(* IEC 61131-3 sources: volt/packages/volt-lsp-iec/test-corpus/pro2193/Device/Plc Logic/Application/09 Misc/Library Manager/BrinkEdgePcLogging, 50 files *)

(* ---- ANYNUMBER.dut ---- *)
TYPE ANYNUMBER :
UNION
	SINTVAL : SINT;
	USINTVAL : USINT;
	INTVAL : INT;
	UINTVAL : UINT;
	DINTVAL : DINT;
	UDINTVAL : UDINT;
	LINTVAL : LINT;
	ULINTVAL : ULINT;
	REALVALUE : REAL;
	LREALVALUE : LREAL;
END_UNION
END_TYPE

(* ---- CACHESTATUS.dut ---- *)
TYPE CACHESTATUS :
STRUCT
	LOCK : DWORD;
	COUNT : BYTE;
END_STRUCT
END_TYPE

(* ---- CAVITYPLCDATATYPES.dut ---- *)
TYPE CAVITYPLCDATATYPES :
STRUCT
	PRODUCED : PlcDataType := -1;
	UNCOUNTEDREJECT : PlcDataType := -1;
	REJECTED : PlcDataType := -1;
	REJECTREASONS : ARRAY [0..20] OF PlcDataType := [21(-1)];
	STACKED : PlcDataType := -1;
END_STRUCT
END_TYPE

(* ---- CLIENTSTATISTICS.dut ---- *)
TYPE CLIENTSTATISTICS :
STRUCT
	LOGFAILDISCONNECTED : ULINT;
	RECONNECTCOUNT : ULINT;
	LOSTDUETOCONNECTIONPROBLEMS : ULINT;
	KEEPALIVEMESSAGESSENT : ULINT;
	PLCDATATYPENOTDEFINED : ULINT;
	SENDNOTIMMEDIATELYCOMPLETED : ULINT;
	DATATOOLONG : ULINT;
	LOGQUEUESFULL : ULINT;
	LOGQUEUESBUSY : ULINT;
	ERRORWHILESENDINGDATA : ULINT;
	WRITEISBUSY : ULINT;
	TOOMANYWRITESPERCYCLE : ULINT;
END_STRUCT
END_TYPE

(* ---- CONNECTIONSPEED.dut ---- *)
TYPE CONNECTIONSPEED :
(
	S100MBPS := 100,
	S1000MBPS := 1000
);
END_TYPE

(* ---- DATATYPE.dut ---- *)
TYPE DATATYPE :
(
	NONE := -1,
	ULINTEGER := 0,
	INTEGER := 1,
	FLOAT := 2,
	BOOLEAN := 3,
	TEXT := 4
);
END_TYPE

(* ---- DEBUGLOGINFO.dut ---- *)
TYPE DEBUGLOGINFO :
STRUCT
	MSTIME : ULINT;
	DESCRIPTION : STRING(255);
END_STRUCT
END_TYPE

(* ---- LABELADJUSTMENTSPLCDATATYPESCONFIG.dut ---- *)
TYPE LABELADJUSTMENTSPLCDATATYPESCONFIG : ARRAY [1..2, 1..2, 1..32, 1..3] OF PlcDataType;
END_TYPE

(* ---- LOGCACHE.dut ---- *)
TYPE LOGCACHE : ARRAY [1..QueuesInCache] OF LogQueue;
END_TYPE

(* ---- LOGQUEUESTATS.dut ---- *)
TYPE LOGQUEUESTATS :
STRUCT
	ADDLOGFAILEDDUETOQUEUEFULL : ULINT;
END_STRUCT
END_TYPE

(* ---- LOGRECORD.dut ---- *)
TYPE LOGRECORD :
STRUCT
	PLCDATATYPE : PlcDataType;
	DATATYPE : DataType;
	PLCUTCTIME : ULINT;
	VALUE : NumberUnion;
END_STRUCT
END_TYPE

(* ---- LOGRECORDARRAY.dut ---- *)
TYPE LOGRECORDARRAY : ARRAY [1..GVL_Dashboard.LogQueueLength] OF LogRecord;
END_TYPE

(* ---- MOULDCONTROLCAVITYPLCDATATYPES.dut ---- *)
TYPE MOULDCONTROLCAVITYPLCDATATYPES :
STRUCT
	PEAKPRESSURE : PlcDataType := -1;
	TARGETVALUE : PlcDataType := -1;
	ACTUALVALUE : PlcDataType := -1;
END_STRUCT
END_TYPE

(* ---- MOULDCONTROLCAVITYPLCDATATYPESCONFIG.dut ---- *)
TYPE MOULDCONTROLCAVITYPLCDATATYPESCONFIG : ARRAY [1..64] OF MouldControlCavityPlcDataTypes;
END_TYPE

(* ---- MVACUUMSPLCDATATYPESCONFIG.dut ---- *)
TYPE MVACUUMSPLCDATATYPESCONFIG : ARRAY [1..2, 1..32] OF PlcDataType;
END_TYPE

(* ---- NUMBERUNION.dut ---- *)
TYPE NUMBERUNION :
UNION
	BOOLVALUE : BOOL;
	INTVALUE : LINT;
	UINTVALUE : ULINT;
	REALVALUE : LREAL;
END_UNION
END_TYPE

(* ---- PLCDATATYPE.dut ---- *)
TYPE PLCDATATYPE :
(
	MAIN_ROBOTSTATUS := 23,
	MAIN_ENABLEIML := 24,
	MAIN_ENABLEHMU := 25,
	MAIN_ENABLEVISION := 26,
	MAIN_RELAYS_HIGHVACUUMPUMPRUNNING := 27,
	MAIN_RELAYS_LOWVACUUMPUMPRUNNING := 28,
	RELAYS_MOULDAREAFREE := 29,
	RELAYS_ENABLEMOULDCLOSURE := 30,
	RELAYS_ENABLEFULLMOULDOPENING := 31,
	RELAYS_OPERATIONWITHROBOT := 32,
	RELAYS_ENABLEEJECTORBACK := 33,
	RELAYS_ENABLEEJECTORFORWARD := 34,
	RELAYS_ENABLECOREPOS1BACK := 35,
	RELAYS_ENABLECOREPOS2FORWARD := 36,
	RELAYS_GLOBALRESET := 37,
	RELAYS_MAINAIRVALVE := 38,
	RELAYS_YUNIT_MOTORCOOLING := 39,
	RELAYS_ENABLEFREQUENCYCONTROLLER := 40,
	RELAYS_SAFETYGATE := 41,
	YUNIT_ACTPOS := 42,
	YUNIT_ERRORID := 43,
	YUNIT_AXISERRORID := 44,
	YUNIT_DRIVEERRORID := 45,
	YUNIT_DRIVEUTILISATION := 46,
	YUNIT_MOTORUTILISATION := 47,
	XRUNIT_ACTPOS := 48,
	XRUNIT_ERRORID := 49,
	XRUNIT_AXISERRORID := 50,
	XRUNIT_DRIVEERRORID := 51,
	XRUNIT_DRIVEUTILISATION := 52,
	XRUNIT_MOTORUTILISATION := 53,
	XIUNIT_ACTPOS := 54,
	XIUNIT_ERRORID := 55,
	XIUNIT_AXISERRORID := 56,
	XIUNIT_DRIVEERRORID := 57,
	XIUNIT_DRIVEUTILISATION := 58,
	XIUNIT_MOTORUTILISATION := 59,
	XUUNIT_ACTPOS := 60,
	XUUNIT_ERRORID := 61,
	XUUNIT_AXISERRORID := 62,
	XUUNIT_DRIVEERRORID := 63,
	XUUNIT_DRIVEUTILISATION := 64,
	XUUNIT_MOTORUTILISATION := 65,
	CHAIN_ACTPOS := 66,
	CHAIN_ERRORID := 67,
	CHAIN_AXISERRORID := 68,
	CHAIN_DRIVEERRORID := 69,
	CHAIN_DRIVEUTILISATION := 70,
	CHAIN_MOTORUTILISATION := 71,
	MAGAZINE_M1_1_ACTPOS := 72,
	MAGAZINE_M1_1_ERRORID := 73,
	MAGAZINE_M1_1_AXISERRORID := 74,
	MAGAZINE_M1_1_DRIVEERRORID := 75,
	MAGAZINE_M1_1_DRIVEUTILISATION := 76,
	MAGAZINE_M1_1_MOTORUTILISATION := 77,
	MAGAZINE_M1_2_ACTPOS := 78,
	MAGAZINE_M1_2_ERRORID := 79,
	MAGAZINE_M1_2_AXISERRORID := 80,
	MAGAZINE_M1_2_DRIVEERRORID := 81,
	MAGAZINE_M1_2_DRIVEUTILISATION := 82,
	MAGAZINE_M1_2_MOTORUTILISATION := 83,
	ZUNIT_ACTPOS := 84,
	ZUNIT_ERRORID := 85,
	ZUNIT_AXISERRORID := 86,
	ZUNIT_DRIVEERRORID := 87,
	ZUNIT_DRIVEUTILISATION := 88,
	ZUNIT_MOTORUTILISATION := 89,
	YUNIT_ACTTORQUE := 90,
	XRUNIT_ACTTORQUE := 91,
	XIUNIT_ACTTORQUE := 92,
	XUUNIT_ACTTORQUE := 93,
	CHAIN_ACTTORQUE := 94,
	MAGAZINE_M1_1_ACTTORQUE := 95,
	MAGAZINE_M1_2_ACTTORQUE := 96,
	ZUNIT_ACTTORQUE := 97,
	YUNIT_COVEREDDISTANCE := 98,
	XRUNIT_COVEREDDISTANCE := 99,
	XIUNIT_COVEREDDISTANCE := 100,
	XUUNIT_COVEREDDISTANCE := 101,
	CHAIN_COVEREDDISTANCE := 102,
	MAGAZINE_M1_1_COVEREDDISTANCE := 103,
	MAGAZINE_M1_2_COVEREDDISTANCE := 104,
	ZUNIT_COVEREDDISTANCE := 105,
	CYCLETIMES_TIMESTOPPED := 106,
	CYCLETIMES_TIMERESETTING := 107,
	CYCLETIMES_TIMEIDLE := 108,
	CYCLETIMES_TIMEAUTOMATIC := 109,
	CYCLETIMES_AUTOMATICCYCLESTARTS := 110,
	YUNIT_ALARMS := 111,
	YUNIT_TIME_ACTIVE := 112,
	YUNIT_TIME_IDLE := 113,
	XRUNIT_ALARMS := 114,
	XRUNIT_TIME_ACTIVE := 115,
	XRUNIT_TIME_IDLE := 116,
	XIUNIT_ALARMS := 117,
	XIUNIT_TIME_ACTIVE := 118,
	XIUNIT_TIME_IDLE := 119,
	XUUNIT_ALARMS := 120,
	XUUNIT_TIME_ACTIVE := 121,
	XUUNIT_TIME_IDLE := 122,
	CHAIN_ALARMS := 123,
	CHAIN_TIME_ACTIVE := 124,
	CHAIN_TIME_IDLE := 125,
	MAGAZINE_M1_1_ALARMS := 126,
	MAGAZINE_M1_1_TIME_ACTIVE := 127,
	MAGAZINE_M1_1_TIME_IDLE := 128,
	MAGAZINE_M1_2_ALARMS := 129,
	MAGAZINE_M1_2_TIME_ACTIVE := 130,
	MAGAZINE_M1_2_TIME_IDLE := 131,
	ZUNIT_ALARMS := 132,
	ZUNIT_TIME_ACTIVE := 133,
	ZUNIT_TIME_IDLE := 134,
	CAMERA_ALARMS := 135,
	CAMERA_TIME_ACTIVE := 136,
	CAMERA_TIME_IDLE := 137,
	REJECTSTATION_ALARMS := 138,
	REJECTSTATION_TIME_ACTIVE := 139,
	REJECTSTATION_TIME_IDLE := 140,
	CONVEYORS_ALARMS := 141,
	CONVEYORS_TIME_ACTIVE := 142,
	CONVEYORS_TIME_IDLE := 143,
	IMM_CYCLETIMETAKEOUT := 144,
	IMM_CYCLETIMETOTAL := 145,
	IMM_SAVEDCYCLETIMEBYEARLYMOULDCLOSING := 146,
	XUUNIT_SENSORTIMES_VACUUM_1 := 147,
	XUUNIT_SENSORTIMES_VACUUM_2 := 148,
	XUUNIT_SENSORTIMES_VACUUM_3 := 149,
	XUUNIT_SENSORTIMES_SHIFTIN := 150,
	XUUNIT_SENSORTIMES_SHIFTOUT := 151,
	MAGAZINE_SENSORTIMES_VACUUM_1 := 152,
	MAGAZINE_SENSORTIMES_VACUUM_2 := 153,
	MAGAZINE_SENSORTIMES_VACUUM_3 := 154,
	MAGAZINE_SENSORTIMES_VACUUM_4 := 155,
	MAGAZINE_SENSORTIMES_FLIPLABEL1IN := 156,
	MAGAZINE_SENSORTIMES_FLIPLABEL1OUT := 157,
	MAGAZINE_SENSORTIMES_FLIPLABEL2IN := 158,
	MAGAZINE_SENSORTIMES_FLIPLABEL2OUT := 159,
	MAGAZINE_SENSORTIMES_CHANGEDRAWERIN := 160,
	MAGAZINE_SENSORTIMES_CHANGEDRAWEROUT := 161,
	MAGAZINE_SENSORTIMES_LOCKDRAWERIN := 162,
	MAGAZINE_SENSORTIMES_LOCKDRAWEROUT := 163,
	ZUNIT_SENSORTIMES_VACUUM_1 := 164,
	ZUNIT_SENSORTIMES_VACUUM_2 := 165,
	ZUNIT_SENSORTIMES_VACUUM_3 := 166,
	ZUNIT_SENSORTIMES_VACUUM_4 := 167,
	ZUNIT_SENSORTIMES_ROTATEIN := 168,
	ZUNIT_SENSORTIMES_ROTATEOUT := 169,
	ZUNIT_SENSORTIMES_EXTEND1IN := 170,
	ZUNIT_SENSORTIMES_EXTEND2IN := 171,
	ZUNIT_SENSORTIMES_EXTEND3IN := 172,
	ZUNIT_SENSORTIMES_EXTEND4IN := 173,
	REJECTSTATION_SENSORTIMES_REJECTCYLINDERIN := 174,
	REJECTSTATION_SENSORTIMES_REJECTCYLINDEROUT := 175,
	METADATA_REJECTREASON_0_DESCRIPTION := 176,
	METADATA_REJECTREASON_1_DESCRIPTION := 177,
	METADATA_REJECTREASON_2_DESCRIPTION := 178,
	METADATA_REJECTREASON_3_DESCRIPTION := 179,
	METADATA_REJECTREASON_4_DESCRIPTION := 180,
	METADATA_REJECTREASON_5_DESCRIPTION := 181,
	METADATA_REJECTREASON_6_DESCRIPTION := 182,
	PRODUCTIONCOUNTERS_TOTAL_PRODUCED := 183,
	PRODUCTIONCOUNTERS_TOTAL_STACKED := 184,
	PRODUCTIONCOUNTERS_TOTAL_REJECTED := 185,
	PRODUCTIONCOUNTERS_TOTAL_UNCOUNTEDREJECT := 186,
	PRODUCTIONCOUNTERS_TOTAL_REJECTREASON_0 := 187,
	PRODUCTIONCOUNTERS_TOTAL_REJECTREASON_1 := 188,
	PRODUCTIONCOUNTERS_TOTAL_REJECTREASON_2 := 189,
	PRODUCTIONCOUNTERS_TOTAL_REJECTREASON_3 := 190,
	PRODUCTIONCOUNTERS_TOTAL_REJECTREASON_4 := 191,
	PRODUCTIONCOUNTERS_TOTAL_REJECTREASON_5 := 192,
	PRODUCTIONCOUNTERS_TOTAL_REJECTREASON_6 := 193,
	PRODUCTIONCOUNTERS_CAVITY_1_PRODUCED := 194,
	PRODUCTIONCOUNTERS_CAVITY_1_STACKED := 195,
	PRODUCTIONCOUNTERS_CAVITY_1_REJECTED := 196,
	PRODUCTIONCOUNTERS_CAVITY_1_UNCOUNTEDREJECT := 197,
	PRODUCTIONCOUNTERS_CAVITY_1_REJECTREASON_0 := 198,
	PRODUCTIONCOUNTERS_CAVITY_1_REJECTREASON_1 := 199,
	PRODUCTIONCOUNTERS_CAVITY_1_REJECTREASON_2 := 200,
	PRODUCTIONCOUNTERS_CAVITY_1_REJECTREASON_3 := 201,
	PRODUCTIONCOUNTERS_CAVITY_1_REJECTREASON_4 := 202,
	PRODUCTIONCOUNTERS_CAVITY_1_REJECTREASON_5 := 203,
	PRODUCTIONCOUNTERS_CAVITY_1_REJECTREASON_6 := 204,
	PRODUCTIONCOUNTERS_CAVITY_2_PRODUCED := 205,
	PRODUCTIONCOUNTERS_CAVITY_2_STACKED := 206,
	PRODUCTIONCOUNTERS_CAVITY_2_REJECTED := 207,
	PRODUCTIONCOUNTERS_CAVITY_2_UNCOUNTEDREJECT := 208,
	PRODUCTIONCOUNTERS_CAVITY_2_REJECTREASON_0 := 209,
	PRODUCTIONCOUNTERS_CAVITY_2_REJECTREASON_1 := 210,
	PRODUCTIONCOUNTERS_CAVITY_2_REJECTREASON_2 := 211,
	PRODUCTIONCOUNTERS_CAVITY_2_REJECTREASON_3 := 212,
	PRODUCTIONCOUNTERS_CAVITY_2_REJECTREASON_4 := 213,
	PRODUCTIONCOUNTERS_CAVITY_2_REJECTREASON_5 := 214,
	PRODUCTIONCOUNTERS_CAVITY_2_REJECTREASON_6 := 215,
	PRODUCTIONCOUNTERS_CAVITY_3_PRODUCED := 216,
	PRODUCTIONCOUNTERS_CAVITY_3_STACKED := 217,
	PRODUCTIONCOUNTERS_CAVITY_3_REJECTED := 218,
	PRODUCTIONCOUNTERS_CAVITY_3_UNCOUNTEDREJECT := 219,
	PRODUCTIONCOUNTERS_CAVITY_3_REJECTREASON_0 := 220,
	PRODUCTIONCOUNTERS_CAVITY_3_REJECTREASON_1 := 221,
	PRODUCTIONCOUNTERS_CAVITY_3_REJECTREASON_2 := 222,
	PRODUCTIONCOUNTERS_CAVITY_3_REJECTREASON_3 := 223,
	PRODUCTIONCOUNTERS_CAVITY_3_REJECTREASON_4 := 224,
	PRODUCTIONCOUNTERS_CAVITY_3_REJECTREASON_5 := 225,
	PRODUCTIONCOUNTERS_CAVITY_3_REJECTREASON_6 := 226,
	PRODUCTIONCOUNTERS_CAVITY_4_PRODUCED := 227,
	PRODUCTIONCOUNTERS_CAVITY_4_STACKED := 228,
	PRODUCTIONCOUNTERS_CAVITY_4_REJECTED := 229,
	PRODUCTIONCOUNTERS_CAVITY_4_UNCOUNTEDREJECT := 230,
	PRODUCTIONCOUNTERS_CAVITY_4_REJECTREASON_0 := 231,
	PRODUCTIONCOUNTERS_CAVITY_4_REJECTREASON_1 := 232,
	PRODUCTIONCOUNTERS_CAVITY_4_REJECTREASON_2 := 233,
	PRODUCTIONCOUNTERS_CAVITY_4_REJECTREASON_3 := 234,
	PRODUCTIONCOUNTERS_CAVITY_4_REJECTREASON_4 := 235,
	PRODUCTIONCOUNTERS_CAVITY_4_REJECTREASON_5 := 236,
	PRODUCTIONCOUNTERS_CAVITY_4_REJECTREASON_6 := 237,
	PRODUCTIONCOUNTERS_CAVITY_5_PRODUCED := 238,
	PRODUCTIONCOUNTERS_CAVITY_5_STACKED := 239,
	PRODUCTIONCOUNTERS_CAVITY_5_REJECTED := 240,
	PRODUCTIONCOUNTERS_CAVITY_5_UNCOUNTEDREJECT := 241,
	PRODUCTIONCOUNTERS_CAVITY_5_REJECTREASON_0 := 242,
	PRODUCTIONCOUNTERS_CAVITY_5_REJECTREASON_1 := 243,
	PRODUCTIONCOUNTERS_CAVITY_5_REJECTREASON_2 := 244,
	PRODUCTIONCOUNTERS_CAVITY_5_REJECTREASON_3 := 245,
	PRODUCTIONCOUNTERS_CAVITY_5_REJECTREASON_4 := 246,
	PRODUCTIONCOUNTERS_CAVITY_5_REJECTREASON_5 := 247,
	PRODUCTIONCOUNTERS_CAVITY_5_REJECTREASON_6 := 248,
	PRODUCTIONCOUNTERS_CAVITY_6_PRODUCED := 249,
	PRODUCTIONCOUNTERS_CAVITY_6_STACKED := 250,
	PRODUCTIONCOUNTERS_CAVITY_6_REJECTED := 251,
	PRODUCTIONCOUNTERS_CAVITY_6_UNCOUNTEDREJECT := 252,
	PRODUCTIONCOUNTERS_CAVITY_6_REJECTREASON_0 := 253,
	PRODUCTIONCOUNTERS_CAVITY_6_REJECTREASON_1 := 254,
	PRODUCTIONCOUNTERS_CAVITY_6_REJECTREASON_2 := 255,
	PRODUCTIONCOUNTERS_CAVITY_6_REJECTREASON_3 := 256,
	PRODUCTIONCOUNTERS_CAVITY_6_REJECTREASON_4 := 257,
	PRODUCTIONCOUNTERS_CAVITY_6_REJECTREASON_5 := 258,
	PRODUCTIONCOUNTERS_CAVITY_6_REJECTREASON_6 := 259,
	MAIN_RECIPENAME := 260,
	MAIN_RECIPENAME_CASSETTE := 261,
	MAIN_PARAMETERCHANGED := 262,
	MAIN_AIRPRESSUREOK := 263,
	MAIN_GENERALALARMACTIVE := 264,
	MAIN_GENERALWARNINGACTIVE := 265,
	MAIN_ALARMS := 266,
	MAIN_ALARMSFUSE := 267,
	MAIN_ALARMSIMM := 268,
	MAIN_MESSAGES := 269,
	MAIN_WARNINGS := 270,
	MAGAZINE_ALARMS := 273,
	YUNIT_ALARMSMOTIONCONTROL := 274,
	MAIN_SAFETYPLCSTATUS1 := 275,
	MAIN_SAFETYPLCSTATUS2 := 276,
	MAIN_SAFETYPLCSTATUS3 := 277,
	ROBOTCONNECTED := 278,
	ZUNIT_SENSORTIMES_SHIFT1IN := 279,
	ZUNIT_SENSORTIMES_SHIFT1OUT := 280,
	MAIN_SER_STATE := 281,
	MAIN_SER_OPERATIONMODE := 282,
	MAIN_RECIPENAME_BRINK := 283,
	REJECTSTATION_SENSORTIMES_REJECTCYLINDER2IN := 284,
	REJECTSTATION_SENSORTIMES_REJECTCYLINDER2OUT := 285,
	XUUNIT_SENSORTIMES_SHIFTHORIZONTALIN := 286,
	XUUNIT_SENSORTIMES_SHIFTHORIZONTALOUT := 287,
	XUUNIT_SENSORTIMES_SHIFTVERTICALIN := 288,
	XUUNIT_SENSORTIMES_SHIFTVERTICALOUT := 289,
	METADATA_REJECTREASON_7_DESCRIPTION := 290,
	PRODUCTIONCOUNTERS_TOTAL_REJECTREASON_7 := 291,
	PRODUCTIONCOUNTERS_CAVITY_1_REJECTREASON_7 := 292,
	PRODUCTIONCOUNTERS_CAVITY_2_REJECTREASON_7 := 293,
	PRODUCTIONCOUNTERS_CAVITY_3_REJECTREASON_7 := 294,
	PRODUCTIONCOUNTERS_CAVITY_4_REJECTREASON_7 := 295,
	PRODUCTIONCOUNTERS_CAVITY_5_REJECTREASON_7 := 296,
	PRODUCTIONCOUNTERS_CAVITY_6_REJECTREASON_7 := 297,
	MOULDMEASUREMENT_MAXPRESSURE := 298,
	MOULDMEASUREMENT_MINPRESSURE := 299,
	MOULDMEASUREMENT_IDEALPRESSURE := 300,
	MOULDMEASUREMENT_AVERAGEPRESSURE := 301,
	MOULDMEASUREMENT_CALCULATEDIDEALPRESSURE := 302,
	MOULDMEASUREMENT_HOLDINGPRESSURE_TARGETVALUE := 303,
	MOULDMEASUREMENT_HOLDINGPRESSURE_ACTUALVALUE := 304,
	MOULDMEASUREMENT_SWITCHOVERPOINT_TARGETVALUE := 305,
	MOULDMEASUREMENT_SWITCHOVERPOINT_ACTUALVALUE := 306,
	MOULDMEASUREMENT_CAVITY_1_PEAKPRESSURE := 307,
	MOULDMEASUREMENT_CAVITY_2_PEAKPRESSURE := 308,
	MOULDMEASUREMENT_CAVITY_3_PEAKPRESSURE := 309,
	MOULDMEASUREMENT_CAVITY_4_PEAKPRESSURE := 310,
	MOULDMEASUREMENT_CAVITY_5_PEAKPRESSURE := 311,
	MOULDMEASUREMENT_CAVITY_6_PEAKPRESSURE := 312,
	MOULDMEASUREMENT_HOTRUNNER_CAVITY_1_TARGETVALUE := 313,
	MOULDMEASUREMENT_HOTRUNNER_CAVITY_1_ACTUALVALUE := 314,
	MOULDMEASUREMENT_HOTRUNNER_CAVITY_2_TARGETVALUE := 315,
	MOULDMEASUREMENT_HOTRUNNER_CAVITY_2_ACTUALVALUE := 316,
	MOULDMEASUREMENT_HOTRUNNER_CAVITY_3_TARGETVALUE := 317,
	MOULDMEASUREMENT_HOTRUNNER_CAVITY_3_ACTUALVALUE := 318,
	MOULDMEASUREMENT_HOTRUNNER_CAVITY_4_TARGETVALUE := 319,
	MOULDMEASUREMENT_HOTRUNNER_CAVITY_4_ACTUALVALUE := 320,
	MOULDMEASUREMENT_HOTRUNNER_CAVITY_5_TARGETVALUE := 321,
	MOULDMEASUREMENT_HOTRUNNER_CAVITY_5_ACTUALVALUE := 322,
	MOULDMEASUREMENT_HOTRUNNER_CAVITY_6_TARGETVALUE := 323,
	MOULDMEASUREMENT_HOTRUNNER_CAVITY_6_ACTUALVALUE := 324,
	METADATA_REJECTREASON_8_DESCRIPTION := 325,
	PRODUCTIONCOUNTERS_TOTAL_REJECTREASON_8 := 326,
	PRODUCTIONCOUNTERS_CAVITY_1_REJECTREASON_8 := 327,
	PRODUCTIONCOUNTERS_CAVITY_2_REJECTREASON_8 := 328,
	PRODUCTIONCOUNTERS_CAVITY_3_REJECTREASON_8 := 329,
	PRODUCTIONCOUNTERS_CAVITY_4_REJECTREASON_8 := 330,
	PRODUCTIONCOUNTERS_CAVITY_5_REJECTREASON_8 := 331,
	PRODUCTIONCOUNTERS_CAVITY_6_REJECTREASON_8 := 332,
	METADATA_REJECTREASON_9_DESCRIPTION := 333,
	PRODUCTIONCOUNTERS_TOTAL_REJECTREASON_9 := 334,
	PRODUCTIONCOUNTERS_CAVITY_1_REJECTREASON_9 := 335,
	PRODUCTIONCOUNTERS_CAVITY_2_REJECTREASON_9 := 336,
	PRODUCTIONCOUNTERS_CAVITY_3_REJECTREASON_9 := 337,
	PRODUCTIONCOUNTERS_CAVITY_4_REJECTREASON_9 := 338,
	PRODUCTIONCOUNTERS_CAVITY_5_REJECTREASON_9 := 339,
	PRODUCTIONCOUNTERS_CAVITY_6_REJECTREASON_9 := 340,
	METADATA_REJECTREASON_10_DESCRIPTION := 341,
	PRODUCTIONCOUNTERS_TOTAL_REJECTREASON_10 := 342,
	PRODUCTIONCOUNTERS_CAVITY_1_REJECTREASON_10 := 343,
	PRODUCTIONCOUNTERS_CAVITY_2_REJECTREASON_10 := 344,
	PRODUCTIONCOUNTERS_CAVITY_3_REJECTREASON_10 := 345,
	PRODUCTIONCOUNTERS_CAVITY_4_REJECTREASON_10 := 346,
	PRODUCTIONCOUNTERS_CAVITY_5_REJECTREASON_10 := 347,
	PRODUCTIONCOUNTERS_CAVITY_6_REJECTREASON_10 := 348,
	METADATA_REJECTREASON_11_DESCRIPTION := 349,
	PRODUCTIONCOUNTERS_TOTAL_REJECTREASON_11 := 350,
	PRODUCTIONCOUNTERS_CAVITY_1_REJECTREASON_11 := 351,
	PRODUCTIONCOUNTERS_CAVITY_2_REJECTREASON_11 := 352,
	PRODUCTIONCOUNTERS_CAVITY_3_REJECTREASON_11 := 353,
	PRODUCTIONCOUNTERS_CAVITY_4_REJECTREASON_11 := 354,
	PRODUCTIONCOUNTERS_CAVITY_5_REJECTREASON_11 := 355,
	PRODUCTIONCOUNTERS_CAVITY_6_REJECTREASON_11 := 356,
	METADATA_REJECTREASON_12_DESCRIPTION := 357,
	PRODUCTIONCOUNTERS_TOTAL_REJECTREASON_12 := 358,
	PRODUCTIONCOUNTERS_CAVITY_1_REJECTREASON_12 := 359,
	PRODUCTIONCOUNTERS_CAVITY_2_REJECTREASON_12 := 360,
	PRODUCTIONCOUNTERS_CAVITY_3_REJECTREASON_12 := 361,
	PRODUCTIONCOUNTERS_CAVITY_4_REJECTREASON_12 := 362,
	PRODUCTIONCOUNTERS_CAVITY_5_REJECTREASON_12 := 363,
	PRODUCTIONCOUNTERS_CAVITY_6_REJECTREASON_12 := 364,
	METADATA_REJECTREASON_13_DESCRIPTION := 365,
	PRODUCTIONCOUNTERS_TOTAL_REJECTREASON_13 := 366,
	PRODUCTIONCOUNTERS_CAVITY_1_REJECTREASON_13 := 367,
	PRODUCTIONCOUNTERS_CAVITY_2_REJECTREASON_13 := 368,
	PRODUCTIONCOUNTERS_CAVITY_3_REJECTREASON_13 := 369,
	PRODUCTIONCOUNTERS_CAVITY_4_REJECTREASON_13 := 370,
	PRODUCTIONCOUNTERS_CAVITY_5_REJECTREASON_13 := 371,
	PRODUCTIONCOUNTERS_CAVITY_6_REJECTREASON_13 := 372,
	METADATA_REJECTREASON_14_DESCRIPTION := 373,
	PRODUCTIONCOUNTERS_TOTAL_REJECTREASON_14 := 374,
	PRODUCTIONCOUNTERS_CAVITY_1_REJECTREASON_14 := 375,
	PRODUCTIONCOUNTERS_CAVITY_2_REJECTREASON_14 := 376,
	PRODUCTIONCOUNTERS_CAVITY_3_REJECTREASON_14 := 377,
	PRODUCTIONCOUNTERS_CAVITY_4_REJECTREASON_14 := 378,
	PRODUCTIONCOUNTERS_CAVITY_5_REJECTREASON_14 := 379,
	PRODUCTIONCOUNTERS_CAVITY_6_REJECTREASON_14 := 380,
	METADATA_REJECTREASON_15_DESCRIPTION := 381,
	PRODUCTIONCOUNTERS_TOTAL_REJECTREASON_15 := 382,
	PRODUCTIONCOUNTERS_CAVITY_1_REJECTREASON_15 := 383,
	PRODUCTIONCOUNTERS_CAVITY_2_REJECTREASON_15 := 384,
	PRODUCTIONCOUNTERS_CAVITY_3_REJECTREASON_15 := 385,
	PRODUCTIONCOUNTERS_CAVITY_4_REJECTREASON_15 := 386,
	PRODUCTIONCOUNTERS_CAVITY_5_REJECTREASON_15 := 387,
	PRODUCTIONCOUNTERS_CAVITY_6_REJECTREASON_15 := 388,
	METADATA_REJECTREASON_16_DESCRIPTION := 389,
	PRODUCTIONCOUNTERS_TOTAL_REJECTREASON_16 := 390,
	PRODUCTIONCOUNTERS_CAVITY_1_REJECTREASON_16 := 391,
	PRODUCTIONCOUNTERS_CAVITY_2_REJECTREASON_16 := 392,
	PRODUCTIONCOUNTERS_CAVITY_3_REJECTREASON_16 := 393,
	PRODUCTIONCOUNTERS_CAVITY_4_REJECTREASON_16 := 394,
	PRODUCTIONCOUNTERS_CAVITY_5_REJECTREASON_16 := 395,
	PRODUCTIONCOUNTERS_CAVITY_6_REJECTREASON_16 := 396,
	METADATA_REJECTREASON_17_DESCRIPTION := 397,
	PRODUCTIONCOUNTERS_TOTAL_REJECTREASON_17 := 398,
	PRODUCTIONCOUNTERS_CAVITY_1_REJECTREASON_17 := 399,
	PRODUCTIONCOUNTERS_CAVITY_2_REJECTREASON_17 := 400,
	PRODUCTIONCOUNTERS_CAVITY_3_REJECTREASON_17 := 401,
	PRODUCTIONCOUNTERS_CAVITY_4_REJECTREASON_17 := 402,
	PRODUCTIONCOUNTERS_CAVITY_5_REJECTREASON_17 := 403,
	PRODUCTIONCOUNTERS_CAVITY_6_REJECTREASON_17 := 404,
	METADATA_REJECTREASON_18_DESCRIPTION := 405,
	PRODUCTIONCOUNTERS_TOTAL_REJECTREASON_18 := 406,
	PRODUCTIONCOUNTERS_CAVITY_1_REJECTREASON_18 := 407,
	PRODUCTIONCOUNTERS_CAVITY_2_REJECTREASON_18 := 408,
	PRODUCTIONCOUNTERS_CAVITY_3_REJECTREASON_18 := 409,
	PRODUCTIONCOUNTERS_CAVITY_4_REJECTREASON_18 := 410,
	PRODUCTIONCOUNTERS_CAVITY_5_REJECTREASON_18 := 411,
	PRODUCTIONCOUNTERS_CAVITY_6_REJECTREASON_18 := 412,
	METADATA_REJECTREASON_19_DESCRIPTION := 413,
	PRODUCTIONCOUNTERS_TOTAL_REJECTREASON_19 := 414,
	PRODUCTIONCOUNTERS_CAVITY_1_REJECTREASON_19 := 415,
	PRODUCTIONCOUNTERS_CAVITY_2_REJECTREASON_19 := 416,
	PRODUCTIONCOUNTERS_CAVITY_3_REJECTREASON_19 := 417,
	PRODUCTIONCOUNTERS_CAVITY_4_REJECTREASON_19 := 418,
	PRODUCTIONCOUNTERS_CAVITY_5_REJECTREASON_19 := 419,
	PRODUCTIONCOUNTERS_CAVITY_6_REJECTREASON_19 := 420,
	METADATA_REJECTREASON_20_DESCRIPTION := 421,
	PRODUCTIONCOUNTERS_TOTAL_REJECTREASON_20 := 422,
	PRODUCTIONCOUNTERS_CAVITY_1_REJECTREASON_20 := 423,
	PRODUCTIONCOUNTERS_CAVITY_2_REJECTREASON_20 := 424,
	PRODUCTIONCOUNTERS_CAVITY_3_REJECTREASON_20 := 425,
	PRODUCTIONCOUNTERS_CAVITY_4_REJECTREASON_20 := 426,
	PRODUCTIONCOUNTERS_CAVITY_5_REJECTREASON_20 := 427,
	PRODUCTIONCOUNTERS_CAVITY_6_REJECTREASON_20 := 428,
	PRODUCTIONCOUNTERS_CAVITY_7_PRODUCED := 429,
	PRODUCTIONCOUNTERS_CAVITY_7_STACKED := 430,
	PRODUCTIONCOUNTERS_CAVITY_7_REJECTED := 431,
	PRODUCTIONCOUNTERS_CAVITY_7_UNCOUNTEDREJECT := 432,
	PRODUCTIONCOUNTERS_CAVITY_7_REJECTREASON_0 := 433,
	PRODUCTIONCOUNTERS_CAVITY_7_REJECTREASON_1 := 434,
	PRODUCTIONCOUNTERS_CAVITY_7_REJECTREASON_2 := 435,
	PRODUCTIONCOUNTERS_CAVITY_7_REJECTREASON_3 := 436,
	PRODUCTIONCOUNTERS_CAVITY_7_REJECTREASON_4 := 437,
	PRODUCTIONCOUNTERS_CAVITY_7_REJECTREASON_5 := 438,
	PRODUCTIONCOUNTERS_CAVITY_7_REJECTREASON_6 := 439,
	PRODUCTIONCOUNTERS_CAVITY_7_REJECTREASON_7 := 440,
	PRODUCTIONCOUNTERS_CAVITY_7_REJECTREASON_8 := 441,
	PRODUCTIONCOUNTERS_CAVITY_7_REJECTREASON_9 := 442,
	PRODUCTIONCOUNTERS_CAVITY_7_REJECTREASON_10 := 443,
	PRODUCTIONCOUNTERS_CAVITY_7_REJECTREASON_11 := 444,
	PRODUCTIONCOUNTERS_CAVITY_7_REJECTREASON_12 := 445,
	PRODUCTIONCOUNTERS_CAVITY_7_REJECTREASON_13 := 446,
	PRODUCTIONCOUNTERS_CAVITY_7_REJECTREASON_14 := 447,
	PRODUCTIONCOUNTERS_CAVITY_7_REJECTREASON_15 := 448,
	PRODUCTIONCOUNTERS_CAVITY_7_REJECTREASON_16 := 449,
	PRODUCTIONCOUNTERS_CAVITY_7_REJECTREASON_17 := 450,
	PRODUCTIONCOUNTERS_CAVITY_7_REJECTREASON_18 := 451,
	PRODUCTIONCOUNTERS_CAVITY_7_REJECTREASON_19 := 452,
	PRODUCTIONCOUNTERS_CAVITY_7_REJECTREASON_20 := 453,
	MOULDMEASUREMENT_CAVITY_7_PEAKPRESSURE := 454,
	MOULDMEASUREMENT_HOTRUNNER_CAVITY_7_TARGETVALUE := 455,
	MOULDMEASUREMENT_HOTRUNNER_CAVITY_7_ACTUALVALUE := 456,
	PRODUCTIONCOUNTERS_CAVITY_8_PRODUCED := 457,
	PRODUCTIONCOUNTERS_CAVITY_8_STACKED := 458,
	PRODUCTIONCOUNTERS_CAVITY_8_REJECTED := 459,
	PRODUCTIONCOUNTERS_CAVITY_8_UNCOUNTEDREJECT := 460,
	PRODUCTIONCOUNTERS_CAVITY_8_REJECTREASON_0 := 461,
	PRODUCTIONCOUNTERS_CAVITY_8_REJECTREASON_1 := 462,
	PRODUCTIONCOUNTERS_CAVITY_8_REJECTREASON_2 := 463,
	PRODUCTIONCOUNTERS_CAVITY_8_REJECTREASON_3 := 464,
	PRODUCTIONCOUNTERS_CAVITY_8_REJECTREASON_4 := 465,
	PRODUCTIONCOUNTERS_CAVITY_8_REJECTREASON_5 := 466,
	PRODUCTIONCOUNTERS_CAVITY_8_REJECTREASON_6 := 467,
	PRODUCTIONCOUNTERS_CAVITY_8_REJECTREASON_7 := 468,
	PRODUCTIONCOUNTERS_CAVITY_8_REJECTREASON_8 := 469,
	PRODUCTIONCOUNTERS_CAVITY_8_REJECTREASON_9 := 470,
	PRODUCTIONCOUNTERS_CAVITY_8_REJECTREASON_10 := 471,
	PRODUCTIONCOUNTERS_CAVITY_8_REJECTREASON_11 := 472,
	PRODUCTIONCOUNTERS_CAVITY_8_REJECTREASON_12 := 473,
	PRODUCTIONCOUNTERS_CAVITY_8_REJECTREASON_13 := 474,
	PRODUCTIONCOUNTERS_CAVITY_8_REJECTREASON_14 := 475,
	PRODUCTIONCOUNTERS_CAVITY_8_REJECTREASON_15 := 476,
	PRODUCTIONCOUNTERS_CAVITY_8_REJECTREASON_16 := 477,
	PRODUCTIONCOUNTERS_CAVITY_8_REJECTREASON_17 := 478,
	PRODUCTIONCOUNTERS_CAVITY_8_REJECTREASON_18 := 479,
	PRODUCTIONCOUNTERS_CAVITY_8_REJECTREASON_19 := 480,
	PRODUCTIONCOUNTERS_CAVITY_8_REJECTREASON_20 := 481,
	MOULDMEASUREMENT_CAVITY_8_PEAKPRESSURE := 482,
	MOULDMEASUREMENT_HOTRUNNER_CAVITY_8_TARGETVALUE := 483,
	MOULDMEASUREMENT_HOTRUNNER_CAVITY_8_ACTUALVALUE := 484,
	PRODUCTIONCOUNTERS_CAVITY_9_PRODUCED := 485,
	PRODUCTIONCOUNTERS_CAVITY_9_STACKED := 486,
	PRODUCTIONCOUNTERS_CAVITY_9_REJECTED := 487,
	PRODUCTIONCOUNTERS_CAVITY_9_UNCOUNTEDREJECT := 488,
	PRODUCTIONCOUNTERS_CAVITY_9_REJECTREASON_0 := 489,
	PRODUCTIONCOUNTERS_CAVITY_9_REJECTREASON_1 := 490,
	PRODUCTIONCOUNTERS_CAVITY_9_REJECTREASON_2 := 491,
	PRODUCTIONCOUNTERS_CAVITY_9_REJECTREASON_3 := 492,
	PRODUCTIONCOUNTERS_CAVITY_9_REJECTREASON_4 := 493,
	PRODUCTIONCOUNTERS_CAVITY_9_REJECTREASON_5 := 494,
	PRODUCTIONCOUNTERS_CAVITY_9_REJECTREASON_6 := 495,
	PRODUCTIONCOUNTERS_CAVITY_9_REJECTREASON_7 := 496,
	PRODUCTIONCOUNTERS_CAVITY_9_REJECTREASON_8 := 497,
	PRODUCTIONCOUNTERS_CAVITY_9_REJECTREASON_9 := 498,
	PRODUCTIONCOUNTERS_CAVITY_9_REJECTREASON_10 := 499,
	PRODUCTIONCOUNTERS_CAVITY_9_REJECTREASON_11 := 500,
	PRODUCTIONCOUNTERS_CAVITY_9_REJECTREASON_12 := 501,
	PRODUCTIONCOUNTERS_CAVITY_9_REJECTREASON_13 := 502,
	PRODUCTIONCOUNTERS_CAVITY_9_REJECTREASON_14 := 503,
	PRODUCTIONCOUNTERS_CAVITY_9_REJECTREASON_15 := 504,
	PRODUCTIONCOUNTERS_CAVITY_9_REJECTREASON_16 := 505,
	PRODUCTIONCOUNTERS_CAVITY_9_REJECTREASON_17 := 506,
	PRODUCTIONCOUNTERS_CAVITY_9_REJECTREASON_18 := 507,
	PRODUCTIONCOUNTERS_CAVITY_9_REJECTREASON_19 := 508,
	PRODUCTIONCOUNTERS_CAVITY_9_REJECTREASON_20 := 509,
	MOULDMEASUREMENT_CAVITY_9_PEAKPRESSURE := 510,
	MOULDMEASUREMENT_HOTRUNNER_CAVITY_9_TARGETVALUE := 511,
	MOULDMEASUREMENT_HOTRUNNER_CAVITY_9_ACTUALVALUE := 512,
	PRODUCTIONCOUNTERS_CAVITY_10_PRODUCED := 513,
	PRODUCTIONCOUNTERS_CAVITY_10_STACKED := 514,
	PRODUCTIONCOUNTERS_CAVITY_10_REJECTED := 515,
	PRODUCTIONCOUNTERS_CAVITY_10_UNCOUNTEDREJECT := 516,
	PRODUCTIONCOUNTERS_CAVITY_10_REJECTREASON_0 := 517,
	PRODUCTIONCOUNTERS_CAVITY_10_REJECTREASON_1 := 518,
	PRODUCTIONCOUNTERS_CAVITY_10_REJECTREASON_2 := 519,
	PRODUCTIONCOUNTERS_CAVITY_10_REJECTREASON_3 := 520,
	PRODUCTIONCOUNTERS_CAVITY_10_REJECTREASON_4 := 521,
	PRODUCTIONCOUNTERS_CAVITY_10_REJECTREASON_5 := 522,
	PRODUCTIONCOUNTERS_CAVITY_10_REJECTREASON_6 := 523,
	PRODUCTIONCOUNTERS_CAVITY_10_REJECTREASON_7 := 524,
	PRODUCTIONCOUNTERS_CAVITY_10_REJECTREASON_8 := 525,
	PRODUCTIONCOUNTERS_CAVITY_10_REJECTREASON_9 := 526,
	PRODUCTIONCOUNTERS_CAVITY_10_REJECTREASON_10 := 527,
	PRODUCTIONCOUNTERS_CAVITY_10_REJECTREASON_11 := 528,
	PRODUCTIONCOUNTERS_CAVITY_10_REJECTREASON_12 := 529,
	PRODUCTIONCOUNTERS_CAVITY_10_REJECTREASON_13 := 530,
	PRODUCTIONCOUNTERS_CAVITY_10_REJECTREASON_14 := 531,
	PRODUCTIONCOUNTERS_CAVITY_10_REJECTREASON_15 := 532,
	PRODUCTIONCOUNTERS_CAVITY_10_REJECTREASON_16 := 533,
	PRODUCTIONCOUNTERS_CAVITY_10_REJECTREASON_17 := 534,
	PRODUCTIONCOUNTERS_CAVITY_10_REJECTREASON_18 := 535,
	PRODUCTIONCOUNTERS_CAVITY_10_REJECTREASON_19 := 536,
	PRODUCTIONCOUNTERS_CAVITY_10_REJECTREASON_20 := 537,
	MOULDMEASUREMENT_CAVITY_10_PEAKPRESSURE := 538,
	MOULDMEASUREMENT_HOTRUNNER_CAVITY_10_TARGETVALUE := 539,
	MOULDMEASUREMENT_HOTRUNNER_CAVITY_10_ACTUALVALUE := 540,
	PRODUCTIONCOUNTERS_CAVITY_11_PRODUCED := 541,
	PRODUCTIONCOUNTERS_CAVITY_11_STACKED := 542,
	PRODUCTIONCOUNTERS_CAVITY_11_REJECTED := 543,
	PRODUCTIONCOUNTERS_CAVITY_11_UNCOUNTEDREJECT := 544,
	PRODUCTIONCOUNTERS_CAVITY_11_REJECTREASON_0 := 545,
	PRODUCTIONCOUNTERS_CAVITY_11_REJECTREASON_1 := 546,
	PRODUCTIONCOUNTERS_CAVITY_11_REJECTREASON_2 := 547,
	PRODUCTIONCOUNTERS_CAVITY_11_REJECTREASON_3 := 548,
	PRODUCTIONCOUNTERS_CAVITY_11_REJECTREASON_4 := 549,
	PRODUCTIONCOUNTERS_CAVITY_11_REJECTREASON_5 := 550,
	PRODUCTIONCOUNTERS_CAVITY_11_REJECTREASON_6 := 551,
	PRODUCTIONCOUNTERS_CAVITY_11_REJECTREASON_7 := 552,
	PRODUCTIONCOUNTERS_CAVITY_11_REJECTREASON_8 := 553,
	PRODUCTIONCOUNTERS_CAVITY_11_REJECTREASON_9 := 554,
	PRODUCTIONCOUNTERS_CAVITY_11_REJECTREASON_10 := 555,
	PRODUCTIONCOUNTERS_CAVITY_11_REJECTREASON_11 := 556,
	PRODUCTIONCOUNTERS_CAVITY_11_REJECTREASON_12 := 557,
	PRODUCTIONCOUNTERS_CAVITY_11_REJECTREASON_13 := 558,
	PRODUCTIONCOUNTERS_CAVITY_11_REJECTREASON_14 := 559,
	PRODUCTIONCOUNTERS_CAVITY_11_REJECTREASON_15 := 560,
	PRODUCTIONCOUNTERS_CAVITY_11_REJECTREASON_16 := 561,
	PRODUCTIONCOUNTERS_CAVITY_11_REJECTREASON_17 := 562,
	PRODUCTIONCOUNTERS_CAVITY_11_REJECTREASON_18 := 563,
	PRODUCTIONCOUNTERS_CAVITY_11_REJECTREASON_19 := 564,
	PRODUCTIONCOUNTERS_CAVITY_11_REJECTREASON_20 := 565,
	MOULDMEASUREMENT_CAVITY_11_PEAKPRESSURE := 566,
	MOULDMEASUREMENT_HOTRUNNER_CAVITY_11_TARGETVALUE := 567,
	MOULDMEASUREMENT_HOTRUNNER_CAVITY_11_ACTUALVALUE := 568,
	PRODUCTIONCOUNTERS_CAVITY_12_PRODUCED := 569,
	PRODUCTIONCOUNTERS_CAVITY_12_STACKED := 570,
	PRODUCTIONCOUNTERS_CAVITY_12_REJECTED := 571,
	PRODUCTIONCOUNTERS_CAVITY_12_UNCOUNTEDREJECT := 572,
	PRODUCTIONCOUNTERS_CAVITY_12_REJECTREASON_0 := 573,
	PRODUCTIONCOUNTERS_CAVITY_12_REJECTREASON_1 := 574,
	PRODUCTIONCOUNTERS_CAVITY_12_REJECTREASON_2 := 575,
	PRODUCTIONCOUNTERS_CAVITY_12_REJECTREASON_3 := 576,
	PRODUCTIONCOUNTERS_CAVITY_12_REJECTREASON_4 := 577,
	PRODUCTIONCOUNTERS_CAVITY_12_REJECTREASON_5 := 578,
	PRODUCTIONCOUNTERS_CAVITY_12_REJECTREASON_6 := 579,
	PRODUCTIONCOUNTERS_CAVITY_12_REJECTREASON_7 := 580,
	PRODUCTIONCOUNTERS_CAVITY_12_REJECTREASON_8 := 581,
	PRODUCTIONCOUNTERS_CAVITY_12_REJECTREASON_9 := 582,
	PRODUCTIONCOUNTERS_CAVITY_12_REJECTREASON_10 := 583,
	PRODUCTIONCOUNTERS_CAVITY_12_REJECTREASON_11 := 584,
	PRODUCTIONCOUNTERS_CAVITY_12_REJECTREASON_12 := 585,
	PRODUCTIONCOUNTERS_CAVITY_12_REJECTREASON_13 := 586,
	PRODUCTIONCOUNTERS_CAVITY_12_REJECTREASON_14 := 587,
	PRODUCTIONCOUNTERS_CAVITY_12_REJECTREASON_15 := 588,
	PRODUCTIONCOUNTERS_CAVITY_12_REJECTREASON_16 := 589,
	PRODUCTIONCOUNTERS_CAVITY_12_REJECTREASON_17 := 590,
	PRODUCTIONCOUNTERS_CAVITY_12_REJECTREASON_18 := 591,
	PRODUCTIONCOUNTERS_CAVITY_12_REJECTREASON_19 := 592,
	PRODUCTIONCOUNTERS_CAVITY_12_REJECTREASON_20 := 593,
	MOULDMEASUREMENT_CAVITY_12_PEAKPRESSURE := 594,
	MOULDMEASUREMENT_HOTRUNNER_CAVITY_12_TARGETVALUE := 595,
	MOULDMEASUREMENT_HOTRUNNER_CAVITY_12_ACTUALVALUE := 596,
	PRODUCTIONCOUNTERS_CAVITY_13_PRODUCED := 597,
	PRODUCTIONCOUNTERS_CAVITY_13_STACKED := 598,
	PRODUCTIONCOUNTERS_CAVITY_13_REJECTED := 599,
	PRODUCTIONCOUNTERS_CAVITY_13_UNCOUNTEDREJECT := 600,
	PRODUCTIONCOUNTERS_CAVITY_13_REJECTREASON_0 := 601,
	PRODUCTIONCOUNTERS_CAVITY_13_REJECTREASON_1 := 602,
	PRODUCTIONCOUNTERS_CAVITY_13_REJECTREASON_2 := 603,
	PRODUCTIONCOUNTERS_CAVITY_13_REJECTREASON_3 := 604,
	PRODUCTIONCOUNTERS_CAVITY_13_REJECTREASON_4 := 605,
	PRODUCTIONCOUNTERS_CAVITY_13_REJECTREASON_5 := 606,
	PRODUCTIONCOUNTERS_CAVITY_13_REJECTREASON_6 := 607,
	PRODUCTIONCOUNTERS_CAVITY_13_REJECTREASON_7 := 608,
	PRODUCTIONCOUNTERS_CAVITY_13_REJECTREASON_8 := 609,
	PRODUCTIONCOUNTERS_CAVITY_13_REJECTREASON_9 := 610,
	PRODUCTIONCOUNTERS_CAVITY_13_REJECTREASON_10 := 611,
	PRODUCTIONCOUNTERS_CAVITY_13_REJECTREASON_11 := 612,
	PRODUCTIONCOUNTERS_CAVITY_13_REJECTREASON_12 := 613,
	PRODUCTIONCOUNTERS_CAVITY_13_REJECTREASON_13 := 614,
	PRODUCTIONCOUNTERS_CAVITY_13_REJECTREASON_14 := 615,
	PRODUCTIONCOUNTERS_CAVITY_13_REJECTREASON_15 := 616,
	PRODUCTIONCOUNTERS_CAVITY_13_REJECTREASON_16 := 617,
	PRODUCTIONCOUNTERS_CAVITY_13_REJECTREASON_17 := 618,
	PRODUCTIONCOUNTERS_CAVITY_13_REJECTREASON_18 := 619,
	PRODUCTIONCOUNTERS_CAVITY_13_REJECTREASON_19 := 620,
	PRODUCTIONCOUNTERS_CAVITY_13_REJECTREASON_20 := 621,
	MOULDMEASUREMENT_CAVITY_13_PEAKPRESSURE := 622,
	MOULDMEASUREMENT_HOTRUNNER_CAVITY_13_TARGETVALUE := 623,
	MOULDMEASUREMENT_HOTRUNNER_CAVITY_13_ACTUALVALUE := 624,
	PRODUCTIONCOUNTERS_CAVITY_14_PRODUCED := 625,
	PRODUCTIONCOUNTERS_CAVITY_14_STACKED := 626,
	PRODUCTIONCOUNTERS_CAVITY_14_REJECTED := 627,
	PRODUCTIONCOUNTERS_CAVITY_14_UNCOUNTEDREJECT := 628,
	PRODUCTIONCOUNTERS_CAVITY_14_REJECTREASON_0 := 629,
	PRODUCTIONCOUNTERS_CAVITY_14_REJECTREASON_1 := 630,
	PRODUCTIONCOUNTERS_CAVITY_14_REJECTREASON_2 := 631,
	PRODUCTIONCOUNTERS_CAVITY_14_REJECTREASON_3 := 632,
	PRODUCTIONCOUNTERS_CAVITY_14_REJECTREASON_4 := 633,
	PRODUCTIONCOUNTERS_CAVITY_14_REJECTREASON_5 := 634,
	PRODUCTIONCOUNTERS_CAVITY_14_REJECTREASON_6 := 635,
	PRODUCTIONCOUNTERS_CAVITY_14_REJECTREASON_7 := 636,
	PRODUCTIONCOUNTERS_CAVITY_14_REJECTREASON_8 := 637,
	PRODUCTIONCOUNTERS_CAVITY_14_REJECTREASON_9 := 638,
	PRODUCTIONCOUNTERS_CAVITY_14_REJECTREASON_10 := 639,
	PRODUCTIONCOUNTERS_CAVITY_14_REJECTREASON_11 := 640,
	PRODUCTIONCOUNTERS_CAVITY_14_REJECTREASON_12 := 641,
	PRODUCTIONCOUNTERS_CAVITY_14_REJECTREASON_13 := 642,
	PRODUCTIONCOUNTERS_CAVITY_14_REJECTREASON_14 := 643,
	PRODUCTIONCOUNTERS_CAVITY_14_REJECTREASON_15 := 644,
	PRODUCTIONCOUNTERS_CAVITY_14_REJECTREASON_16 := 645,
	PRODUCTIONCOUNTERS_CAVITY_14_REJECTREASON_17 := 646,
	PRODUCTIONCOUNTERS_CAVITY_14_REJECTREASON_18 := 647,
	PRODUCTIONCOUNTERS_CAVITY_14_REJECTREASON_19 := 648,
	PRODUCTIONCOUNTERS_CAVITY_14_REJECTREASON_20 := 649,
	MOULDMEASUREMENT_CAVITY_14_PEAKPRESSURE := 650,
	MOULDMEASUREMENT_HOTRUNNER_CAVITY_14_TARGETVALUE := 651,
	MOULDMEASUREMENT_HOTRUNNER_CAVITY_14_ACTUALVALUE := 652,
	PRODUCTIONCOUNTERS_CAVITY_15_PRODUCED := 653,
	PRODUCTIONCOUNTERS_CAVITY_15_STACKED := 654,
	PRODUCTIONCOUNTERS_CAVITY_15_REJECTED := 655,
	PRODUCTIONCOUNTERS_CAVITY_15_UNCOUNTEDREJECT := 656,
	PRODUCTIONCOUNTERS_CAVITY_15_REJECTREASON_0 := 657,
	PRODUCTIONCOUNTERS_CAVITY_15_REJECTREASON_1 := 658,
	PRODUCTIONCOUNTERS_CAVITY_15_REJECTREASON_2 := 659,
	PRODUCTIONCOUNTERS_CAVITY_15_REJECTREASON_3 := 660,
	PRODUCTIONCOUNTERS_CAVITY_15_REJECTREASON_4 := 661,
	PRODUCTIONCOUNTERS_CAVITY_15_REJECTREASON_5 := 662,
	PRODUCTIONCOUNTERS_CAVITY_15_REJECTREASON_6 := 663,
	PRODUCTIONCOUNTERS_CAVITY_15_REJECTREASON_7 := 664,
	PRODUCTIONCOUNTERS_CAVITY_15_REJECTREASON_8 := 665,
	PRODUCTIONCOUNTERS_CAVITY_15_REJECTREASON_9 := 666,
	PRODUCTIONCOUNTERS_CAVITY_15_REJECTREASON_10 := 667,
	PRODUCTIONCOUNTERS_CAVITY_15_REJECTREASON_11 := 668,
	PRODUCTIONCOUNTERS_CAVITY_15_REJECTREASON_12 := 669,
	PRODUCTIONCOUNTERS_CAVITY_15_REJECTREASON_13 := 670,
	PRODUCTIONCOUNTERS_CAVITY_15_REJECTREASON_14 := 671,
	PRODUCTIONCOUNTERS_CAVITY_15_REJECTREASON_15 := 672,
	PRODUCTIONCOUNTERS_CAVITY_15_REJECTREASON_16 := 673,
	PRODUCTIONCOUNTERS_CAVITY_15_REJECTREASON_17 := 674,
	PRODUCTIONCOUNTERS_CAVITY_15_REJECTREASON_18 := 675,
	PRODUCTIONCOUNTERS_CAVITY_15_REJECTREASON_19 := 676,
	PRODUCTIONCOUNTERS_CAVITY_15_REJECTREASON_20 := 677,
	MOULDMEASUREMENT_CAVITY_15_PEAKPRESSURE := 678,
	MOULDMEASUREMENT_HOTRUNNER_CAVITY_15_TARGETVALUE := 679,
	MOULDMEASUREMENT_HOTRUNNER_CAVITY_15_ACTUALVALUE := 680,
	PRODUCTIONCOUNTERS_CAVITY_16_PRODUCED := 681,
	PRODUCTIONCOUNTERS_CAVITY_16_STACKED := 682,
	PRODUCTIONCOUNTERS_CAVITY_16_REJECTED := 683,
	PRODUCTIONCOUNTERS_CAVITY_16_UNCOUNTEDREJECT := 684,
	PRODUCTIONCOUNTERS_CAVITY_16_REJECTREASON_0 := 685,
	PRODUCTIONCOUNTERS_CAVITY_16_REJECTREASON_1 := 686,
	PRODUCTIONCOUNTERS_CAVITY_16_REJECTREASON_2 := 687,
	PRODUCTIONCOUNTERS_CAVITY_16_REJECTREASON_3 := 688,
	PRODUCTIONCOUNTERS_CAVITY_16_REJECTREASON_4 := 689,
	PRODUCTIONCOUNTERS_CAVITY_16_REJECTREASON_5 := 690,
	PRODUCTIONCOUNTERS_CAVITY_16_REJECTREASON_6 := 691,
	PRODUCTIONCOUNTERS_CAVITY_16_REJECTREASON_7 := 692,
	PRODUCTIONCOUNTERS_CAVITY_16_REJECTREASON_8 := 693,
	PRODUCTIONCOUNTERS_CAVITY_16_REJECTREASON_9 := 694,
	PRODUCTIONCOUNTERS_CAVITY_16_REJECTREASON_10 := 695,
	PRODUCTIONCOUNTERS_CAVITY_16_REJECTREASON_11 := 696,
	PRODUCTIONCOUNTERS_CAVITY_16_REJECTREASON_12 := 697,
	PRODUCTIONCOUNTERS_CAVITY_16_REJECTREASON_13 := 698,
	PRODUCTIONCOUNTERS_CAVITY_16_REJECTREASON_14 := 699,
	PRODUCTIONCOUNTERS_CAVITY_16_REJECTREASON_15 := 700,
	PRODUCTIONCOUNTERS_CAVITY_16_REJECTREASON_16 := 701,
	PRODUCTIONCOUNTERS_CAVITY_16_REJECTREASON_17 := 702,
	PRODUCTIONCOUNTERS_CAVITY_16_REJECTREASON_18 := 703,
	PRODUCTIONCOUNTERS_CAVITY_16_REJECTREASON_19 := 704,
	PRODUCTIONCOUNTERS_CAVITY_16_REJECTREASON_20 := 705,
	MOULDMEASUREMENT_CAVITY_16_PEAKPRESSURE := 706,
	MOULDMEASUREMENT_HOTRUNNER_CAVITY_16_TARGETVALUE := 707,
	MOULDMEASUREMENT_HOTRUNNER_CAVITY_16_ACTUALVALUE := 708,
	PRODUCTIONCOUNTERS_CAVITY_17_PRODUCED := 709,
	PRODUCTIONCOUNTERS_CAVITY_17_STACKED := 710,
	PRODUCTIONCOUNTERS_CAVITY_17_REJECTED := 711,
	PRODUCTIONCOUNTERS_CAVITY_17_UNCOUNTEDREJECT := 712,
	PRODUCTIONCOUNTERS_CAVITY_17_REJECTREASON_0 := 713,
	PRODUCTIONCOUNTERS_CAVITY_17_REJECTREASON_1 := 714,
	PRODUCTIONCOUNTERS_CAVITY_17_REJECTREASON_2 := 715,
	PRODUCTIONCOUNTERS_CAVITY_17_REJECTREASON_3 := 716,
	PRODUCTIONCOUNTERS_CAVITY_17_REJECTREASON_4 := 717,
	PRODUCTIONCOUNTERS_CAVITY_17_REJECTREASON_5 := 718,
	PRODUCTIONCOUNTERS_CAVITY_17_REJECTREASON_6 := 719,
	PRODUCTIONCOUNTERS_CAVITY_17_REJECTREASON_7 := 720,
	PRODUCTIONCOUNTERS_CAVITY_17_REJECTREASON_8 := 721,
	PRODUCTIONCOUNTERS_CAVITY_17_REJECTREASON_9 := 722,
	PRODUCTIONCOUNTERS_CAVITY_17_REJECTREASON_10 := 723,
	PRODUCTIONCOUNTERS_CAVITY_17_REJECTREASON_11 := 724,
	PRODUCTIONCOUNTERS_CAVITY_17_REJECTREASON_12 := 725,
	PRODUCTIONCOUNTERS_CAVITY_17_REJECTREASON_13 := 726,
	PRODUCTIONCOUNTERS_CAVITY_17_REJECTREASON_14 := 727,
	PRODUCTIONCOUNTERS_CAVITY_17_REJECTREASON_15 := 728,
	PRODUCTIONCOUNTERS_CAVITY_17_REJECTREASON_16 := 729,
	PRODUCTIONCOUNTERS_CAVITY_17_REJECTREASON_17 := 730,
	PRODUCTIONCOUNTERS_CAVITY_17_REJECTREASON_18 := 731,
	PRODUCTIONCOUNTERS_CAVITY_17_REJECTREASON_19 := 732,
	PRODUCTIONCOUNTERS_CAVITY_17_REJECTREASON_20 := 733,
	MOULDMEASUREMENT_CAVITY_17_PEAKPRESSURE := 734,
	MOULDMEASUREMENT_HOTRUNNER_CAVITY_17_TARGETVALUE := 735,
	MOULDMEASUREMENT_HOTRUNNER_CAVITY_17_ACTUALVALUE := 736,
	PRODUCTIONCOUNTERS_CAVITY_18_PRODUCED := 737,
	PRODUCTIONCOUNTERS_CAVITY_18_STACKED := 738,
	PRODUCTIONCOUNTERS_CAVITY_18_REJECTED := 739,
	PRODUCTIONCOUNTERS_CAVITY_18_UNCOUNTEDREJECT := 740,
	PRODUCTIONCOUNTERS_CAVITY_18_REJECTREASON_0 := 741,
	PRODUCTIONCOUNTERS_CAVITY_18_REJECTREASON_1 := 742,
	PRODUCTIONCOUNTERS_CAVITY_18_REJECTREASON_2 := 743,
	PRODUCTIONCOUNTERS_CAVITY_18_REJECTREASON_3 := 744,
	PRODUCTIONCOUNTERS_CAVITY_18_REJECTREASON_4 := 745,
	PRODUCTIONCOUNTERS_CAVITY_18_REJECTREASON_5 := 746,
	PRODUCTIONCOUNTERS_CAVITY_18_REJECTREASON_6 := 747,
	PRODUCTIONCOUNTERS_CAVITY_18_REJECTREASON_7 := 748,
	PRODUCTIONCOUNTERS_CAVITY_18_REJECTREASON_8 := 749,
	PRODUCTIONCOUNTERS_CAVITY_18_REJECTREASON_9 := 750,
	PRODUCTIONCOUNTERS_CAVITY_18_REJECTREASON_10 := 751,
	PRODUCTIONCOUNTERS_CAVITY_18_REJECTREASON_11 := 752,
	PRODUCTIONCOUNTERS_CAVITY_18_REJECTREASON_12 := 753,
	PRODUCTIONCOUNTERS_CAVITY_18_REJECTREASON_13 := 754,
	PRODUCTIONCOUNTERS_CAVITY_18_REJECTREASON_14 := 755,
	PRODUCTIONCOUNTERS_CAVITY_18_REJECTREASON_15 := 756,
	PRODUCTIONCOUNTERS_CAVITY_18_REJECTREASON_16 := 757,
	PRODUCTIONCOUNTERS_CAVITY_18_REJECTREASON_17 := 758,
	PRODUCTIONCOUNTERS_CAVITY_18_REJECTREASON_18 := 759,
	PRODUCTIONCOUNTERS_CAVITY_18_REJECTREASON_19 := 760,
	PRODUCTIONCOUNTERS_CAVITY_18_REJECTREASON_20 := 761,
	MOULDMEASUREMENT_CAVITY_18_PEAKPRESSURE := 762,
	MOULDMEASUREMENT_HOTRUNNER_CAVITY_18_TARGETVALUE := 763,
	MOULDMEASUREMENT_HOTRUNNER_CAVITY_18_ACTUALVALUE := 764,
	PRODUCTIONCOUNTERS_CAVITY_19_PRODUCED := 765,
	PRODUCTIONCOUNTERS_CAVITY_19_STACKED := 766,
	PRODUCTIONCOUNTERS_CAVITY_19_REJECTED := 767,
	PRODUCTIONCOUNTERS_CAVITY_19_UNCOUNTEDREJECT := 768,
	PRODUCTIONCOUNTERS_CAVITY_19_REJECTREASON_0 := 769,
	PRODUCTIONCOUNTERS_CAVITY_19_REJECTREASON_1 := 770,
	PRODUCTIONCOUNTERS_CAVITY_19_REJECTREASON_2 := 771,
	PRODUCTIONCOUNTERS_CAVITY_19_REJECTREASON_3 := 772,
	PRODUCTIONCOUNTERS_CAVITY_19_REJECTREASON_4 := 773,
	PRODUCTIONCOUNTERS_CAVITY_19_REJECTREASON_5 := 774,
	PRODUCTIONCOUNTERS_CAVITY_19_REJECTREASON_6 := 775,
	PRODUCTIONCOUNTERS_CAVITY_19_REJECTREASON_7 := 776,
	PRODUCTIONCOUNTERS_CAVITY_19_REJECTREASON_8 := 777,
	PRODUCTIONCOUNTERS_CAVITY_19_REJECTREASON_9 := 778,
	PRODUCTIONCOUNTERS_CAVITY_19_REJECTREASON_10 := 779,
	PRODUCTIONCOUNTERS_CAVITY_19_REJECTREASON_11 := 780,
	PRODUCTIONCOUNTERS_CAVITY_19_REJECTREASON_12 := 781,
	PRODUCTIONCOUNTERS_CAVITY_19_REJECTREASON_13 := 782,
	PRODUCTIONCOUNTERS_CAVITY_19_REJECTREASON_14 := 783,
	PRODUCTIONCOUNTERS_CAVITY_19_REJECTREASON_15 := 784,
	PRODUCTIONCOUNTERS_CAVITY_19_REJECTREASON_16 := 785,
	PRODUCTIONCOUNTERS_CAVITY_19_REJECTREASON_17 := 786,
	PRODUCTIONCOUNTERS_CAVITY_19_REJECTREASON_18 := 787,
	PRODUCTIONCOUNTERS_CAVITY_19_REJECTREASON_19 := 788,
	PRODUCTIONCOUNTERS_CAVITY_19_REJECTREASON_20 := 789,
	MOULDMEASUREMENT_CAVITY_19_PEAKPRESSURE := 790,
	MOULDMEASUREMENT_HOTRUNNER_CAVITY_19_TARGETVALUE := 791,
	MOULDMEASUREMENT_HOTRUNNER_CAVITY_19_ACTUALVALUE := 792,
	PRODUCTIONCOUNTERS_CAVITY_20_PRODUCED := 793,
	PRODUCTIONCOUNTERS_CAVITY_20_STACKED := 794,
	PRODUCTIONCOUNTERS_CAVITY_20_REJECTED := 795,
	PRODUCTIONCOUNTERS_CAVITY_20_UNCOUNTEDREJECT := 796,
	PRODUCTIONCOUNTERS_CAVITY_20_REJECTREASON_0 := 797,
	PRODUCTIONCOUNTERS_CAVITY_20_REJECTREASON_1 := 798,
	PRODUCTIONCOUNTERS_CAVITY_20_REJECTREASON_2 := 799,
	PRODUCTIONCOUNTERS_CAVITY_20_REJECTREASON_3 := 800,
	PRODUCTIONCOUNTERS_CAVITY_20_REJECTREASON_4 := 801,
	PRODUCTIONCOUNTERS_CAVITY_20_REJECTREASON_5 := 802,
	PRODUCTIONCOUNTERS_CAVITY_20_REJECTREASON_6 := 803,
	PRODUCTIONCOUNTERS_CAVITY_20_REJECTREASON_7 := 804,
	PRODUCTIONCOUNTERS_CAVITY_20_REJECTREASON_8 := 805,
	PRODUCTIONCOUNTERS_CAVITY_20_REJECTREASON_9 := 806,
	PRODUCTIONCOUNTERS_CAVITY_20_REJECTREASON_10 := 807,
	PRODUCTIONCOUNTERS_CAVITY_20_REJECTREASON_11 := 808,
	PRODUCTIONCOUNTERS_CAVITY_20_REJECTREASON_12 := 809,
	PRODUCTIONCOUNTERS_CAVITY_20_REJECTREASON_13 := 810,
	PRODUCTIONCOUNTERS_CAVITY_20_REJECTREASON_14 := 811,
	PRODUCTIONCOUNTERS_CAVITY_20_REJECTREASON_15 := 812,
	PRODUCTIONCOUNTERS_CAVITY_20_REJECTREASON_16 := 813,
	PRODUCTIONCOUNTERS_CAVITY_20_REJECTREASON_17 := 814,
	PRODUCTIONCOUNTERS_CAVITY_20_REJECTREASON_18 := 815,
	PRODUCTIONCOUNTERS_CAVITY_20_REJECTREASON_19 := 816,
	PRODUCTIONCOUNTERS_CAVITY_20_REJECTREASON_20 := 817,
	MOULDMEASUREMENT_CAVITY_20_PEAKPRESSURE := 818,
	MOULDMEASUREMENT_HOTRUNNER_CAVITY_20_TARGETVALUE := 819,
	MOULDMEASUREMENT_HOTRUNNER_CAVITY_20_ACTUALVALUE := 820,
	PRODUCTIONCOUNTERS_CAVITY_21_PRODUCED := 821,
	PRODUCTIONCOUNTERS_CAVITY_21_STACKED := 822,
	PRODUCTIONCOUNTERS_CAVITY_21_REJECTED := 823,
	PRODUCTIONCOUNTERS_CAVITY_21_UNCOUNTEDREJECT := 824,
	PRODUCTIONCOUNTERS_CAVITY_21_REJECTREASON_0 := 825,
	PRODUCTIONCOUNTERS_CAVITY_21_REJECTREASON_1 := 826,
	PRODUCTIONCOUNTERS_CAVITY_21_REJECTREASON_2 := 827,
	PRODUCTIONCOUNTERS_CAVITY_21_REJECTREASON_3 := 828,
	PRODUCTIONCOUNTERS_CAVITY_21_REJECTREASON_4 := 829,
	PRODUCTIONCOUNTERS_CAVITY_21_REJECTREASON_5 := 830,
	PRODUCTIONCOUNTERS_CAVITY_21_REJECTREASON_6 := 831,
	PRODUCTIONCOUNTERS_CAVITY_21_REJECTREASON_7 := 832,
	PRODUCTIONCOUNTERS_CAVITY_21_REJECTREASON_8 := 833,
	PRODUCTIONCOUNTERS_CAVITY_21_REJECTREASON_9 := 834,
	PRODUCTIONCOUNTERS_CAVITY_21_REJECTREASON_10 := 835,
	PRODUCTIONCOUNTERS_CAVITY_21_REJECTREASON_11 := 836,
	PRODUCTIONCOUNTERS_CAVITY_21_REJECTREASON_12 := 837,
	PRODUCTIONCOUNTERS_CAVITY_21_REJECTREASON_13 := 838,
	PRODUCTIONCOUNTERS_CAVITY_21_REJECTREASON_14 := 839,
	PRODUCTIONCOUNTERS_CAVITY_21_REJECTREASON_15 := 840,
	PRODUCTIONCOUNTERS_CAVITY_21_REJECTREASON_16 := 841,
	PRODUCTIONCOUNTERS_CAVITY_21_REJECTREASON_17 := 842,
	PRODUCTIONCOUNTERS_CAVITY_21_REJECTREASON_18 := 843,
	PRODUCTIONCOUNTERS_CAVITY_21_REJECTREASON_19 := 844,
	PRODUCTIONCOUNTERS_CAVITY_21_REJECTREASON_20 := 845,
	MOULDMEASUREMENT_CAVITY_21_PEAKPRESSURE := 846,
	MOULDMEASUREMENT_HOTRUNNER_CAVITY_21_TARGETVALUE := 847,
	MOULDMEASUREMENT_HOTRUNNER_CAVITY_21_ACTUALVALUE := 848,
	PRODUCTIONCOUNTERS_CAVITY_22_PRODUCED := 849,
	PRODUCTIONCOUNTERS_CAVITY_22_STACKED := 850,
	PRODUCTIONCOUNTERS_CAVITY_22_REJECTED := 851,
	PRODUCTIONCOUNTERS_CAVITY_22_UNCOUNTEDREJECT := 852,
	PRODUCTIONCOUNTERS_CAVITY_22_REJECTREASON_0 := 853,
	PRODUCTIONCOUNTERS_CAVITY_22_REJECTREASON_1 := 854,
	PRODUCTIONCOUNTERS_CAVITY_22_REJECTREASON_2 := 855,
	PRODUCTIONCOUNTERS_CAVITY_22_REJECTREASON_3 := 856,
	PRODUCTIONCOUNTERS_CAVITY_22_REJECTREASON_4 := 857,
	PRODUCTIONCOUNTERS_CAVITY_22_REJECTREASON_5 := 858,
	PRODUCTIONCOUNTERS_CAVITY_22_REJECTREASON_6 := 859,
	PRODUCTIONCOUNTERS_CAVITY_22_REJECTREASON_7 := 860,
	PRODUCTIONCOUNTERS_CAVITY_22_REJECTREASON_8 := 861,
	PRODUCTIONCOUNTERS_CAVITY_22_REJECTREASON_9 := 862,
	PRODUCTIONCOUNTERS_CAVITY_22_REJECTREASON_10 := 863,
	PRODUCTIONCOUNTERS_CAVITY_22_REJECTREASON_11 := 864,
	PRODUCTIONCOUNTERS_CAVITY_22_REJECTREASON_12 := 865,
	PRODUCTIONCOUNTERS_CAVITY_22_REJECTREASON_13 := 866,
	PRODUCTIONCOUNTERS_CAVITY_22_REJECTREASON_14 := 867,
	PRODUCTIONCOUNTERS_CAVITY_22_REJECTREASON_15 := 868,
	PRODUCTIONCOUNTERS_CAVITY_22_REJECTREASON_16 := 869,
	PRODUCTIONCOUNTERS_CAVITY_22_REJECTREASON_17 := 870,
	PRODUCTIONCOUNTERS_CAVITY_22_REJECTREASON_18 := 871,
	PRODUCTIONCOUNTERS_CAVITY_22_REJECTREASON_19 := 872,
	PRODUCTIONCOUNTERS_CAVITY_22_REJECTREASON_20 := 873,
	MOULDMEASUREMENT_CAVITY_22_PEAKPRESSURE := 874,
	MOULDMEASUREMENT_HOTRUNNER_CAVITY_22_TARGETVALUE := 875,
	MOULDMEASUREMENT_HOTRUNNER_CAVITY_22_ACTUALVALUE := 876,
	PRODUCTIONCOUNTERS_CAVITY_23_PRODUCED := 877,
	PRODUCTIONCOUNTERS_CAVITY_23_STACKED := 878,
	PRODUCTIONCOUNTERS_CAVITY_23_REJECTED := 879,
	PRODUCTIONCOUNTERS_CAVITY_23_UNCOUNTEDREJECT := 880,
	PRODUCTIONCOUNTERS_CAVITY_23_REJECTREASON_0 := 881,
	PRODUCTIONCOUNTERS_CAVITY_23_REJECTREASON_1 := 882,
	PRODUCTIONCOUNTERS_CAVITY_23_REJECTREASON_2 := 883,
	PRODUCTIONCOUNTERS_CAVITY_23_REJECTREASON_3 := 884,
	PRODUCTIONCOUNTERS_CAVITY_23_REJECTREASON_4 := 885,
	PRODUCTIONCOUNTERS_CAVITY_23_REJECTREASON_5 := 886,
	PRODUCTIONCOUNTERS_CAVITY_23_REJECTREASON_6 := 887,
	PRODUCTIONCOUNTERS_CAVITY_23_REJECTREASON_7 := 888,
	PRODUCTIONCOUNTERS_CAVITY_23_REJECTREASON_8 := 889,
	PRODUCTIONCOUNTERS_CAVITY_23_REJECTREASON_9 := 890,
	PRODUCTIONCOUNTERS_CAVITY_23_REJECTREASON_10 := 891,
	PRODUCTIONCOUNTERS_CAVITY_23_REJECTREASON_11 := 892,
	PRODUCTIONCOUNTERS_CAVITY_23_REJECTREASON_12 := 893,
	PRODUCTIONCOUNTERS_CAVITY_23_REJECTREASON_13 := 894,
	PRODUCTIONCOUNTERS_CAVITY_23_REJECTREASON_14 := 895,
	PRODUCTIONCOUNTERS_CAVITY_23_REJECTREASON_15 := 896,
	PRODUCTIONCOUNTERS_CAVITY_23_REJECTREASON_16 := 897,
	PRODUCTIONCOUNTERS_CAVITY_23_REJECTREASON_17 := 898,
	PRODUCTIONCOUNTERS_CAVITY_23_REJECTREASON_18 := 899,
	PRODUCTIONCOUNTERS_CAVITY_23_REJECTREASON_19 := 900,
	PRODUCTIONCOUNTERS_CAVITY_23_REJECTREASON_20 := 901,
	MOULDMEASUREMENT_CAVITY_23_PEAKPRESSURE := 902,
	MOULDMEASUREMENT_HOTRUNNER_CAVITY_23_TARGETVALUE := 903,
	MOULDMEASUREMENT_HOTRUNNER_CAVITY_23_ACTUALVALUE := 904,
	PRODUCTIONCOUNTERS_CAVITY_24_PRODUCED := 905,
	PRODUCTIONCOUNTERS_CAVITY_24_STACKED := 906,
	PRODUCTIONCOUNTERS_CAVITY_24_REJECTED := 907,
	PRODUCTIONCOUNTERS_CAVITY_24_UNCOUNTEDREJECT := 908,
	PRODUCTIONCOUNTERS_CAVITY_24_REJECTREASON_0 := 909,
	PRODUCTIONCOUNTERS_CAVITY_24_REJECTREASON_1 := 910,
	PRODUCTIONCOUNTERS_CAVITY_24_REJECTREASON_2 := 911,
	PRODUCTIONCOUNTERS_CAVITY_24_REJECTREASON_3 := 912,
	PRODUCTIONCOUNTERS_CAVITY_24_REJECTREASON_4 := 913,
	PRODUCTIONCOUNTERS_CAVITY_24_REJECTREASON_5 := 914,
	PRODUCTIONCOUNTERS_CAVITY_24_REJECTREASON_6 := 915,
	PRODUCTIONCOUNTERS_CAVITY_24_REJECTREASON_7 := 916,
	PRODUCTIONCOUNTERS_CAVITY_24_REJECTREASON_8 := 917,
	PRODUCTIONCOUNTERS_CAVITY_24_REJECTREASON_9 := 918,
	PRODUCTIONCOUNTERS_CAVITY_24_REJECTREASON_10 := 919,
	PRODUCTIONCOUNTERS_CAVITY_24_REJECTREASON_11 := 920,
	PRODUCTIONCOUNTERS_CAVITY_24_REJECTREASON_12 := 921,
	PRODUCTIONCOUNTERS_CAVITY_24_REJECTREASON_13 := 922,
	PRODUCTIONCOUNTERS_CAVITY_24_REJECTREASON_14 := 923,
	PRODUCTIONCOUNTERS_CAVITY_24_REJECTREASON_15 := 924,
	PRODUCTIONCOUNTERS_CAVITY_24_REJECTREASON_16 := 925,
	PRODUCTIONCOUNTERS_CAVITY_24_REJECTREASON_17 := 926,
	PRODUCTIONCOUNTERS_CAVITY_24_REJECTREASON_18 := 927,
	PRODUCTIONCOUNTERS_CAVITY_24_REJECTREASON_19 := 928,
	PRODUCTIONCOUNTERS_CAVITY_24_REJECTREASON_20 := 929,
	MOULDMEASUREMENT_CAVITY_24_PEAKPRESSURE := 930,
	MOULDMEASUREMENT_HOTRUNNER_CAVITY_24_TARGETVALUE := 931,
	MOULDMEASUREMENT_HOTRUNNER_CAVITY_24_ACTUALVALUE := 932,
	PRODUCTIONCOUNTERS_CAVITY_25_PRODUCED := 933,
	PRODUCTIONCOUNTERS_CAVITY_25_STACKED := 934,
	PRODUCTIONCOUNTERS_CAVITY_25_REJECTED := 935,
	PRODUCTIONCOUNTERS_CAVITY_25_UNCOUNTEDREJECT := 936,
	PRODUCTIONCOUNTERS_CAVITY_25_REJECTREASON_0 := 937,
	PRODUCTIONCOUNTERS_CAVITY_25_REJECTREASON_1 := 938,
	PRODUCTIONCOUNTERS_CAVITY_25_REJECTREASON_2 := 939,
	PRODUCTIONCOUNTERS_CAVITY_25_REJECTREASON_3 := 940,
	PRODUCTIONCOUNTERS_CAVITY_25_REJECTREASON_4 := 941,
	PRODUCTIONCOUNTERS_CAVITY_25_REJECTREASON_5 := 942,
	PRODUCTIONCOUNTERS_CAVITY_25_REJECTREASON_6 := 943,
	PRODUCTIONCOUNTERS_CAVITY_25_REJECTREASON_7 := 944,
	PRODUCTIONCOUNTERS_CAVITY_25_REJECTREASON_8 := 945,
	PRODUCTIONCOUNTERS_CAVITY_25_REJECTREASON_9 := 946,
	PRODUCTIONCOUNTERS_CAVITY_25_REJECTREASON_10 := 947,
	PRODUCTIONCOUNTERS_CAVITY_25_REJECTREASON_11 := 948,
	PRODUCTIONCOUNTERS_CAVITY_25_REJECTREASON_12 := 949,
	PRODUCTIONCOUNTERS_CAVITY_25_REJECTREASON_13 := 950,
	PRODUCTIONCOUNTERS_CAVITY_25_REJECTREASON_14 := 951,
	PRODUCTIONCOUNTERS_CAVITY_25_REJECTREASON_15 := 952,
	PRODUCTIONCOUNTERS_CAVITY_25_REJECTREASON_16 := 953,
	PRODUCTIONCOUNTERS_CAVITY_25_REJECTREASON_17 := 954,
	PRODUCTIONCOUNTERS_CAVITY_25_REJECTREASON_18 := 955,
	PRODUCTIONCOUNTERS_CAVITY_25_REJECTREASON_19 := 956,
	PRODUCTIONCOUNTERS_CAVITY_25_REJECTREASON_20 := 957,
	MOULDMEASUREMENT_CAVITY_25_PEAKPRESSURE := 958,
	MOULDMEASUREMENT_HOTRUNNER_CAVITY_25_TARGETVALUE := 959,
	MOULDMEASUREMENT_HOTRUNNER_CAVITY_25_ACTUALVALUE := 960,
	PRODUCTIONCOUNTERS_CAVITY_26_PRODUCED := 961,
	PRODUCTIONCOUNTERS_CAVITY_26_STACKED := 962,
	PRODUCTIONCOUNTERS_CAVITY_26_REJECTED := 963,
	PRODUCTIONCOUNTERS_CAVITY_26_UNCOUNTEDREJECT := 964,
	PRODUCTIONCOUNTERS_CAVITY_26_REJECTREASON_0 := 965,
	PRODUCTIONCOUNTERS_CAVITY_26_REJECTREASON_1 := 966,
	PRODUCTIONCOUNTERS_CAVITY_26_REJECTREASON_2 := 967,
	PRODUCTIONCOUNTERS_CAVITY_26_REJECTREASON_3 := 968,
	PRODUCTIONCOUNTERS_CAVITY_26_REJECTREASON_4 := 969,
	PRODUCTIONCOUNTERS_CAVITY_26_REJECTREASON_5 := 970,
	PRODUCTIONCOUNTERS_CAVITY_26_REJECTREASON_6 := 971,
	PRODUCTIONCOUNTERS_CAVITY_26_REJECTREASON_7 := 972,
	PRODUCTIONCOUNTERS_CAVITY_26_REJECTREASON_8 := 973,
	PRODUCTIONCOUNTERS_CAVITY_26_REJECTREASON_9 := 974,
	PRODUCTIONCOUNTERS_CAVITY_26_REJECTREASON_10 := 975,
	PRODUCTIONCOUNTERS_CAVITY_26_REJECTREASON_11 := 976,
	PRODUCTIONCOUNTERS_CAVITY_26_REJECTREASON_12 := 977,
	PRODUCTIONCOUNTERS_CAVITY_26_REJECTREASON_13 := 978,
	PRODUCTIONCOUNTERS_CAVITY_26_REJECTREASON_14 := 979,
	PRODUCTIONCOUNTERS_CAVITY_26_REJECTREASON_15 := 980,
	PRODUCTIONCOUNTERS_CAVITY_26_REJECTREASON_16 := 981,
	PRODUCTIONCOUNTERS_CAVITY_26_REJECTREASON_17 := 982,
	PRODUCTIONCOUNTERS_CAVITY_26_REJECTREASON_18 := 983,
	PRODUCTIONCOUNTERS_CAVITY_26_REJECTREASON_19 := 984,
	PRODUCTIONCOUNTERS_CAVITY_26_REJECTREASON_20 := 985,
	MOULDMEASUREMENT_CAVITY_26_PEAKPRESSURE := 986,
	MOULDMEASUREMENT_HOTRUNNER_CAVITY_26_TARGETVALUE := 987,
	MOULDMEASUREMENT_HOTRUNNER_CAVITY_26_ACTUALVALUE := 988,
	PRODUCTIONCOUNTERS_CAVITY_27_PRODUCED := 989,
	PRODUCTIONCOUNTERS_CAVITY_27_STACKED := 990,
	PRODUCTIONCOUNTERS_CAVITY_27_REJECTED := 991,
	PRODUCTIONCOUNTERS_CAVITY_27_UNCOUNTEDREJECT := 992,
	PRODUCTIONCOUNTERS_CAVITY_27_REJECTREASON_0 := 993,
	PRODUCTIONCOUNTERS_CAVITY_27_REJECTREASON_1 := 994,
	PRODUCTIONCOUNTERS_CAVITY_27_REJECTREASON_2 := 995,
	PRODUCTIONCOUNTERS_CAVITY_27_REJECTREASON_3 := 996,
	PRODUCTIONCOUNTERS_CAVITY_27_REJECTREASON_4 := 997,
	PRODUCTIONCOUNTERS_CAVITY_27_REJECTREASON_5 := 998,
	PRODUCTIONCOUNTERS_CAVITY_27_REJECTREASON_6 := 999,
	PRODUCTIONCOUNTERS_CAVITY_27_REJECTREASON_7 := 1000,
	PRODUCTIONCOUNTERS_CAVITY_27_REJECTREASON_8 := 1001,
	PRODUCTIONCOUNTERS_CAVITY_27_REJECTREASON_9 := 1002,
	PRODUCTIONCOUNTERS_CAVITY_27_REJECTREASON_10 := 1003,
	PRODUCTIONCOUNTERS_CAVITY_27_REJECTREASON_11 := 1004,
	PRODUCTIONCOUNTERS_CAVITY_27_REJECTREASON_12 := 1005,
	PRODUCTIONCOUNTERS_CAVITY_27_REJECTREASON_13 := 1006,
	PRODUCTIONCOUNTERS_CAVITY_27_REJECTREASON_14 := 1007,
	PRODUCTIONCOUNTERS_CAVITY_27_REJECTREASON_15 := 1008,
	PRODUCTIONCOUNTERS_CAVITY_27_REJECTREASON_16 := 1009,
	PRODUCTIONCOUNTERS_CAVITY_27_REJECTREASON_17 := 1010,
	PRODUCTIONCOUNTERS_CAVITY_27_REJECTREASON_18 := 1011,
	PRODUCTIONCOUNTERS_CAVITY_27_REJECTREASON_19 := 1012,
	PRODUCTIONCOUNTERS_CAVITY_27_REJECTREASON_20 := 1013,
	MOULDMEASUREMENT_CAVITY_27_PEAKPRESSURE := 1014,
	MOULDMEASUREMENT_HOTRUNNER_CAVITY_27_TARGETVALUE := 1015,
	MOULDMEASUREMENT_HOTRUNNER_CAVITY_27_ACTUALVALUE := 1016,
	PRODUCTIONCOUNTERS_CAVITY_28_PRODUCED := 1017,
	PRODUCTIONCOUNTERS_CAVITY_28_STACKED := 1018,
	PRODUCTIONCOUNTERS_CAVITY_28_REJECTED := 1019,
	PRODUCTIONCOUNTERS_CAVITY_28_UNCOUNTEDREJECT := 1020,
	PRODUCTIONCOUNTERS_CAVITY_28_REJECTREASON_0 := 1021,
	PRODUCTIONCOUNTERS_CAVITY_28_REJECTREASON_1 := 1022,
	PRODUCTIONCOUNTERS_CAVITY_28_REJECTREASON_2 := 1023,
	PRODUCTIONCOUNTERS_CAVITY_28_REJECTREASON_3 := 1024,
	PRODUCTIONCOUNTERS_CAVITY_28_REJECTREASON_4 := 1025,
	PRODUCTIONCOUNTERS_CAVITY_28_REJECTREASON_5 := 1026,
	PRODUCTIONCOUNTERS_CAVITY_28_REJECTREASON_6 := 1027,
	PRODUCTIONCOUNTERS_CAVITY_28_REJECTREASON_7 := 1028,
	PRODUCTIONCOUNTERS_CAVITY_28_REJECTREASON_8 := 1029,
	PRODUCTIONCOUNTERS_CAVITY_28_REJECTREASON_9 := 1030,
	PRODUCTIONCOUNTERS_CAVITY_28_REJECTREASON_10 := 1031,
	PRODUCTIONCOUNTERS_CAVITY_28_REJECTREASON_11 := 1032,
	PRODUCTIONCOUNTERS_CAVITY_28_REJECTREASON_12 := 1033,
	PRODUCTIONCOUNTERS_CAVITY_28_REJECTREASON_13 := 1034,
	PRODUCTIONCOUNTERS_CAVITY_28_REJECTREASON_14 := 1035,
	PRODUCTIONCOUNTERS_CAVITY_28_REJECTREASON_15 := 1036,
	PRODUCTIONCOUNTERS_CAVITY_28_REJECTREASON_16 := 1037,
	PRODUCTIONCOUNTERS_CAVITY_28_REJECTREASON_17 := 1038,
	PRODUCTIONCOUNTERS_CAVITY_28_REJECTREASON_18 := 1039,
	PRODUCTIONCOUNTERS_CAVITY_28_REJECTREASON_19 := 1040,
	PRODUCTIONCOUNTERS_CAVITY_28_REJECTREASON_20 := 1041,
	MOULDMEASUREMENT_CAVITY_28_PEAKPRESSURE := 1042,
	MOULDMEASUREMENT_HOTRUNNER_CAVITY_28_TARGETVALUE := 1043,
	MOULDMEASUREMENT_HOTRUNNER_CAVITY_28_ACTUALVALUE := 1044,
	PRODUCTIONCOUNTERS_CAVITY_29_PRODUCED := 1045,
	PRODUCTIONCOUNTERS_CAVITY_29_STACKED := 1046,
	PRODUCTIONCOUNTERS_CAVITY_29_REJECTED := 1047,
	PRODUCTIONCOUNTERS_CAVITY_29_UNCOUNTEDREJECT := 1048,
	PRODUCTIONCOUNTERS_CAVITY_29_REJECTREASON_0 := 1049,
	PRODUCTIONCOUNTERS_CAVITY_29_REJECTREASON_1 := 1050,
	PRODUCTIONCOUNTERS_CAVITY_29_REJECTREASON_2 := 1051,
	PRODUCTIONCOUNTERS_CAVITY_29_REJECTREASON_3 := 1052,
	PRODUCTIONCOUNTERS_CAVITY_29_REJECTREASON_4 := 1053,
	PRODUCTIONCOUNTERS_CAVITY_29_REJECTREASON_5 := 1054,
	PRODUCTIONCOUNTERS_CAVITY_29_REJECTREASON_6 := 1055,
	PRODUCTIONCOUNTERS_CAVITY_29_REJECTREASON_7 := 1056,
	PRODUCTIONCOUNTERS_CAVITY_29_REJECTREASON_8 := 1057,
	PRODUCTIONCOUNTERS_CAVITY_29_REJECTREASON_9 := 1058,
	PRODUCTIONCOUNTERS_CAVITY_29_REJECTREASON_10 := 1059,
	PRODUCTIONCOUNTERS_CAVITY_29_REJECTREASON_11 := 1060,
	PRODUCTIONCOUNTERS_CAVITY_29_REJECTREASON_12 := 1061,
	PRODUCTIONCOUNTERS_CAVITY_29_REJECTREASON_13 := 1062,
	PRODUCTIONCOUNTERS_CAVITY_29_REJECTREASON_14 := 1063,
	PRODUCTIONCOUNTERS_CAVITY_29_REJECTREASON_15 := 1064,
	PRODUCTIONCOUNTERS_CAVITY_29_REJECTREASON_16 := 1065,
	PRODUCTIONCOUNTERS_CAVITY_29_REJECTREASON_17 := 1066,
	PRODUCTIONCOUNTERS_CAVITY_29_REJECTREASON_18 := 1067,
	PRODUCTIONCOUNTERS_CAVITY_29_REJECTREASON_19 := 1068,
	PRODUCTIONCOUNTERS_CAVITY_29_REJECTREASON_20 := 1069,
	MOULDMEASUREMENT_CAVITY_29_PEAKPRESSURE := 1070,
	MOULDMEASUREMENT_HOTRUNNER_CAVITY_29_TARGETVALUE := 1071,
	MOULDMEASUREMENT_HOTRUNNER_CAVITY_29_ACTUALVALUE := 1072,
	PRODUCTIONCOUNTERS_CAVITY_30_PRODUCED := 1073,
	PRODUCTIONCOUNTERS_CAVITY_30_STACKED := 1074,
	PRODUCTIONCOUNTERS_CAVITY_30_REJECTED := 1075,
	PRODUCTIONCOUNTERS_CAVITY_30_UNCOUNTEDREJECT := 1076,
	PRODUCTIONCOUNTERS_CAVITY_30_REJECTREASON_0 := 1077,
	PRODUCTIONCOUNTERS_CAVITY_30_REJECTREASON_1 := 1078,
	PRODUCTIONCOUNTERS_CAVITY_30_REJECTREASON_2 := 1079,
	PRODUCTIONCOUNTERS_CAVITY_30_REJECTREASON_3 := 1080,
	PRODUCTIONCOUNTERS_CAVITY_30_REJECTREASON_4 := 1081,
	PRODUCTIONCOUNTERS_CAVITY_30_REJECTREASON_5 := 1082,
	PRODUCTIONCOUNTERS_CAVITY_30_REJECTREASON_6 := 1083,
	PRODUCTIONCOUNTERS_CAVITY_30_REJECTREASON_7 := 1084,
	PRODUCTIONCOUNTERS_CAVITY_30_REJECTREASON_8 := 1085,
	PRODUCTIONCOUNTERS_CAVITY_30_REJECTREASON_9 := 1086,
	PRODUCTIONCOUNTERS_CAVITY_30_REJECTREASON_10 := 1087,
	PRODUCTIONCOUNTERS_CAVITY_30_REJECTREASON_11 := 1088,
	PRODUCTIONCOUNTERS_CAVITY_30_REJECTREASON_12 := 1089,
	PRODUCTIONCOUNTERS_CAVITY_30_REJECTREASON_13 := 1090,
	PRODUCTIONCOUNTERS_CAVITY_30_REJECTREASON_14 := 1091,
	PRODUCTIONCOUNTERS_CAVITY_30_REJECTREASON_15 := 1092,
	PRODUCTIONCOUNTERS_CAVITY_30_REJECTREASON_16 := 1093,
	PRODUCTIONCOUNTERS_CAVITY_30_REJECTREASON_17 := 1094,
	PRODUCTIONCOUNTERS_CAVITY_30_REJECTREASON_18 := 1095,
	PRODUCTIONCOUNTERS_CAVITY_30_REJECTREASON_19 := 1096,
	PRODUCTIONCOUNTERS_CAVITY_30_REJECTREASON_20 := 1097,
	MOULDMEASUREMENT_CAVITY_30_PEAKPRESSURE := 1098,
	MOULDMEASUREMENT_HOTRUNNER_CAVITY_30_TARGETVALUE := 1099,
	MOULDMEASUREMENT_HOTRUNNER_CAVITY_30_ACTUALVALUE := 1100,
	PRODUCTIONCOUNTERS_CAVITY_31_PRODUCED := 1101,
	PRODUCTIONCOUNTERS_CAVITY_31_STACKED := 1102,
	PRODUCTIONCOUNTERS_CAVITY_31_REJECTED := 1103,
	PRODUCTIONCOUNTERS_CAVITY_31_UNCOUNTEDREJECT := 1104,
	PRODUCTIONCOUNTERS_CAVITY_31_REJECTREASON_0 := 1105,
	PRODUCTIONCOUNTERS_CAVITY_31_REJECTREASON_1 := 1106,
	PRODUCTIONCOUNTERS_CAVITY_31_REJECTREASON_2 := 1107,
	PRODUCTIONCOUNTERS_CAVITY_31_REJECTREASON_3 := 1108,
	PRODUCTIONCOUNTERS_CAVITY_31_REJECTREASON_4 := 1109,
	PRODUCTIONCOUNTERS_CAVITY_31_REJECTREASON_5 := 1110,
	PRODUCTIONCOUNTERS_CAVITY_31_REJECTREASON_6 := 1111,
	PRODUCTIONCOUNTERS_CAVITY_31_REJECTREASON_7 := 1112,
	PRODUCTIONCOUNTERS_CAVITY_31_REJECTREASON_8 := 1113,
	PRODUCTIONCOUNTERS_CAVITY_31_REJECTREASON_9 := 1114,
	PRODUCTIONCOUNTERS_CAVITY_31_REJECTREASON_10 := 1115,
	PRODUCTIONCOUNTERS_CAVITY_31_REJECTREASON_11 := 1116,
	PRODUCTIONCOUNTERS_CAVITY_31_REJECTREASON_12 := 1117,
	PRODUCTIONCOUNTERS_CAVITY_31_REJECTREASON_13 := 1118,
	PRODUCTIONCOUNTERS_CAVITY_31_REJECTREASON_14 := 1119,
	PRODUCTIONCOUNTERS_CAVITY_31_REJECTREASON_15 := 1120,
	PRODUCTIONCOUNTERS_CAVITY_31_REJECTREASON_16 := 1121,
	PRODUCTIONCOUNTERS_CAVITY_31_REJECTREASON_17 := 1122,
	PRODUCTIONCOUNTERS_CAVITY_31_REJECTREASON_18 := 1123,
	PRODUCTIONCOUNTERS_CAVITY_31_REJECTREASON_19 := 1124,
	PRODUCTIONCOUNTERS_CAVITY_31_REJECTREASON_20 := 1125,
	MOULDMEASUREMENT_CAVITY_31_PEAKPRESSURE := 1126,
	MOULDMEASUREMENT_HOTRUNNER_CAVITY_31_TARGETVALUE := 1127,
	MOULDMEASUREMENT_HOTRUNNER_CAVITY_31_ACTUALVALUE := 1128,
	PRODUCTIONCOUNTERS_CAVITY_32_PRODUCED := 1129,
	PRODUCTIONCOUNTERS_CAVITY_32_STACKED := 1130,
	PRODUCTIONCOUNTERS_CAVITY_32_REJECTED := 1131,
	PRODUCTIONCOUNTERS_CAVITY_32_UNCOUNTEDREJECT := 1132,
	PRODUCTIONCOUNTERS_CAVITY_32_REJECTREASON_0 := 1133,
	PRODUCTIONCOUNTERS_CAVITY_32_REJECTREASON_1 := 1134,
	PRODUCTIONCOUNTERS_CAVITY_32_REJECTREASON_2 := 1135,
	PRODUCTIONCOUNTERS_CAVITY_32_REJECTREASON_3 := 1136,
	PRODUCTIONCOUNTERS_CAVITY_32_REJECTREASON_4 := 1137,
	PRODUCTIONCOUNTERS_CAVITY_32_REJECTREASON_5 := 1138,
	PRODUCTIONCOUNTERS_CAVITY_32_REJECTREASON_6 := 1139,
	PRODUCTIONCOUNTERS_CAVITY_32_REJECTREASON_7 := 1140,
	PRODUCTIONCOUNTERS_CAVITY_32_REJECTREASON_8 := 1141,
	PRODUCTIONCOUNTERS_CAVITY_32_REJECTREASON_9 := 1142,
	PRODUCTIONCOUNTERS_CAVITY_32_REJECTREASON_10 := 1143,
	PRODUCTIONCOUNTERS_CAVITY_32_REJECTREASON_11 := 1144,
	PRODUCTIONCOUNTERS_CAVITY_32_REJECTREASON_12 := 1145,
	PRODUCTIONCOUNTERS_CAVITY_32_REJECTREASON_13 := 1146,
	PRODUCTIONCOUNTERS_CAVITY_32_REJECTREASON_14 := 1147,
	PRODUCTIONCOUNTERS_CAVITY_32_REJECTREASON_15 := 1148,
	PRODUCTIONCOUNTERS_CAVITY_32_REJECTREASON_16 := 1149,
	PRODUCTIONCOUNTERS_CAVITY_32_REJECTREASON_17 := 1150,
	PRODUCTIONCOUNTERS_CAVITY_32_REJECTREASON_18 := 1151,
	PRODUCTIONCOUNTERS_CAVITY_32_REJECTREASON_19 := 1152,
	PRODUCTIONCOUNTERS_CAVITY_32_REJECTREASON_20 := 1153,
	MOULDMEASUREMENT_CAVITY_32_PEAKPRESSURE := 1154,
	MOULDMEASUREMENT_HOTRUNNER_CAVITY_32_TARGETVALUE := 1155,
	MOULDMEASUREMENT_HOTRUNNER_CAVITY_32_ACTUALVALUE := 1156,
	PRODUCTIONCOUNTERS_CAVITY_33_PRODUCED := 1157,
	PRODUCTIONCOUNTERS_CAVITY_33_STACKED := 1158,
	PRODUCTIONCOUNTERS_CAVITY_33_REJECTED := 1159,
	PRODUCTIONCOUNTERS_CAVITY_33_UNCOUNTEDREJECT := 1160,
	PRODUCTIONCOUNTERS_CAVITY_33_REJECTREASON_0 := 1161,
	PRODUCTIONCOUNTERS_CAVITY_33_REJECTREASON_1 := 1162,
	PRODUCTIONCOUNTERS_CAVITY_33_REJECTREASON_2 := 1163,
	PRODUCTIONCOUNTERS_CAVITY_33_REJECTREASON_3 := 1164,
	PRODUCTIONCOUNTERS_CAVITY_33_REJECTREASON_4 := 1165,
	PRODUCTIONCOUNTERS_CAVITY_33_REJECTREASON_5 := 1166,
	PRODUCTIONCOUNTERS_CAVITY_33_REJECTREASON_6 := 1167,
	PRODUCTIONCOUNTERS_CAVITY_33_REJECTREASON_7 := 1168,
	PRODUCTIONCOUNTERS_CAVITY_33_REJECTREASON_8 := 1169,
	PRODUCTIONCOUNTERS_CAVITY_33_REJECTREASON_9 := 1170,
	PRODUCTIONCOUNTERS_CAVITY_33_REJECTREASON_10 := 1171,
	PRODUCTIONCOUNTERS_CAVITY_33_REJECTREASON_11 := 1172,
	PRODUCTIONCOUNTERS_CAVITY_33_REJECTREASON_12 := 1173,
	PRODUCTIONCOUNTERS_CAVITY_33_REJECTREASON_13 := 1174,
	PRODUCTIONCOUNTERS_CAVITY_33_REJECTREASON_14 := 1175,
	PRODUCTIONCOUNTERS_CAVITY_33_REJECTREASON_15 := 1176,
	PRODUCTIONCOUNTERS_CAVITY_33_REJECTREASON_16 := 1177,
	PRODUCTIONCOUNTERS_CAVITY_33_REJECTREASON_17 := 1178,
	PRODUCTIONCOUNTERS_CAVITY_33_REJECTREASON_18 := 1179,
	PRODUCTIONCOUNTERS_CAVITY_33_REJECTREASON_19 := 1180,
	PRODUCTIONCOUNTERS_CAVITY_33_REJECTREASON_20 := 1181,
	MOULDMEASUREMENT_CAVITY_33_PEAKPRESSURE := 1182,
	MOULDMEASUREMENT_HOTRUNNER_CAVITY_33_TARGETVALUE := 1183,
	MOULDMEASUREMENT_HOTRUNNER_CAVITY_33_ACTUALVALUE := 1184,
	PRODUCTIONCOUNTERS_CAVITY_34_PRODUCED := 1185,
	PRODUCTIONCOUNTERS_CAVITY_34_STACKED := 1186,
	PRODUCTIONCOUNTERS_CAVITY_34_REJECTED := 1187,
	PRODUCTIONCOUNTERS_CAVITY_34_UNCOUNTEDREJECT := 1188,
	PRODUCTIONCOUNTERS_CAVITY_34_REJECTREASON_0 := 1189,
	PRODUCTIONCOUNTERS_CAVITY_34_REJECTREASON_1 := 1190,
	PRODUCTIONCOUNTERS_CAVITY_34_REJECTREASON_2 := 1191,
	PRODUCTIONCOUNTERS_CAVITY_34_REJECTREASON_3 := 1192,
	PRODUCTIONCOUNTERS_CAVITY_34_REJECTREASON_4 := 1193,
	PRODUCTIONCOUNTERS_CAVITY_34_REJECTREASON_5 := 1194,
	PRODUCTIONCOUNTERS_CAVITY_34_REJECTREASON_6 := 1195,
	PRODUCTIONCOUNTERS_CAVITY_34_REJECTREASON_7 := 1196,
	PRODUCTIONCOUNTERS_CAVITY_34_REJECTREASON_8 := 1197,
	PRODUCTIONCOUNTERS_CAVITY_34_REJECTREASON_9 := 1198,
	PRODUCTIONCOUNTERS_CAVITY_34_REJECTREASON_10 := 1199,
	PRODUCTIONCOUNTERS_CAVITY_34_REJECTREASON_11 := 1200,
	PRODUCTIONCOUNTERS_CAVITY_34_REJECTREASON_12 := 1201,
	PRODUCTIONCOUNTERS_CAVITY_34_REJECTREASON_13 := 1202,
	PRODUCTIONCOUNTERS_CAVITY_34_REJECTREASON_14 := 1203,
	PRODUCTIONCOUNTERS_CAVITY_34_REJECTREASON_15 := 1204,
	PRODUCTIONCOUNTERS_CAVITY_34_REJECTREASON_16 := 1205,
	PRODUCTIONCOUNTERS_CAVITY_34_REJECTREASON_17 := 1206,
	PRODUCTIONCOUNTERS_CAVITY_34_REJECTREASON_18 := 1207,
	PRODUCTIONCOUNTERS_CAVITY_34_REJECTREASON_19 := 1208,
	PRODUCTIONCOUNTERS_CAVITY_34_REJECTREASON_20 := 1209,
	MOULDMEASUREMENT_CAVITY_34_PEAKPRESSURE := 1210,
	MOULDMEASUREMENT_HOTRUNNER_CAVITY_34_TARGETVALUE := 1211,
	MOULDMEASUREMENT_HOTRUNNER_CAVITY_34_ACTUALVALUE := 1212,
	PRODUCTIONCOUNTERS_CAVITY_35_PRODUCED := 1213,
	PRODUCTIONCOUNTERS_CAVITY_35_STACKED := 1214,
	PRODUCTIONCOUNTERS_CAVITY_35_REJECTED := 1215,
	PRODUCTIONCOUNTERS_CAVITY_35_UNCOUNTEDREJECT := 1216,
	PRODUCTIONCOUNTERS_CAVITY_35_REJECTREASON_0 := 1217,
	PRODUCTIONCOUNTERS_CAVITY_35_REJECTREASON_1 := 1218,
	PRODUCTIONCOUNTERS_CAVITY_35_REJECTREASON_2 := 1219,
	PRODUCTIONCOUNTERS_CAVITY_35_REJECTREASON_3 := 1220,
	PRODUCTIONCOUNTERS_CAVITY_35_REJECTREASON_4 := 1221,
	PRODUCTIONCOUNTERS_CAVITY_35_REJECTREASON_5 := 1222,
	PRODUCTIONCOUNTERS_CAVITY_35_REJECTREASON_6 := 1223,
	PRODUCTIONCOUNTERS_CAVITY_35_REJECTREASON_7 := 1224,
	PRODUCTIONCOUNTERS_CAVITY_35_REJECTREASON_8 := 1225,
	PRODUCTIONCOUNTERS_CAVITY_35_REJECTREASON_9 := 1226,
	PRODUCTIONCOUNTERS_CAVITY_35_REJECTREASON_10 := 1227,
	PRODUCTIONCOUNTERS_CAVITY_35_REJECTREASON_11 := 1228,
	PRODUCTIONCOUNTERS_CAVITY_35_REJECTREASON_12 := 1229,
	PRODUCTIONCOUNTERS_CAVITY_35_REJECTREASON_13 := 1230,
	PRODUCTIONCOUNTERS_CAVITY_35_REJECTREASON_14 := 1231,
	PRODUCTIONCOUNTERS_CAVITY_35_REJECTREASON_15 := 1232,
	PRODUCTIONCOUNTERS_CAVITY_35_REJECTREASON_16 := 1233,
	PRODUCTIONCOUNTERS_CAVITY_35_REJECTREASON_17 := 1234,
	PRODUCTIONCOUNTERS_CAVITY_35_REJECTREASON_18 := 1235,
	PRODUCTIONCOUNTERS_CAVITY_35_REJECTREASON_19 := 1236,
	PRODUCTIONCOUNTERS_CAVITY_35_REJECTREASON_20 := 1237,
	MOULDMEASUREMENT_CAVITY_35_PEAKPRESSURE := 1238,
	MOULDMEASUREMENT_HOTRUNNER_CAVITY_35_TARGETVALUE := 1239,
	MOULDMEASUREMENT_HOTRUNNER_CAVITY_35_ACTUALVALUE := 1240,
	PRODUCTIONCOUNTERS_CAVITY_36_PRODUCED := 1241,
	PRODUCTIONCOUNTERS_CAVITY_36_STACKED := 1242,
	PRODUCTIONCOUNTERS_CAVITY_36_REJECTED := 1243,
	PRODUCTIONCOUNTERS_CAVITY_36_UNCOUNTEDREJECT := 1244,
	PRODUCTIONCOUNTERS_CAVITY_36_REJECTREASON_0 := 1245,
	PRODUCTIONCOUNTERS_CAVITY_36_REJECTREASON_1 := 1246,
	PRODUCTIONCOUNTERS_CAVITY_36_REJECTREASON_2 := 1247,
	PRODUCTIONCOUNTERS_CAVITY_36_REJECTREASON_3 := 1248,
	PRODUCTIONCOUNTERS_CAVITY_36_REJECTREASON_4 := 1249,
	PRODUCTIONCOUNTERS_CAVITY_36_REJECTREASON_5 := 1250,
	PRODUCTIONCOUNTERS_CAVITY_36_REJECTREASON_6 := 1251,
	PRODUCTIONCOUNTERS_CAVITY_36_REJECTREASON_7 := 1252,
	PRODUCTIONCOUNTERS_CAVITY_36_REJECTREASON_8 := 1253,
	PRODUCTIONCOUNTERS_CAVITY_36_REJECTREASON_9 := 1254,
	PRODUCTIONCOUNTERS_CAVITY_36_REJECTREASON_10 := 1255,
	PRODUCTIONCOUNTERS_CAVITY_36_REJECTREASON_11 := 1256,
	PRODUCTIONCOUNTERS_CAVITY_36_REJECTREASON_12 := 1257,
	PRODUCTIONCOUNTERS_CAVITY_36_REJECTREASON_13 := 1258,
	PRODUCTIONCOUNTERS_CAVITY_36_REJECTREASON_14 := 1259,
	PRODUCTIONCOUNTERS_CAVITY_36_REJECTREASON_15 := 1260,
	PRODUCTIONCOUNTERS_CAVITY_36_REJECTREASON_16 := 1261,
	PRODUCTIONCOUNTERS_CAVITY_36_REJECTREASON_17 := 1262,
	PRODUCTIONCOUNTERS_CAVITY_36_REJECTREASON_18 := 1263,
	PRODUCTIONCOUNTERS_CAVITY_36_REJECTREASON_19 := 1264,
	PRODUCTIONCOUNTERS_CAVITY_36_REJECTREASON_20 := 1265,
	MOULDMEASUREMENT_CAVITY_36_PEAKPRESSURE := 1266,
	MOULDMEASUREMENT_HOTRUNNER_CAVITY_36_TARGETVALUE := 1267,
	MOULDMEASUREMENT_HOTRUNNER_CAVITY_36_ACTUALVALUE := 1268,
	PRODUCTIONCOUNTERS_CAVITY_37_PRODUCED := 1269,
	PRODUCTIONCOUNTERS_CAVITY_37_STACKED := 1270,
	PRODUCTIONCOUNTERS_CAVITY_37_REJECTED := 1271,
	PRODUCTIONCOUNTERS_CAVITY_37_UNCOUNTEDREJECT := 1272,
	PRODUCTIONCOUNTERS_CAVITY_37_REJECTREASON_0 := 1273,
	PRODUCTIONCOUNTERS_CAVITY_37_REJECTREASON_1 := 1274,
	PRODUCTIONCOUNTERS_CAVITY_37_REJECTREASON_2 := 1275,
	PRODUCTIONCOUNTERS_CAVITY_37_REJECTREASON_3 := 1276,
	PRODUCTIONCOUNTERS_CAVITY_37_REJECTREASON_4 := 1277,
	PRODUCTIONCOUNTERS_CAVITY_37_REJECTREASON_5 := 1278,
	PRODUCTIONCOUNTERS_CAVITY_37_REJECTREASON_6 := 1279,
	PRODUCTIONCOUNTERS_CAVITY_37_REJECTREASON_7 := 1280,
	PRODUCTIONCOUNTERS_CAVITY_37_REJECTREASON_8 := 1281,
	PRODUCTIONCOUNTERS_CAVITY_37_REJECTREASON_9 := 1282,
	PRODUCTIONCOUNTERS_CAVITY_37_REJECTREASON_10 := 1283,
	PRODUCTIONCOUNTERS_CAVITY_37_REJECTREASON_11 := 1284,
	PRODUCTIONCOUNTERS_CAVITY_37_REJECTREASON_12 := 1285,
	PRODUCTIONCOUNTERS_CAVITY_37_REJECTREASON_13 := 1286,
	PRODUCTIONCOUNTERS_CAVITY_37_REJECTREASON_14 := 1287,
	PRODUCTIONCOUNTERS_CAVITY_37_REJECTREASON_15 := 1288,
	PRODUCTIONCOUNTERS_CAVITY_37_REJECTREASON_16 := 1289,
	PRODUCTIONCOUNTERS_CAVITY_37_REJECTREASON_17 := 1290,
	PRODUCTIONCOUNTERS_CAVITY_37_REJECTREASON_18 := 1291,
	PRODUCTIONCOUNTERS_CAVITY_37_REJECTREASON_19 := 1292,
	PRODUCTIONCOUNTERS_CAVITY_37_REJECTREASON_20 := 1293,
	MOULDMEASUREMENT_CAVITY_37_PEAKPRESSURE := 1294,
	MOULDMEASUREMENT_HOTRUNNER_CAVITY_37_TARGETVALUE := 1295,
	MOULDMEASUREMENT_HOTRUNNER_CAVITY_37_ACTUALVALUE := 1296,
	PRODUCTIONCOUNTERS_CAVITY_38_PRODUCED := 1297,
	PRODUCTIONCOUNTERS_CAVITY_38_STACKED := 1298,
	PRODUCTIONCOUNTERS_CAVITY_38_REJECTED := 1299,
	PRODUCTIONCOUNTERS_CAVITY_38_UNCOUNTEDREJECT := 1300,
	PRODUCTIONCOUNTERS_CAVITY_38_REJECTREASON_0 := 1301,
	PRODUCTIONCOUNTERS_CAVITY_38_REJECTREASON_1 := 1302,
	PRODUCTIONCOUNTERS_CAVITY_38_REJECTREASON_2 := 1303,
	PRODUCTIONCOUNTERS_CAVITY_38_REJECTREASON_3 := 1304,
	PRODUCTIONCOUNTERS_CAVITY_38_REJECTREASON_4 := 1305,
	PRODUCTIONCOUNTERS_CAVITY_38_REJECTREASON_5 := 1306,
	PRODUCTIONCOUNTERS_CAVITY_38_REJECTREASON_6 := 1307,
	PRODUCTIONCOUNTERS_CAVITY_38_REJECTREASON_7 := 1308,
	PRODUCTIONCOUNTERS_CAVITY_38_REJECTREASON_8 := 1309,
	PRODUCTIONCOUNTERS_CAVITY_38_REJECTREASON_9 := 1310,
	PRODUCTIONCOUNTERS_CAVITY_38_REJECTREASON_10 := 1311,
	PRODUCTIONCOUNTERS_CAVITY_38_REJECTREASON_11 := 1312,
	PRODUCTIONCOUNTERS_CAVITY_38_REJECTREASON_12 := 1313,
	PRODUCTIONCOUNTERS_CAVITY_38_REJECTREASON_13 := 1314,
	PRODUCTIONCOUNTERS_CAVITY_38_REJECTREASON_14 := 1315,
	PRODUCTIONCOUNTERS_CAVITY_38_REJECTREASON_15 := 1316,
	PRODUCTIONCOUNTERS_CAVITY_38_REJECTREASON_16 := 1317,
	PRODUCTIONCOUNTERS_CAVITY_38_REJECTREASON_17 := 1318,
	PRODUCTIONCOUNTERS_CAVITY_38_REJECTREASON_18 := 1319,
	PRODUCTIONCOUNTERS_CAVITY_38_REJECTREASON_19 := 1320,
	PRODUCTIONCOUNTERS_CAVITY_38_REJECTREASON_20 := 1321,
	MOULDMEASUREMENT_CAVITY_38_PEAKPRESSURE := 1322,
	MOULDMEASUREMENT_HOTRUNNER_CAVITY_38_TARGETVALUE := 1323,
	MOULDMEASUREMENT_HOTRUNNER_CAVITY_38_ACTUALVALUE := 1324,
	PRODUCTIONCOUNTERS_CAVITY_39_PRODUCED := 1325,
	PRODUCTIONCOUNTERS_CAVITY_39_STACKED := 1326,
	PRODUCTIONCOUNTERS_CAVITY_39_REJECTED := 1327,
	PRODUCTIONCOUNTERS_CAVITY_39_UNCOUNTEDREJECT := 1328,
	PRODUCTIONCOUNTERS_CAVITY_39_REJECTREASON_0 := 1329,
	PRODUCTIONCOUNTERS_CAVITY_39_REJECTREASON_1 := 1330,
	PRODUCTIONCOUNTERS_CAVITY_39_REJECTREASON_2 := 1331,
	PRODUCTIONCOUNTERS_CAVITY_39_REJECTREASON_3 := 1332,
	PRODUCTIONCOUNTERS_CAVITY_39_REJECTREASON_4 := 1333,
	PRODUCTIONCOUNTERS_CAVITY_39_REJECTREASON_5 := 1334,
	PRODUCTIONCOUNTERS_CAVITY_39_REJECTREASON_6 := 1335,
	PRODUCTIONCOUNTERS_CAVITY_39_REJECTREASON_7 := 1336,
	PRODUCTIONCOUNTERS_CAVITY_39_REJECTREASON_8 := 1337,
	PRODUCTIONCOUNTERS_CAVITY_39_REJECTREASON_9 := 1338,
	PRODUCTIONCOUNTERS_CAVITY_39_REJECTREASON_10 := 1339,
	PRODUCTIONCOUNTERS_CAVITY_39_REJECTREASON_11 := 1340,
	PRODUCTIONCOUNTERS_CAVITY_39_REJECTREASON_12 := 1341,
	PRODUCTIONCOUNTERS_CAVITY_39_REJECTREASON_13 := 1342,
	PRODUCTIONCOUNTERS_CAVITY_39_REJECTREASON_14 := 1343,
	PRODUCTIONCOUNTERS_CAVITY_39_REJECTREASON_15 := 1344,
	PRODUCTIONCOUNTERS_CAVITY_39_REJECTREASON_16 := 1345,
	PRODUCTIONCOUNTERS_CAVITY_39_REJECTREASON_17 := 1346,
	PRODUCTIONCOUNTERS_CAVITY_39_REJECTREASON_18 := 1347,
	PRODUCTIONCOUNTERS_CAVITY_39_REJECTREASON_19 := 1348,
	PRODUCTIONCOUNTERS_CAVITY_39_REJECTREASON_20 := 1349,
	MOULDMEASUREMENT_CAVITY_39_PEAKPRESSURE := 1350,
	MOULDMEASUREMENT_HOTRUNNER_CAVITY_39_TARGETVALUE := 1351,
	MOULDMEASUREMENT_HOTRUNNER_CAVITY_39_ACTUALVALUE := 1352,
	PRODUCTIONCOUNTERS_CAVITY_40_PRODUCED := 1353,
	PRODUCTIONCOUNTERS_CAVITY_40_STACKED := 1354,
	PRODUCTIONCOUNTERS_CAVITY_40_REJECTED := 1355,
	PRODUCTIONCOUNTERS_CAVITY_40_UNCOUNTEDREJECT := 1356,
	PRODUCTIONCOUNTERS_CAVITY_40_REJECTREASON_0 := 1357,
	PRODUCTIONCOUNTERS_CAVITY_40_REJECTREASON_1 := 1358,
	PRODUCTIONCOUNTERS_CAVITY_40_REJECTREASON_2 := 1359,
	PRODUCTIONCOUNTERS_CAVITY_40_REJECTREASON_3 := 1360,
	PRODUCTIONCOUNTERS_CAVITY_40_REJECTREASON_4 := 1361,
	PRODUCTIONCOUNTERS_CAVITY_40_REJECTREASON_5 := 1362,
	PRODUCTIONCOUNTERS_CAVITY_40_REJECTREASON_6 := 1363,
	PRODUCTIONCOUNTERS_CAVITY_40_REJECTREASON_7 := 1364,
	PRODUCTIONCOUNTERS_CAVITY_40_REJECTREASON_8 := 1365,
	PRODUCTIONCOUNTERS_CAVITY_40_REJECTREASON_9 := 1366,
	PRODUCTIONCOUNTERS_CAVITY_40_REJECTREASON_10 := 1367,
	PRODUCTIONCOUNTERS_CAVITY_40_REJECTREASON_11 := 1368,
	PRODUCTIONCOUNTERS_CAVITY_40_REJECTREASON_12 := 1369,
	PRODUCTIONCOUNTERS_CAVITY_40_REJECTREASON_13 := 1370,
	PRODUCTIONCOUNTERS_CAVITY_40_REJECTREASON_14 := 1371,
	PRODUCTIONCOUNTERS_CAVITY_40_REJECTREASON_15 := 1372,
	PRODUCTIONCOUNTERS_CAVITY_40_REJECTREASON_16 := 1373,
	PRODUCTIONCOUNTERS_CAVITY_40_REJECTREASON_17 := 1374,
	PRODUCTIONCOUNTERS_CAVITY_40_REJECTREASON_18 := 1375,
	PRODUCTIONCOUNTERS_CAVITY_40_REJECTREASON_19 := 1376,
	PRODUCTIONCOUNTERS_CAVITY_40_REJECTREASON_20 := 1377,
	MOULDMEASUREMENT_CAVITY_40_PEAKPRESSURE := 1378,
	MOULDMEASUREMENT_HOTRUNNER_CAVITY_40_TARGETVALUE := 1379,
	MOULDMEASUREMENT_HOTRUNNER_CAVITY_40_ACTUALVALUE := 1380,
	PRODUCTIONCOUNTERS_CAVITY_41_PRODUCED := 1381,
	PRODUCTIONCOUNTERS_CAVITY_41_STACKED := 1382,
	PRODUCTIONCOUNTERS_CAVITY_41_REJECTED := 1383,
	PRODUCTIONCOUNTERS_CAVITY_41_UNCOUNTEDREJECT := 1384,
	PRODUCTIONCOUNTERS_CAVITY_41_REJECTREASON_0 := 1385,
	PRODUCTIONCOUNTERS_CAVITY_41_REJECTREASON_1 := 1386,
	PRODUCTIONCOUNTERS_CAVITY_41_REJECTREASON_2 := 1387,
	PRODUCTIONCOUNTERS_CAVITY_41_REJECTREASON_3 := 1388,
	PRODUCTIONCOUNTERS_CAVITY_41_REJECTREASON_4 := 1389,
	PRODUCTIONCOUNTERS_CAVITY_41_REJECTREASON_5 := 1390,
	PRODUCTIONCOUNTERS_CAVITY_41_REJECTREASON_6 := 1391,
	PRODUCTIONCOUNTERS_CAVITY_41_REJECTREASON_7 := 1392,
	PRODUCTIONCOUNTERS_CAVITY_41_REJECTREASON_8 := 1393,
	PRODUCTIONCOUNTERS_CAVITY_41_REJECTREASON_9 := 1394,
	PRODUCTIONCOUNTERS_CAVITY_41_REJECTREASON_10 := 1395,
	PRODUCTIONCOUNTERS_CAVITY_41_REJECTREASON_11 := 1396,
	PRODUCTIONCOUNTERS_CAVITY_41_REJECTREASON_12 := 1397,
	PRODUCTIONCOUNTERS_CAVITY_41_REJECTREASON_13 := 1398,
	PRODUCTIONCOUNTERS_CAVITY_41_REJECTREASON_14 := 1399,
	PRODUCTIONCOUNTERS_CAVITY_41_REJECTREASON_15 := 1400,
	PRODUCTIONCOUNTERS_CAVITY_41_REJECTREASON_16 := 1401,
	PRODUCTIONCOUNTERS_CAVITY_41_REJECTREASON_17 := 1402,
	PRODUCTIONCOUNTERS_CAVITY_41_REJECTREASON_18 := 1403,
	PRODUCTIONCOUNTERS_CAVITY_41_REJECTREASON_19 := 1404,
	PRODUCTIONCOUNTERS_CAVITY_41_REJECTREASON_20 := 1405,
	MOULDMEASUREMENT_CAVITY_41_PEAKPRESSURE := 1406,
	MOULDMEASUREMENT_HOTRUNNER_CAVITY_41_TARGETVALUE := 1407,
	MOULDMEASUREMENT_HOTRUNNER_CAVITY_41_ACTUALVALUE := 1408,
	PRODUCTIONCOUNTERS_CAVITY_42_PRODUCED := 1409,
	PRODUCTIONCOUNTERS_CAVITY_42_STACKED := 1410,
	PRODUCTIONCOUNTERS_CAVITY_42_REJECTED := 1411,
	PRODUCTIONCOUNTERS_CAVITY_42_UNCOUNTEDREJECT := 1412,
	PRODUCTIONCOUNTERS_CAVITY_42_REJECTREASON_0 := 1413,
	PRODUCTIONCOUNTERS_CAVITY_42_REJECTREASON_1 := 1414,
	PRODUCTIONCOUNTERS_CAVITY_42_REJECTREASON_2 := 1415,
	PRODUCTIONCOUNTERS_CAVITY_42_REJECTREASON_3 := 1416,
	PRODUCTIONCOUNTERS_CAVITY_42_REJECTREASON_4 := 1417,
	PRODUCTIONCOUNTERS_CAVITY_42_REJECTREASON_5 := 1418,
	PRODUCTIONCOUNTERS_CAVITY_42_REJECTREASON_6 := 1419,
	PRODUCTIONCOUNTERS_CAVITY_42_REJECTREASON_7 := 1420,
	PRODUCTIONCOUNTERS_CAVITY_42_REJECTREASON_8 := 1421,
	PRODUCTIONCOUNTERS_CAVITY_42_REJECTREASON_9 := 1422,
	PRODUCTIONCOUNTERS_CAVITY_42_REJECTREASON_10 := 1423,
	PRODUCTIONCOUNTERS_CAVITY_42_REJECTREASON_11 := 1424,
	PRODUCTIONCOUNTERS_CAVITY_42_REJECTREASON_12 := 1425,
	PRODUCTIONCOUNTERS_CAVITY_42_REJECTREASON_13 := 1426,
	PRODUCTIONCOUNTERS_CAVITY_42_REJECTREASON_14 := 1427,
	PRODUCTIONCOUNTERS_CAVITY_42_REJECTREASON_15 := 1428,
	PRODUCTIONCOUNTERS_CAVITY_42_REJECTREASON_16 := 1429,
	PRODUCTIONCOUNTERS_CAVITY_42_REJECTREASON_17 := 1430,
	PRODUCTIONCOUNTERS_CAVITY_42_REJECTREASON_18 := 1431,
	PRODUCTIONCOUNTERS_CAVITY_42_REJECTREASON_19 := 1432,
	PRODUCTIONCOUNTERS_CAVITY_42_REJECTREASON_20 := 1433,
	MOULDMEASUREMENT_CAVITY_42_PEAKPRESSURE := 1434,
	MOULDMEASUREMENT_HOTRUNNER_CAVITY_42_TARGETVALUE := 1435,
	MOULDMEASUREMENT_HOTRUNNER_CAVITY_42_ACTUALVALUE := 1436,
	PRODUCTIONCOUNTERS_CAVITY_43_PRODUCED := 1437,
	PRODUCTIONCOUNTERS_CAVITY_43_STACKED := 1438,
	PRODUCTIONCOUNTERS_CAVITY_43_REJECTED := 1439,
	PRODUCTIONCOUNTERS_CAVITY_43_UNCOUNTEDREJECT := 1440,
	PRODUCTIONCOUNTERS_CAVITY_43_REJECTREASON_0 := 1441,
	PRODUCTIONCOUNTERS_CAVITY_43_REJECTREASON_1 := 1442,
	PRODUCTIONCOUNTERS_CAVITY_43_REJECTREASON_2 := 1443,
	PRODUCTIONCOUNTERS_CAVITY_43_REJECTREASON_3 := 1444,
	PRODUCTIONCOUNTERS_CAVITY_43_REJECTREASON_4 := 1445,
	PRODUCTIONCOUNTERS_CAVITY_43_REJECTREASON_5 := 1446,
	PRODUCTIONCOUNTERS_CAVITY_43_REJECTREASON_6 := 1447,
	PRODUCTIONCOUNTERS_CAVITY_43_REJECTREASON_7 := 1448,
	PRODUCTIONCOUNTERS_CAVITY_43_REJECTREASON_8 := 1449,
	PRODUCTIONCOUNTERS_CAVITY_43_REJECTREASON_9 := 1450,
	PRODUCTIONCOUNTERS_CAVITY_43_REJECTREASON_10 := 1451,
	PRODUCTIONCOUNTERS_CAVITY_43_REJECTREASON_11 := 1452,
	PRODUCTIONCOUNTERS_CAVITY_43_REJECTREASON_12 := 1453,
	PRODUCTIONCOUNTERS_CAVITY_43_REJECTREASON_13 := 1454,
	PRODUCTIONCOUNTERS_CAVITY_43_REJECTREASON_14 := 1455,
	PRODUCTIONCOUNTERS_CAVITY_43_REJECTREASON_15 := 1456,
	PRODUCTIONCOUNTERS_CAVITY_43_REJECTREASON_16 := 1457,
	PRODUCTIONCOUNTERS_CAVITY_43_REJECTREASON_17 := 1458,
	PRODUCTIONCOUNTERS_CAVITY_43_REJECTREASON_18 := 1459,
	PRODUCTIONCOUNTERS_CAVITY_43_REJECTREASON_19 := 1460,
	PRODUCTIONCOUNTERS_CAVITY_43_REJECTREASON_20 := 1461,
	MOULDMEASUREMENT_CAVITY_43_PEAKPRESSURE := 1462,
	MOULDMEASUREMENT_HOTRUNNER_CAVITY_43_TARGETVALUE := 1463,
	MOULDMEASUREMENT_HOTRUNNER_CAVITY_43_ACTUALVALUE := 1464,
	PRODUCTIONCOUNTERS_CAVITY_44_PRODUCED := 1465,
	PRODUCTIONCOUNTERS_CAVITY_44_STACKED := 1466,
	PRODUCTIONCOUNTERS_CAVITY_44_REJECTED := 1467,
	PRODUCTIONCOUNTERS_CAVITY_44_UNCOUNTEDREJECT := 1468,
	PRODUCTIONCOUNTERS_CAVITY_44_REJECTREASON_0 := 1469,
	PRODUCTIONCOUNTERS_CAVITY_44_REJECTREASON_1 := 1470,
	PRODUCTIONCOUNTERS_CAVITY_44_REJECTREASON_2 := 1471,
	PRODUCTIONCOUNTERS_CAVITY_44_REJECTREASON_3 := 1472,
	PRODUCTIONCOUNTERS_CAVITY_44_REJECTREASON_4 := 1473,
	PRODUCTIONCOUNTERS_CAVITY_44_REJECTREASON_5 := 1474,
	PRODUCTIONCOUNTERS_CAVITY_44_REJECTREASON_6 := 1475,
	PRODUCTIONCOUNTERS_CAVITY_44_REJECTREASON_7 := 1476,
	PRODUCTIONCOUNTERS_CAVITY_44_REJECTREASON_8 := 1477,
	PRODUCTIONCOUNTERS_CAVITY_44_REJECTREASON_9 := 1478,
	PRODUCTIONCOUNTERS_CAVITY_44_REJECTREASON_10 := 1479,
	PRODUCTIONCOUNTERS_CAVITY_44_REJECTREASON_11 := 1480,
	PRODUCTIONCOUNTERS_CAVITY_44_REJECTREASON_12 := 1481,
	PRODUCTIONCOUNTERS_CAVITY_44_REJECTREASON_13 := 1482,
	PRODUCTIONCOUNTERS_CAVITY_44_REJECTREASON_14 := 1483,
	PRODUCTIONCOUNTERS_CAVITY_44_REJECTREASON_15 := 1484,
	PRODUCTIONCOUNTERS_CAVITY_44_REJECTREASON_16 := 1485,
	PRODUCTIONCOUNTERS_CAVITY_44_REJECTREASON_17 := 1486,
	PRODUCTIONCOUNTERS_CAVITY_44_REJECTREASON_18 := 1487,
	PRODUCTIONCOUNTERS_CAVITY_44_REJECTREASON_19 := 1488,
	PRODUCTIONCOUNTERS_CAVITY_44_REJECTREASON_20 := 1489,
	MOULDMEASUREMENT_CAVITY_44_PEAKPRESSURE := 1490,
	MOULDMEASUREMENT_HOTRUNNER_CAVITY_44_TARGETVALUE := 1491,
	MOULDMEASUREMENT_HOTRUNNER_CAVITY_44_ACTUALVALUE := 1492,
	PRODUCTIONCOUNTERS_CAVITY_45_PRODUCED := 1493,
	PRODUCTIONCOUNTERS_CAVITY_45_STACKED := 1494,
	PRODUCTIONCOUNTERS_CAVITY_45_REJECTED := 1495,
	PRODUCTIONCOUNTERS_CAVITY_45_UNCOUNTEDREJECT := 1496,
	PRODUCTIONCOUNTERS_CAVITY_45_REJECTREASON_0 := 1497,
	PRODUCTIONCOUNTERS_CAVITY_45_REJECTREASON_1 := 1498,
	PRODUCTIONCOUNTERS_CAVITY_45_REJECTREASON_2 := 1499,
	PRODUCTIONCOUNTERS_CAVITY_45_REJECTREASON_3 := 1500,
	PRODUCTIONCOUNTERS_CAVITY_45_REJECTREASON_4 := 1501,
	PRODUCTIONCOUNTERS_CAVITY_45_REJECTREASON_5 := 1502,
	PRODUCTIONCOUNTERS_CAVITY_45_REJECTREASON_6 := 1503,
	PRODUCTIONCOUNTERS_CAVITY_45_REJECTREASON_7 := 1504,
	PRODUCTIONCOUNTERS_CAVITY_45_REJECTREASON_8 := 1505,
	PRODUCTIONCOUNTERS_CAVITY_45_REJECTREASON_9 := 1506,
	PRODUCTIONCOUNTERS_CAVITY_45_REJECTREASON_10 := 1507,
	PRODUCTIONCOUNTERS_CAVITY_45_REJECTREASON_11 := 1508,
	PRODUCTIONCOUNTERS_CAVITY_45_REJECTREASON_12 := 1509,
	PRODUCTIONCOUNTERS_CAVITY_45_REJECTREASON_13 := 1510,
	PRODUCTIONCOUNTERS_CAVITY_45_REJECTREASON_14 := 1511,
	PRODUCTIONCOUNTERS_CAVITY_45_REJECTREASON_15 := 1512,
	PRODUCTIONCOUNTERS_CAVITY_45_REJECTREASON_16 := 1513,
	PRODUCTIONCOUNTERS_CAVITY_45_REJECTREASON_17 := 1514,
	PRODUCTIONCOUNTERS_CAVITY_45_REJECTREASON_18 := 1515,
	PRODUCTIONCOUNTERS_CAVITY_45_REJECTREASON_19 := 1516,
	PRODUCTIONCOUNTERS_CAVITY_45_REJECTREASON_20 := 1517,
	MOULDMEASUREMENT_CAVITY_45_PEAKPRESSURE := 1518,
	MOULDMEASUREMENT_HOTRUNNER_CAVITY_45_TARGETVALUE := 1519,
	MOULDMEASUREMENT_HOTRUNNER_CAVITY_45_ACTUALVALUE := 1520,
	PRODUCTIONCOUNTERS_CAVITY_46_PRODUCED := 1521,
	PRODUCTIONCOUNTERS_CAVITY_46_STACKED := 1522,
	PRODUCTIONCOUNTERS_CAVITY_46_REJECTED := 1523,
	PRODUCTIONCOUNTERS_CAVITY_46_UNCOUNTEDREJECT := 1524,
	PRODUCTIONCOUNTERS_CAVITY_46_REJECTREASON_0 := 1525,
	PRODUCTIONCOUNTERS_CAVITY_46_REJECTREASON_1 := 1526,
	PRODUCTIONCOUNTERS_CAVITY_46_REJECTREASON_2 := 1527,
	PRODUCTIONCOUNTERS_CAVITY_46_REJECTREASON_3 := 1528,
	PRODUCTIONCOUNTERS_CAVITY_46_REJECTREASON_4 := 1529,
	PRODUCTIONCOUNTERS_CAVITY_46_REJECTREASON_5 := 1530,
	PRODUCTIONCOUNTERS_CAVITY_46_REJECTREASON_6 := 1531,
	PRODUCTIONCOUNTERS_CAVITY_46_REJECTREASON_7 := 1532,
	PRODUCTIONCOUNTERS_CAVITY_46_REJECTREASON_8 := 1533,
	PRODUCTIONCOUNTERS_CAVITY_46_REJECTREASON_9 := 1534,
	PRODUCTIONCOUNTERS_CAVITY_46_REJECTREASON_10 := 1535,
	PRODUCTIONCOUNTERS_CAVITY_46_REJECTREASON_11 := 1536,
	PRODUCTIONCOUNTERS_CAVITY_46_REJECTREASON_12 := 1537,
	PRODUCTIONCOUNTERS_CAVITY_46_REJECTREASON_13 := 1538,
	PRODUCTIONCOUNTERS_CAVITY_46_REJECTREASON_14 := 1539,
	PRODUCTIONCOUNTERS_CAVITY_46_REJECTREASON_15 := 1540,
	PRODUCTIONCOUNTERS_CAVITY_46_REJECTREASON_16 := 1541,
	PRODUCTIONCOUNTERS_CAVITY_46_REJECTREASON_17 := 1542,
	PRODUCTIONCOUNTERS_CAVITY_46_REJECTREASON_18 := 1543,
	PRODUCTIONCOUNTERS_CAVITY_46_REJECTREASON_19 := 1544,
	PRODUCTIONCOUNTERS_CAVITY_46_REJECTREASON_20 := 1545,
	MOULDMEASUREMENT_CAVITY_46_PEAKPRESSURE := 1546,
	MOULDMEASUREMENT_HOTRUNNER_CAVITY_46_TARGETVALUE := 1547,
	MOULDMEASUREMENT_HOTRUNNER_CAVITY_46_ACTUALVALUE := 1548,
	PRODUCTIONCOUNTERS_CAVITY_47_PRODUCED := 1549,
	PRODUCTIONCOUNTERS_CAVITY_47_STACKED := 1550,
	PRODUCTIONCOUNTERS_CAVITY_47_REJECTED := 1551,
	PRODUCTIONCOUNTERS_CAVITY_47_UNCOUNTEDREJECT := 1552,
	PRODUCTIONCOUNTERS_CAVITY_47_REJECTREASON_0 := 1553,
	PRODUCTIONCOUNTERS_CAVITY_47_REJECTREASON_1 := 1554,
	PRODUCTIONCOUNTERS_CAVITY_47_REJECTREASON_2 := 1555,
	PRODUCTIONCOUNTERS_CAVITY_47_REJECTREASON_3 := 1556,
	PRODUCTIONCOUNTERS_CAVITY_47_REJECTREASON_4 := 1557,
	PRODUCTIONCOUNTERS_CAVITY_47_REJECTREASON_5 := 1558,
	PRODUCTIONCOUNTERS_CAVITY_47_REJECTREASON_6 := 1559,
	PRODUCTIONCOUNTERS_CAVITY_47_REJECTREASON_7 := 1560,
	PRODUCTIONCOUNTERS_CAVITY_47_REJECTREASON_8 := 1561,
	PRODUCTIONCOUNTERS_CAVITY_47_REJECTREASON_9 := 1562,
	PRODUCTIONCOUNTERS_CAVITY_47_REJECTREASON_10 := 1563,
	PRODUCTIONCOUNTERS_CAVITY_47_REJECTREASON_11 := 1564,
	PRODUCTIONCOUNTERS_CAVITY_47_REJECTREASON_12 := 1565,
	PRODUCTIONCOUNTERS_CAVITY_47_REJECTREASON_13 := 1566,
	PRODUCTIONCOUNTERS_CAVITY_47_REJECTREASON_14 := 1567,
	PRODUCTIONCOUNTERS_CAVITY_47_REJECTREASON_15 := 1568,
	PRODUCTIONCOUNTERS_CAVITY_47_REJECTREASON_16 := 1569,
	PRODUCTIONCOUNTERS_CAVITY_47_REJECTREASON_17 := 1570,
	PRODUCTIONCOUNTERS_CAVITY_47_REJECTREASON_18 := 1571,
	PRODUCTIONCOUNTERS_CAVITY_47_REJECTREASON_19 := 1572,
	PRODUCTIONCOUNTERS_CAVITY_47_REJECTREASON_20 := 1573,
	MOULDMEASUREMENT_CAVITY_47_PEAKPRESSURE := 1574,
	MOULDMEASUREMENT_HOTRUNNER_CAVITY_47_TARGETVALUE := 1575,
	MOULDMEASUREMENT_HOTRUNNER_CAVITY_47_ACTUALVALUE := 1576,
	PRODUCTIONCOUNTERS_CAVITY_48_PRODUCED := 1577,
	PRODUCTIONCOUNTERS_CAVITY_48_STACKED := 1578,
	PRODUCTIONCOUNTERS_CAVITY_48_REJECTED := 1579,
	PRODUCTIONCOUNTERS_CAVITY_48_UNCOUNTEDREJECT := 1580,
	PRODUCTIONCOUNTERS_CAVITY_48_REJECTREASON_0 := 1581,
	PRODUCTIONCOUNTERS_CAVITY_48_REJECTREASON_1 := 1582,
	PRODUCTIONCOUNTERS_CAVITY_48_REJECTREASON_2 := 1583,
	PRODUCTIONCOUNTERS_CAVITY_48_REJECTREASON_3 := 1584,
	PRODUCTIONCOUNTERS_CAVITY_48_REJECTREASON_4 := 1585,
	PRODUCTIONCOUNTERS_CAVITY_48_REJECTREASON_5 := 1586,
	PRODUCTIONCOUNTERS_CAVITY_48_REJECTREASON_6 := 1587,
	PRODUCTIONCOUNTERS_CAVITY_48_REJECTREASON_7 := 1588,
	PRODUCTIONCOUNTERS_CAVITY_48_REJECTREASON_8 := 1589,
	PRODUCTIONCOUNTERS_CAVITY_48_REJECTREASON_9 := 1590,
	PRODUCTIONCOUNTERS_CAVITY_48_REJECTREASON_10 := 1591,
	PRODUCTIONCOUNTERS_CAVITY_48_REJECTREASON_11 := 1592,
	PRODUCTIONCOUNTERS_CAVITY_48_REJECTREASON_12 := 1593,
	PRODUCTIONCOUNTERS_CAVITY_48_REJECTREASON_13 := 1594,
	PRODUCTIONCOUNTERS_CAVITY_48_REJECTREASON_14 := 1595,
	PRODUCTIONCOUNTERS_CAVITY_48_REJECTREASON_15 := 1596,
	PRODUCTIONCOUNTERS_CAVITY_48_REJECTREASON_16 := 1597,
	PRODUCTIONCOUNTERS_CAVITY_48_REJECTREASON_17 := 1598,
	PRODUCTIONCOUNTERS_CAVITY_48_REJECTREASON_18 := 1599,
	PRODUCTIONCOUNTERS_CAVITY_48_REJECTREASON_19 := 1600,
	PRODUCTIONCOUNTERS_CAVITY_48_REJECTREASON_20 := 1601,
	MOULDMEASUREMENT_CAVITY_48_PEAKPRESSURE := 1602,
	MOULDMEASUREMENT_HOTRUNNER_CAVITY_48_TARGETVALUE := 1603,
	MOULDMEASUREMENT_HOTRUNNER_CAVITY_48_ACTUALVALUE := 1604,
	PRODUCTIONCOUNTERS_CAVITY_49_PRODUCED := 1605,
	PRODUCTIONCOUNTERS_CAVITY_49_STACKED := 1606,
	PRODUCTIONCOUNTERS_CAVITY_49_REJECTED := 1607,
	PRODUCTIONCOUNTERS_CAVITY_49_UNCOUNTEDREJECT := 1608,
	PRODUCTIONCOUNTERS_CAVITY_49_REJECTREASON_0 := 1609,
	PRODUCTIONCOUNTERS_CAVITY_49_REJECTREASON_1 := 1610,
	PRODUCTIONCOUNTERS_CAVITY_49_REJECTREASON_2 := 1611,
	PRODUCTIONCOUNTERS_CAVITY_49_REJECTREASON_3 := 1612,
	PRODUCTIONCOUNTERS_CAVITY_49_REJECTREASON_4 := 1613,
	PRODUCTIONCOUNTERS_CAVITY_49_REJECTREASON_5 := 1614,
	PRODUCTIONCOUNTERS_CAVITY_49_REJECTREASON_6 := 1615,
	PRODUCTIONCOUNTERS_CAVITY_49_REJECTREASON_7 := 1616,
	PRODUCTIONCOUNTERS_CAVITY_49_REJECTREASON_8 := 1617,
	PRODUCTIONCOUNTERS_CAVITY_49_REJECTREASON_9 := 1618,
	PRODUCTIONCOUNTERS_CAVITY_49_REJECTREASON_10 := 1619,
	PRODUCTIONCOUNTERS_CAVITY_49_REJECTREASON_11 := 1620,
	PRODUCTIONCOUNTERS_CAVITY_49_REJECTREASON_12 := 1621,
	PRODUCTIONCOUNTERS_CAVITY_49_REJECTREASON_13 := 1622,
	PRODUCTIONCOUNTERS_CAVITY_49_REJECTREASON_14 := 1623,
	PRODUCTIONCOUNTERS_CAVITY_49_REJECTREASON_15 := 1624,
	PRODUCTIONCOUNTERS_CAVITY_49_REJECTREASON_16 := 1625,
	PRODUCTIONCOUNTERS_CAVITY_49_REJECTREASON_17 := 1626,
	PRODUCTIONCOUNTERS_CAVITY_49_REJECTREASON_18 := 1627,
	PRODUCTIONCOUNTERS_CAVITY_49_REJECTREASON_19 := 1628,
	PRODUCTIONCOUNTERS_CAVITY_49_REJECTREASON_20 := 1629,
	MOULDMEASUREMENT_CAVITY_49_PEAKPRESSURE := 1630,
	MOULDMEASUREMENT_HOTRUNNER_CAVITY_49_TARGETVALUE := 1631,
	MOULDMEASUREMENT_HOTRUNNER_CAVITY_49_ACTUALVALUE := 1632,
	PRODUCTIONCOUNTERS_CAVITY_50_PRODUCED := 1633,
	PRODUCTIONCOUNTERS_CAVITY_50_STACKED := 1634,
	PRODUCTIONCOUNTERS_CAVITY_50_REJECTED := 1635,
	PRODUCTIONCOUNTERS_CAVITY_50_UNCOUNTEDREJECT := 1636,
	PRODUCTIONCOUNTERS_CAVITY_50_REJECTREASON_0 := 1637,
	PRODUCTIONCOUNTERS_CAVITY_50_REJECTREASON_1 := 1638,
	PRODUCTIONCOUNTERS_CAVITY_50_REJECTREASON_2 := 1639,
	PRODUCTIONCOUNTERS_CAVITY_50_REJECTREASON_3 := 1640,
	PRODUCTIONCOUNTERS_CAVITY_50_REJECTREASON_4 := 1641,
	PRODUCTIONCOUNTERS_CAVITY_50_REJECTREASON_5 := 1642,
	PRODUCTIONCOUNTERS_CAVITY_50_REJECTREASON_6 := 1643,
	PRODUCTIONCOUNTERS_CAVITY_50_REJECTREASON_7 := 1644,
	PRODUCTIONCOUNTERS_CAVITY_50_REJECTREASON_8 := 1645,
	PRODUCTIONCOUNTERS_CAVITY_50_REJECTREASON_9 := 1646,
	PRODUCTIONCOUNTERS_CAVITY_50_REJECTREASON_10 := 1647,
	PRODUCTIONCOUNTERS_CAVITY_50_REJECTREASON_11 := 1648,
	PRODUCTIONCOUNTERS_CAVITY_50_REJECTREASON_12 := 1649,
	PRODUCTIONCOUNTERS_CAVITY_50_REJECTREASON_13 := 1650,
	PRODUCTIONCOUNTERS_CAVITY_50_REJECTREASON_14 := 1651,
	PRODUCTIONCOUNTERS_CAVITY_50_REJECTREASON_15 := 1652,
	PRODUCTIONCOUNTERS_CAVITY_50_REJECTREASON_16 := 1653,
	PRODUCTIONCOUNTERS_CAVITY_50_REJECTREASON_17 := 1654,
	PRODUCTIONCOUNTERS_CAVITY_50_REJECTREASON_18 := 1655,
	PRODUCTIONCOUNTERS_CAVITY_50_REJECTREASON_19 := 1656,
	PRODUCTIONCOUNTERS_CAVITY_50_REJECTREASON_20 := 1657,
	MOULDMEASUREMENT_CAVITY_50_PEAKPRESSURE := 1658,
	MOULDMEASUREMENT_HOTRUNNER_CAVITY_50_TARGETVALUE := 1659,
	MOULDMEASUREMENT_HOTRUNNER_CAVITY_50_ACTUALVALUE := 1660,
	PRODUCTIONCOUNTERS_CAVITY_51_PRODUCED := 1661,
	PRODUCTIONCOUNTERS_CAVITY_51_STACKED := 1662,
	PRODUCTIONCOUNTERS_CAVITY_51_REJECTED := 1663,
	PRODUCTIONCOUNTERS_CAVITY_51_UNCOUNTEDREJECT := 1664,
	PRODUCTIONCOUNTERS_CAVITY_51_REJECTREASON_0 := 1665,
	PRODUCTIONCOUNTERS_CAVITY_51_REJECTREASON_1 := 1666,
	PRODUCTIONCOUNTERS_CAVITY_51_REJECTREASON_2 := 1667,
	PRODUCTIONCOUNTERS_CAVITY_51_REJECTREASON_3 := 1668,
	PRODUCTIONCOUNTERS_CAVITY_51_REJECTREASON_4 := 1669,
	PRODUCTIONCOUNTERS_CAVITY_51_REJECTREASON_5 := 1670,
	PRODUCTIONCOUNTERS_CAVITY_51_REJECTREASON_6 := 1671,
	PRODUCTIONCOUNTERS_CAVITY_51_REJECTREASON_7 := 1672,
	PRODUCTIONCOUNTERS_CAVITY_51_REJECTREASON_8 := 1673,
	PRODUCTIONCOUNTERS_CAVITY_51_REJECTREASON_9 := 1674,
	PRODUCTIONCOUNTERS_CAVITY_51_REJECTREASON_10 := 1675,
	PRODUCTIONCOUNTERS_CAVITY_51_REJECTREASON_11 := 1676,
	PRODUCTIONCOUNTERS_CAVITY_51_REJECTREASON_12 := 1677,
	PRODUCTIONCOUNTERS_CAVITY_51_REJECTREASON_13 := 1678,
	PRODUCTIONCOUNTERS_CAVITY_51_REJECTREASON_14 := 1679,
	PRODUCTIONCOUNTERS_CAVITY_51_REJECTREASON_15 := 1680,
	PRODUCTIONCOUNTERS_CAVITY_51_REJECTREASON_16 := 1681,
	PRODUCTIONCOUNTERS_CAVITY_51_REJECTREASON_17 := 1682,
	PRODUCTIONCOUNTERS_CAVITY_51_REJECTREASON_18 := 1683,
	PRODUCTIONCOUNTERS_CAVITY_51_REJECTREASON_19 := 1684,
	PRODUCTIONCOUNTERS_CAVITY_51_REJECTREASON_20 := 1685,
	MOULDMEASUREMENT_CAVITY_51_PEAKPRESSURE := 1686,
	MOULDMEASUREMENT_HOTRUNNER_CAVITY_51_TARGETVALUE := 1687,
	MOULDMEASUREMENT_HOTRUNNER_CAVITY_51_ACTUALVALUE := 1688,
	PRODUCTIONCOUNTERS_CAVITY_52_PRODUCED := 1689,
	PRODUCTIONCOUNTERS_CAVITY_52_STACKED := 1690,
	PRODUCTIONCOUNTERS_CAVITY_52_REJECTED := 1691,
	PRODUCTIONCOUNTERS_CAVITY_52_UNCOUNTEDREJECT := 1692,
	PRODUCTIONCOUNTERS_CAVITY_52_REJECTREASON_0 := 1693,
	PRODUCTIONCOUNTERS_CAVITY_52_REJECTREASON_1 := 1694,
	PRODUCTIONCOUNTERS_CAVITY_52_REJECTREASON_2 := 1695,
	PRODUCTIONCOUNTERS_CAVITY_52_REJECTREASON_3 := 1696,
	PRODUCTIONCOUNTERS_CAVITY_52_REJECTREASON_4 := 1697,
	PRODUCTIONCOUNTERS_CAVITY_52_REJECTREASON_5 := 1698,
	PRODUCTIONCOUNTERS_CAVITY_52_REJECTREASON_6 := 1699,
	PRODUCTIONCOUNTERS_CAVITY_52_REJECTREASON_7 := 1700,
	PRODUCTIONCOUNTERS_CAVITY_52_REJECTREASON_8 := 1701,
	PRODUCTIONCOUNTERS_CAVITY_52_REJECTREASON_9 := 1702,
	PRODUCTIONCOUNTERS_CAVITY_52_REJECTREASON_10 := 1703,
	PRODUCTIONCOUNTERS_CAVITY_52_REJECTREASON_11 := 1704,
	PRODUCTIONCOUNTERS_CAVITY_52_REJECTREASON_12 := 1705,
	PRODUCTIONCOUNTERS_CAVITY_52_REJECTREASON_13 := 1706,
	PRODUCTIONCOUNTERS_CAVITY_52_REJECTREASON_14 := 1707,
	PRODUCTIONCOUNTERS_CAVITY_52_REJECTREASON_15 := 1708,
	PRODUCTIONCOUNTERS_CAVITY_52_REJECTREASON_16 := 1709,
	PRODUCTIONCOUNTERS_CAVITY_52_REJECTREASON_17 := 1710,
	PRODUCTIONCOUNTERS_CAVITY_52_REJECTREASON_18 := 1711,
	PRODUCTIONCOUNTERS_CAVITY_52_REJECTREASON_19 := 1712,
	PRODUCTIONCOUNTERS_CAVITY_52_REJECTREASON_20 := 1713,
	MOULDMEASUREMENT_CAVITY_52_PEAKPRESSURE := 1714,
	MOULDMEASUREMENT_HOTRUNNER_CAVITY_52_TARGETVALUE := 1715,
	MOULDMEASUREMENT_HOTRUNNER_CAVITY_52_ACTUALVALUE := 1716,
	PRODUCTIONCOUNTERS_CAVITY_53_PRODUCED := 1717,
	PRODUCTIONCOUNTERS_CAVITY_53_STACKED := 1718,
	PRODUCTIONCOUNTERS_CAVITY_53_REJECTED := 1719,
	PRODUCTIONCOUNTERS_CAVITY_53_UNCOUNTEDREJECT := 1720,
	PRODUCTIONCOUNTERS_CAVITY_53_REJECTREASON_0 := 1721,
	PRODUCTIONCOUNTERS_CAVITY_53_REJECTREASON_1 := 1722,
	PRODUCTIONCOUNTERS_CAVITY_53_REJECTREASON_2 := 1723,
	PRODUCTIONCOUNTERS_CAVITY_53_REJECTREASON_3 := 1724,
	PRODUCTIONCOUNTERS_CAVITY_53_REJECTREASON_4 := 1725,
	PRODUCTIONCOUNTERS_CAVITY_53_REJECTREASON_5 := 1726,
	PRODUCTIONCOUNTERS_CAVITY_53_REJECTREASON_6 := 1727,
	PRODUCTIONCOUNTERS_CAVITY_53_REJECTREASON_7 := 1728,
	PRODUCTIONCOUNTERS_CAVITY_53_REJECTREASON_8 := 1729,
	PRODUCTIONCOUNTERS_CAVITY_53_REJECTREASON_9 := 1730,
	PRODUCTIONCOUNTERS_CAVITY_53_REJECTREASON_10 := 1731,
	PRODUCTIONCOUNTERS_CAVITY_53_REJECTREASON_11 := 1732,
	PRODUCTIONCOUNTERS_CAVITY_53_REJECTREASON_12 := 1733,
	PRODUCTIONCOUNTERS_CAVITY_53_REJECTREASON_13 := 1734,
	PRODUCTIONCOUNTERS_CAVITY_53_REJECTREASON_14 := 1735,
	PRODUCTIONCOUNTERS_CAVITY_53_REJECTREASON_15 := 1736,
	PRODUCTIONCOUNTERS_CAVITY_53_REJECTREASON_16 := 1737,
	PRODUCTIONCOUNTERS_CAVITY_53_REJECTREASON_17 := 1738,
	PRODUCTIONCOUNTERS_CAVITY_53_REJECTREASON_18 := 1739,
	PRODUCTIONCOUNTERS_CAVITY_53_REJECTREASON_19 := 1740,
	PRODUCTIONCOUNTERS_CAVITY_53_REJECTREASON_20 := 1741,
	MOULDMEASUREMENT_CAVITY_53_PEAKPRESSURE := 1742,
	MOULDMEASUREMENT_HOTRUNNER_CAVITY_53_TARGETVALUE := 1743,
	MOULDMEASUREMENT_HOTRUNNER_CAVITY_53_ACTUALVALUE := 1744,
	PRODUCTIONCOUNTERS_CAVITY_54_PRODUCED := 1745,
	PRODUCTIONCOUNTERS_CAVITY_54_STACKED := 1746,
	PRODUCTIONCOUNTERS_CAVITY_54_REJECTED := 1747,
	PRODUCTIONCOUNTERS_CAVITY_54_UNCOUNTEDREJECT := 1748,
	PRODUCTIONCOUNTERS_CAVITY_54_REJECTREASON_0 := 1749,
	PRODUCTIONCOUNTERS_CAVITY_54_REJECTREASON_1 := 1750,
	PRODUCTIONCOUNTERS_CAVITY_54_REJECTREASON_2 := 1751,
	PRODUCTIONCOUNTERS_CAVITY_54_REJECTREASON_3 := 1752,
	PRODUCTIONCOUNTERS_CAVITY_54_REJECTREASON_4 := 1753,
	PRODUCTIONCOUNTERS_CAVITY_54_REJECTREASON_5 := 1754,
	PRODUCTIONCOUNTERS_CAVITY_54_REJECTREASON_6 := 1755,
	PRODUCTIONCOUNTERS_CAVITY_54_REJECTREASON_7 := 1756,
	PRODUCTIONCOUNTERS_CAVITY_54_REJECTREASON_8 := 1757,
	PRODUCTIONCOUNTERS_CAVITY_54_REJECTREASON_9 := 1758,
	PRODUCTIONCOUNTERS_CAVITY_54_REJECTREASON_10 := 1759,
	PRODUCTIONCOUNTERS_CAVITY_54_REJECTREASON_11 := 1760,
	PRODUCTIONCOUNTERS_CAVITY_54_REJECTREASON_12 := 1761,
	PRODUCTIONCOUNTERS_CAVITY_54_REJECTREASON_13 := 1762,
	PRODUCTIONCOUNTERS_CAVITY_54_REJECTREASON_14 := 1763,
	PRODUCTIONCOUNTERS_CAVITY_54_REJECTREASON_15 := 1764,
	PRODUCTIONCOUNTERS_CAVITY_54_REJECTREASON_16 := 1765,
	PRODUCTIONCOUNTERS_CAVITY_54_REJECTREASON_17 := 1766,
	PRODUCTIONCOUNTERS_CAVITY_54_REJECTREASON_18 := 1767,
	PRODUCTIONCOUNTERS_CAVITY_54_REJECTREASON_19 := 1768,
	PRODUCTIONCOUNTERS_CAVITY_54_REJECTREASON_20 := 1769,
	MOULDMEASUREMENT_CAVITY_54_PEAKPRESSURE := 1770,
	MOULDMEASUREMENT_HOTRUNNER_CAVITY_54_TARGETVALUE := 1771,
	MOULDMEASUREMENT_HOTRUNNER_CAVITY_54_ACTUALVALUE := 1772,
	PRODUCTIONCOUNTERS_CAVITY_55_PRODUCED := 1773,
	PRODUCTIONCOUNTERS_CAVITY_55_STACKED := 1774,
	PRODUCTIONCOUNTERS_CAVITY_55_REJECTED := 1775,
	PRODUCTIONCOUNTERS_CAVITY_55_UNCOUNTEDREJECT := 1776,
	PRODUCTIONCOUNTERS_CAVITY_55_REJECTREASON_0 := 1777,
	PRODUCTIONCOUNTERS_CAVITY_55_REJECTREASON_1 := 1778,
	PRODUCTIONCOUNTERS_CAVITY_55_REJECTREASON_2 := 1779,
	PRODUCTIONCOUNTERS_CAVITY_55_REJECTREASON_3 := 1780,
	PRODUCTIONCOUNTERS_CAVITY_55_REJECTREASON_4 := 1781,
	PRODUCTIONCOUNTERS_CAVITY_55_REJECTREASON_5 := 1782,
	PRODUCTIONCOUNTERS_CAVITY_55_REJECTREASON_6 := 1783,
	PRODUCTIONCOUNTERS_CAVITY_55_REJECTREASON_7 := 1784,
	PRODUCTIONCOUNTERS_CAVITY_55_REJECTREASON_8 := 1785,
	PRODUCTIONCOUNTERS_CAVITY_55_REJECTREASON_9 := 1786,
	PRODUCTIONCOUNTERS_CAVITY_55_REJECTREASON_10 := 1787,
	PRODUCTIONCOUNTERS_CAVITY_55_REJECTREASON_11 := 1788,
	PRODUCTIONCOUNTERS_CAVITY_55_REJECTREASON_12 := 1789,
	PRODUCTIONCOUNTERS_CAVITY_55_REJECTREASON_13 := 1790,
	PRODUCTIONCOUNTERS_CAVITY_55_REJECTREASON_14 := 1791,
	PRODUCTIONCOUNTERS_CAVITY_55_REJECTREASON_15 := 1792,
	PRODUCTIONCOUNTERS_CAVITY_55_REJECTREASON_16 := 1793,
	PRODUCTIONCOUNTERS_CAVITY_55_REJECTREASON_17 := 1794,
	PRODUCTIONCOUNTERS_CAVITY_55_REJECTREASON_18 := 1795,
	PRODUCTIONCOUNTERS_CAVITY_55_REJECTREASON_19 := 1796,
	PRODUCTIONCOUNTERS_CAVITY_55_REJECTREASON_20 := 1797,
	MOULDMEASUREMENT_CAVITY_55_PEAKPRESSURE := 1798,
	MOULDMEASUREMENT_HOTRUNNER_CAVITY_55_TARGETVALUE := 1799,
	MOULDMEASUREMENT_HOTRUNNER_CAVITY_55_ACTUALVALUE := 1800,
	PRODUCTIONCOUNTERS_CAVITY_56_PRODUCED := 1801,
	PRODUCTIONCOUNTERS_CAVITY_56_STACKED := 1802,
	PRODUCTIONCOUNTERS_CAVITY_56_REJECTED := 1803,
	PRODUCTIONCOUNTERS_CAVITY_56_UNCOUNTEDREJECT := 1804,
	PRODUCTIONCOUNTERS_CAVITY_56_REJECTREASON_0 := 1805,
	PRODUCTIONCOUNTERS_CAVITY_56_REJECTREASON_1 := 1806,
	PRODUCTIONCOUNTERS_CAVITY_56_REJECTREASON_2 := 1807,
	PRODUCTIONCOUNTERS_CAVITY_56_REJECTREASON_3 := 1808,
	PRODUCTIONCOUNTERS_CAVITY_56_REJECTREASON_4 := 1809,
	PRODUCTIONCOUNTERS_CAVITY_56_REJECTREASON_5 := 1810,
	PRODUCTIONCOUNTERS_CAVITY_56_REJECTREASON_6 := 1811,
	PRODUCTIONCOUNTERS_CAVITY_56_REJECTREASON_7 := 1812,
	PRODUCTIONCOUNTERS_CAVITY_56_REJECTREASON_8 := 1813,
	PRODUCTIONCOUNTERS_CAVITY_56_REJECTREASON_9 := 1814,
	PRODUCTIONCOUNTERS_CAVITY_56_REJECTREASON_10 := 1815,
	PRODUCTIONCOUNTERS_CAVITY_56_REJECTREASON_11 := 1816,
	PRODUCTIONCOUNTERS_CAVITY_56_REJECTREASON_12 := 1817,
	PRODUCTIONCOUNTERS_CAVITY_56_REJECTREASON_13 := 1818,
	PRODUCTIONCOUNTERS_CAVITY_56_REJECTREASON_14 := 1819,
	PRODUCTIONCOUNTERS_CAVITY_56_REJECTREASON_15 := 1820,
	PRODUCTIONCOUNTERS_CAVITY_56_REJECTREASON_16 := 1821,
	PRODUCTIONCOUNTERS_CAVITY_56_REJECTREASON_17 := 1822,
	PRODUCTIONCOUNTERS_CAVITY_56_REJECTREASON_18 := 1823,
	PRODUCTIONCOUNTERS_CAVITY_56_REJECTREASON_19 := 1824,
	PRODUCTIONCOUNTERS_CAVITY_56_REJECTREASON_20 := 1825,
	MOULDMEASUREMENT_CAVITY_56_PEAKPRESSURE := 1826,
	MOULDMEASUREMENT_HOTRUNNER_CAVITY_56_TARGETVALUE := 1827,
	MOULDMEASUREMENT_HOTRUNNER_CAVITY_56_ACTUALVALUE := 1828,
	PRODUCTIONCOUNTERS_CAVITY_57_PRODUCED := 1829,
	PRODUCTIONCOUNTERS_CAVITY_57_STACKED := 1830,
	PRODUCTIONCOUNTERS_CAVITY_57_REJECTED := 1831,
	PRODUCTIONCOUNTERS_CAVITY_57_UNCOUNTEDREJECT := 1832,
	PRODUCTIONCOUNTERS_CAVITY_57_REJECTREASON_0 := 1833,
	PRODUCTIONCOUNTERS_CAVITY_57_REJECTREASON_1 := 1834,
	PRODUCTIONCOUNTERS_CAVITY_57_REJECTREASON_2 := 1835,
	PRODUCTIONCOUNTERS_CAVITY_57_REJECTREASON_3 := 1836,
	PRODUCTIONCOUNTERS_CAVITY_57_REJECTREASON_4 := 1837,
	PRODUCTIONCOUNTERS_CAVITY_57_REJECTREASON_5 := 1838,
	PRODUCTIONCOUNTERS_CAVITY_57_REJECTREASON_6 := 1839,
	PRODUCTIONCOUNTERS_CAVITY_57_REJECTREASON_7 := 1840,
	PRODUCTIONCOUNTERS_CAVITY_57_REJECTREASON_8 := 1841,
	PRODUCTIONCOUNTERS_CAVITY_57_REJECTREASON_9 := 1842,
	PRODUCTIONCOUNTERS_CAVITY_57_REJECTREASON_10 := 1843,
	PRODUCTIONCOUNTERS_CAVITY_57_REJECTREASON_11 := 1844,
	PRODUCTIONCOUNTERS_CAVITY_57_REJECTREASON_12 := 1845,
	PRODUCTIONCOUNTERS_CAVITY_57_REJECTREASON_13 := 1846,
	PRODUCTIONCOUNTERS_CAVITY_57_REJECTREASON_14 := 1847,
	PRODUCTIONCOUNTERS_CAVITY_57_REJECTREASON_15 := 1848,
	PRODUCTIONCOUNTERS_CAVITY_57_REJECTREASON_16 := 1849,
	PRODUCTIONCOUNTERS_CAVITY_57_REJECTREASON_17 := 1850,
	PRODUCTIONCOUNTERS_CAVITY_57_REJECTREASON_18 := 1851,
	PRODUCTIONCOUNTERS_CAVITY_57_REJECTREASON_19 := 1852,
	PRODUCTIONCOUNTERS_CAVITY_57_REJECTREASON_20 := 1853,
	MOULDMEASUREMENT_CAVITY_57_PEAKPRESSURE := 1854,
	MOULDMEASUREMENT_HOTRUNNER_CAVITY_57_TARGETVALUE := 1855,
	MOULDMEASUREMENT_HOTRUNNER_CAVITY_57_ACTUALVALUE := 1856,
	PRODUCTIONCOUNTERS_CAVITY_58_PRODUCED := 1857,
	PRODUCTIONCOUNTERS_CAVITY_58_STACKED := 1858,
	PRODUCTIONCOUNTERS_CAVITY_58_REJECTED := 1859,
	PRODUCTIONCOUNTERS_CAVITY_58_UNCOUNTEDREJECT := 1860,
	PRODUCTIONCOUNTERS_CAVITY_58_REJECTREASON_0 := 1861,
	PRODUCTIONCOUNTERS_CAVITY_58_REJECTREASON_1 := 1862,
	PRODUCTIONCOUNTERS_CAVITY_58_REJECTREASON_2 := 1863,
	PRODUCTIONCOUNTERS_CAVITY_58_REJECTREASON_3 := 1864,
	PRODUCTIONCOUNTERS_CAVITY_58_REJECTREASON_4 := 1865,
	PRODUCTIONCOUNTERS_CAVITY_58_REJECTREASON_5 := 1866,
	PRODUCTIONCOUNTERS_CAVITY_58_REJECTREASON_6 := 1867,
	PRODUCTIONCOUNTERS_CAVITY_58_REJECTREASON_7 := 1868,
	PRODUCTIONCOUNTERS_CAVITY_58_REJECTREASON_8 := 1869,
	PRODUCTIONCOUNTERS_CAVITY_58_REJECTREASON_9 := 1870,
	PRODUCTIONCOUNTERS_CAVITY_58_REJECTREASON_10 := 1871,
	PRODUCTIONCOUNTERS_CAVITY_58_REJECTREASON_11 := 1872,
	PRODUCTIONCOUNTERS_CAVITY_58_REJECTREASON_12 := 1873,
	PRODUCTIONCOUNTERS_CAVITY_58_REJECTREASON_13 := 1874,
	PRODUCTIONCOUNTERS_CAVITY_58_REJECTREASON_14 := 1875,
	PRODUCTIONCOUNTERS_CAVITY_58_REJECTREASON_15 := 1876,
	PRODUCTIONCOUNTERS_CAVITY_58_REJECTREASON_16 := 1877,
	PRODUCTIONCOUNTERS_CAVITY_58_REJECTREASON_17 := 1878,
	PRODUCTIONCOUNTERS_CAVITY_58_REJECTREASON_18 := 1879,
	PRODUCTIONCOUNTERS_CAVITY_58_REJECTREASON_19 := 1880,
	PRODUCTIONCOUNTERS_CAVITY_58_REJECTREASON_20 := 1881,
	MOULDMEASUREMENT_CAVITY_58_PEAKPRESSURE := 1882,
	MOULDMEASUREMENT_HOTRUNNER_CAVITY_58_TARGETVALUE := 1883,
	MOULDMEASUREMENT_HOTRUNNER_CAVITY_58_ACTUALVALUE := 1884,
	PRODUCTIONCOUNTERS_CAVITY_59_PRODUCED := 1885,
	PRODUCTIONCOUNTERS_CAVITY_59_STACKED := 1886,
	PRODUCTIONCOUNTERS_CAVITY_59_REJECTED := 1887,
	PRODUCTIONCOUNTERS_CAVITY_59_UNCOUNTEDREJECT := 1888,
	PRODUCTIONCOUNTERS_CAVITY_59_REJECTREASON_0 := 1889,
	PRODUCTIONCOUNTERS_CAVITY_59_REJECTREASON_1 := 1890,
	PRODUCTIONCOUNTERS_CAVITY_59_REJECTREASON_2 := 1891,
	PRODUCTIONCOUNTERS_CAVITY_59_REJECTREASON_3 := 1892,
	PRODUCTIONCOUNTERS_CAVITY_59_REJECTREASON_4 := 1893,
	PRODUCTIONCOUNTERS_CAVITY_59_REJECTREASON_5 := 1894,
	PRODUCTIONCOUNTERS_CAVITY_59_REJECTREASON_6 := 1895,
	PRODUCTIONCOUNTERS_CAVITY_59_REJECTREASON_7 := 1896,
	PRODUCTIONCOUNTERS_CAVITY_59_REJECTREASON_8 := 1897,
	PRODUCTIONCOUNTERS_CAVITY_59_REJECTREASON_9 := 1898,
	PRODUCTIONCOUNTERS_CAVITY_59_REJECTREASON_10 := 1899,
	PRODUCTIONCOUNTERS_CAVITY_59_REJECTREASON_11 := 1900,
	PRODUCTIONCOUNTERS_CAVITY_59_REJECTREASON_12 := 1901,
	PRODUCTIONCOUNTERS_CAVITY_59_REJECTREASON_13 := 1902,
	PRODUCTIONCOUNTERS_CAVITY_59_REJECTREASON_14 := 1903,
	PRODUCTIONCOUNTERS_CAVITY_59_REJECTREASON_15 := 1904,
	PRODUCTIONCOUNTERS_CAVITY_59_REJECTREASON_16 := 1905,
	PRODUCTIONCOUNTERS_CAVITY_59_REJECTREASON_17 := 1906,
	PRODUCTIONCOUNTERS_CAVITY_59_REJECTREASON_18 := 1907,
	PRODUCTIONCOUNTERS_CAVITY_59_REJECTREASON_19 := 1908,
	PRODUCTIONCOUNTERS_CAVITY_59_REJECTREASON_20 := 1909,
	MOULDMEASUREMENT_CAVITY_59_PEAKPRESSURE := 1910,
	MOULDMEASUREMENT_HOTRUNNER_CAVITY_59_TARGETVALUE := 1911,
	MOULDMEASUREMENT_HOTRUNNER_CAVITY_59_ACTUALVALUE := 1912,
	PRODUCTIONCOUNTERS_CAVITY_60_PRODUCED := 1913,
	PRODUCTIONCOUNTERS_CAVITY_60_STACKED := 1914,
	PRODUCTIONCOUNTERS_CAVITY_60_REJECTED := 1915,
	PRODUCTIONCOUNTERS_CAVITY_60_UNCOUNTEDREJECT := 1916,
	PRODUCTIONCOUNTERS_CAVITY_60_REJECTREASON_0 := 1917,
	PRODUCTIONCOUNTERS_CAVITY_60_REJECTREASON_1 := 1918,
	PRODUCTIONCOUNTERS_CAVITY_60_REJECTREASON_2 := 1919,
	PRODUCTIONCOUNTERS_CAVITY_60_REJECTREASON_3 := 1920,
	PRODUCTIONCOUNTERS_CAVITY_60_REJECTREASON_4 := 1921,
	PRODUCTIONCOUNTERS_CAVITY_60_REJECTREASON_5 := 1922,
	PRODUCTIONCOUNTERS_CAVITY_60_REJECTREASON_6 := 1923,
	PRODUCTIONCOUNTERS_CAVITY_60_REJECTREASON_7 := 1924,
	PRODUCTIONCOUNTERS_CAVITY_60_REJECTREASON_8 := 1925,
	PRODUCTIONCOUNTERS_CAVITY_60_REJECTREASON_9 := 1926,
	PRODUCTIONCOUNTERS_CAVITY_60_REJECTREASON_10 := 1927,
	PRODUCTIONCOUNTERS_CAVITY_60_REJECTREASON_11 := 1928,
	PRODUCTIONCOUNTERS_CAVITY_60_REJECTREASON_12 := 1929,
	PRODUCTIONCOUNTERS_CAVITY_60_REJECTREASON_13 := 1930,
	PRODUCTIONCOUNTERS_CAVITY_60_REJECTREASON_14 := 1931,
	PRODUCTIONCOUNTERS_CAVITY_60_REJECTREASON_15 := 1932,
	PRODUCTIONCOUNTERS_CAVITY_60_REJECTREASON_16 := 1933,
	PRODUCTIONCOUNTERS_CAVITY_60_REJECTREASON_17 := 1934,
	PRODUCTIONCOUNTERS_CAVITY_60_REJECTREASON_18 := 1935,
	PRODUCTIONCOUNTERS_CAVITY_60_REJECTREASON_19 := 1936,
	PRODUCTIONCOUNTERS_CAVITY_60_REJECTREASON_20 := 1937,
	MOULDMEASUREMENT_CAVITY_60_PEAKPRESSURE := 1938,
	MOULDMEASUREMENT_HOTRUNNER_CAVITY_60_TARGETVALUE := 1939,
	MOULDMEASUREMENT_HOTRUNNER_CAVITY_60_ACTUALVALUE := 1940,
	PRODUCTIONCOUNTERS_CAVITY_61_PRODUCED := 1941,
	PRODUCTIONCOUNTERS_CAVITY_61_STACKED := 1942,
	PRODUCTIONCOUNTERS_CAVITY_61_REJECTED := 1943,
	PRODUCTIONCOUNTERS_CAVITY_61_UNCOUNTEDREJECT := 1944,
	PRODUCTIONCOUNTERS_CAVITY_61_REJECTREASON_0 := 1945,
	PRODUCTIONCOUNTERS_CAVITY_61_REJECTREASON_1 := 1946,
	PRODUCTIONCOUNTERS_CAVITY_61_REJECTREASON_2 := 1947,
	PRODUCTIONCOUNTERS_CAVITY_61_REJECTREASON_3 := 1948,
	PRODUCTIONCOUNTERS_CAVITY_61_REJECTREASON_4 := 1949,
	PRODUCTIONCOUNTERS_CAVITY_61_REJECTREASON_5 := 1950,
	PRODUCTIONCOUNTERS_CAVITY_61_REJECTREASON_6 := 1951,
	PRODUCTIONCOUNTERS_CAVITY_61_REJECTREASON_7 := 1952,
	PRODUCTIONCOUNTERS_CAVITY_61_REJECTREASON_8 := 1953,
	PRODUCTIONCOUNTERS_CAVITY_61_REJECTREASON_9 := 1954,
	PRODUCTIONCOUNTERS_CAVITY_61_REJECTREASON_10 := 1955,
	PRODUCTIONCOUNTERS_CAVITY_61_REJECTREASON_11 := 1956,
	PRODUCTIONCOUNTERS_CAVITY_61_REJECTREASON_12 := 1957,
	PRODUCTIONCOUNTERS_CAVITY_61_REJECTREASON_13 := 1958,
	PRODUCTIONCOUNTERS_CAVITY_61_REJECTREASON_14 := 1959,
	PRODUCTIONCOUNTERS_CAVITY_61_REJECTREASON_15 := 1960,
	PRODUCTIONCOUNTERS_CAVITY_61_REJECTREASON_16 := 1961,
	PRODUCTIONCOUNTERS_CAVITY_61_REJECTREASON_17 := 1962,
	PRODUCTIONCOUNTERS_CAVITY_61_REJECTREASON_18 := 1963,
	PRODUCTIONCOUNTERS_CAVITY_61_REJECTREASON_19 := 1964,
	PRODUCTIONCOUNTERS_CAVITY_61_REJECTREASON_20 := 1965,
	MOULDMEASUREMENT_CAVITY_61_PEAKPRESSURE := 1966,
	MOULDMEASUREMENT_HOTRUNNER_CAVITY_61_TARGETVALUE := 1967,
	MOULDMEASUREMENT_HOTRUNNER_CAVITY_61_ACTUALVALUE := 1968,
	PRODUCTIONCOUNTERS_CAVITY_62_PRODUCED := 1969,
	PRODUCTIONCOUNTERS_CAVITY_62_STACKED := 1970,
	PRODUCTIONCOUNTERS_CAVITY_62_REJECTED := 1971,
	PRODUCTIONCOUNTERS_CAVITY_62_UNCOUNTEDREJECT := 1972,
	PRODUCTIONCOUNTERS_CAVITY_62_REJECTREASON_0 := 1973,
	PRODUCTIONCOUNTERS_CAVITY_62_REJECTREASON_1 := 1974,
	PRODUCTIONCOUNTERS_CAVITY_62_REJECTREASON_2 := 1975,
	PRODUCTIONCOUNTERS_CAVITY_62_REJECTREASON_3 := 1976,
	PRODUCTIONCOUNTERS_CAVITY_62_REJECTREASON_4 := 1977,
	PRODUCTIONCOUNTERS_CAVITY_62_REJECTREASON_5 := 1978,
	PRODUCTIONCOUNTERS_CAVITY_62_REJECTREASON_6 := 1979,
	PRODUCTIONCOUNTERS_CAVITY_62_REJECTREASON_7 := 1980,
	PRODUCTIONCOUNTERS_CAVITY_62_REJECTREASON_8 := 1981,
	PRODUCTIONCOUNTERS_CAVITY_62_REJECTREASON_9 := 1982,
	PRODUCTIONCOUNTERS_CAVITY_62_REJECTREASON_10 := 1983,
	PRODUCTIONCOUNTERS_CAVITY_62_REJECTREASON_11 := 1984,
	PRODUCTIONCOUNTERS_CAVITY_62_REJECTREASON_12 := 1985,
	PRODUCTIONCOUNTERS_CAVITY_62_REJECTREASON_13 := 1986,
	PRODUCTIONCOUNTERS_CAVITY_62_REJECTREASON_14 := 1987,
	PRODUCTIONCOUNTERS_CAVITY_62_REJECTREASON_15 := 1988,
	PRODUCTIONCOUNTERS_CAVITY_62_REJECTREASON_16 := 1989,
	PRODUCTIONCOUNTERS_CAVITY_62_REJECTREASON_17 := 1990,
	PRODUCTIONCOUNTERS_CAVITY_62_REJECTREASON_18 := 1991,
	PRODUCTIONCOUNTERS_CAVITY_62_REJECTREASON_19 := 1992,
	PRODUCTIONCOUNTERS_CAVITY_62_REJECTREASON_20 := 1993,
	MOULDMEASUREMENT_CAVITY_62_PEAKPRESSURE := 1994,
	MOULDMEASUREMENT_HOTRUNNER_CAVITY_62_TARGETVALUE := 1995,
	MOULDMEASUREMENT_HOTRUNNER_CAVITY_62_ACTUALVALUE := 1996,
	PRODUCTIONCOUNTERS_CAVITY_63_PRODUCED := 1997,
	PRODUCTIONCOUNTERS_CAVITY_63_STACKED := 1998,
	PRODUCTIONCOUNTERS_CAVITY_63_REJECTED := 1999,
	PRODUCTIONCOUNTERS_CAVITY_63_UNCOUNTEDREJECT := 2000,
	PRODUCTIONCOUNTERS_CAVITY_63_REJECTREASON_0 := 2001,
	PRODUCTIONCOUNTERS_CAVITY_63_REJECTREASON_1 := 2002,
	PRODUCTIONCOUNTERS_CAVITY_63_REJECTREASON_2 := 2003,
	PRODUCTIONCOUNTERS_CAVITY_63_REJECTREASON_3 := 2004,
	PRODUCTIONCOUNTERS_CAVITY_63_REJECTREASON_4 := 2005,
	PRODUCTIONCOUNTERS_CAVITY_63_REJECTREASON_5 := 2006,
	PRODUCTIONCOUNTERS_CAVITY_63_REJECTREASON_6 := 2007,
	PRODUCTIONCOUNTERS_CAVITY_63_REJECTREASON_7 := 2008,
	PRODUCTIONCOUNTERS_CAVITY_63_REJECTREASON_8 := 2009,
	PRODUCTIONCOUNTERS_CAVITY_63_REJECTREASON_9 := 2010,
	PRODUCTIONCOUNTERS_CAVITY_63_REJECTREASON_10 := 2011,
	PRODUCTIONCOUNTERS_CAVITY_63_REJECTREASON_11 := 2012,
	PRODUCTIONCOUNTERS_CAVITY_63_REJECTREASON_12 := 2013,
	PRODUCTIONCOUNTERS_CAVITY_63_REJECTREASON_13 := 2014,
	PRODUCTIONCOUNTERS_CAVITY_63_REJECTREASON_14 := 2015,
	PRODUCTIONCOUNTERS_CAVITY_63_REJECTREASON_15 := 2016,
	PRODUCTIONCOUNTERS_CAVITY_63_REJECTREASON_16 := 2017,
	PRODUCTIONCOUNTERS_CAVITY_63_REJECTREASON_17 := 2018,
	PRODUCTIONCOUNTERS_CAVITY_63_REJECTREASON_18 := 2019,
	PRODUCTIONCOUNTERS_CAVITY_63_REJECTREASON_19 := 2020,
	PRODUCTIONCOUNTERS_CAVITY_63_REJECTREASON_20 := 2021,
	MOULDMEASUREMENT_CAVITY_63_PEAKPRESSURE := 2022,
	MOULDMEASUREMENT_HOTRUNNER_CAVITY_63_TARGETVALUE := 2023,
	MOULDMEASUREMENT_HOTRUNNER_CAVITY_63_ACTUALVALUE := 2024,
	PRODUCTIONCOUNTERS_CAVITY_64_PRODUCED := 2025,
	PRODUCTIONCOUNTERS_CAVITY_64_STACKED := 2026,
	PRODUCTIONCOUNTERS_CAVITY_64_REJECTED := 2027,
	PRODUCTIONCOUNTERS_CAVITY_64_UNCOUNTEDREJECT := 2028,
	PRODUCTIONCOUNTERS_CAVITY_64_REJECTREASON_0 := 2029,
	PRODUCTIONCOUNTERS_CAVITY_64_REJECTREASON_1 := 2030,
	PRODUCTIONCOUNTERS_CAVITY_64_REJECTREASON_2 := 2031,
	PRODUCTIONCOUNTERS_CAVITY_64_REJECTREASON_3 := 2032,
	PRODUCTIONCOUNTERS_CAVITY_64_REJECTREASON_4 := 2033,
	PRODUCTIONCOUNTERS_CAVITY_64_REJECTREASON_5 := 2034,
	PRODUCTIONCOUNTERS_CAVITY_64_REJECTREASON_6 := 2035,
	PRODUCTIONCOUNTERS_CAVITY_64_REJECTREASON_7 := 2036,
	PRODUCTIONCOUNTERS_CAVITY_64_REJECTREASON_8 := 2037,
	PRODUCTIONCOUNTERS_CAVITY_64_REJECTREASON_9 := 2038,
	PRODUCTIONCOUNTERS_CAVITY_64_REJECTREASON_10 := 2039,
	PRODUCTIONCOUNTERS_CAVITY_64_REJECTREASON_11 := 2040,
	PRODUCTIONCOUNTERS_CAVITY_64_REJECTREASON_12 := 2041,
	PRODUCTIONCOUNTERS_CAVITY_64_REJECTREASON_13 := 2042,
	PRODUCTIONCOUNTERS_CAVITY_64_REJECTREASON_14 := 2043,
	PRODUCTIONCOUNTERS_CAVITY_64_REJECTREASON_15 := 2044,
	PRODUCTIONCOUNTERS_CAVITY_64_REJECTREASON_16 := 2045,
	PRODUCTIONCOUNTERS_CAVITY_64_REJECTREASON_17 := 2046,
	PRODUCTIONCOUNTERS_CAVITY_64_REJECTREASON_18 := 2047,
	PRODUCTIONCOUNTERS_CAVITY_64_REJECTREASON_19 := 2048,
	PRODUCTIONCOUNTERS_CAVITY_64_REJECTREASON_20 := 2049,
	MOULDMEASUREMENT_CAVITY_64_PEAKPRESSURE := 2050,
	MOULDMEASUREMENT_HOTRUNNER_CAVITY_64_TARGETVALUE := 2051,
	MOULDMEASUREMENT_HOTRUNNER_CAVITY_64_ACTUALVALUE := 2052,
	CYCLETIMES_TARGETCYCLETIME := 2053,
	MAGAZINE_SENSORTIMES_VACUUM_5 := 2054,
	MAGAZINE_SENSORTIMES_VACUUM_6 := 2055,
	MAGAZINE_SENSORTIMES_VACUUM_7 := 2056,
	MAGAZINE_SENSORTIMES_VACUUM_8 := 2057,
	BOXCONVEYOR_ALARMS := 2058,
	FANUC_ALARMS := 2059,
	MAGAZINE_SENSORTIMES_ROTATEIN := 2060,
	MAGAZINE_SENSORTIMES_ROTATEOUT := 2061,
	MAGAZINE_SENSORTIMES_SHIFTIN := 2062,
	MAGAZINE_SENSORTIMES_SHIFTOUT := 2063,
	YUNIT_BFU_COVEREDDISTANCE := 2064,
	ZUNIT_BFU_COVEREDDISTANCE := 2065,
	ZUNIT_BFU_ERRORID := 2066,
	YUNIT_BFU_ERRORID := 2067,
	ZUNIT_BFU_AXISERRORID := 2068,
	YUNIT_BFU_AXISERRORID := 2069,
	ZUNIT_BFU_DRIVEUTILISATION := 2070,
	YUNIT_BFU_DRIVEUTILISATION := 2071,
	YUNIT_BFU_MOTORUTILISATION := 2072,
	ZUNIT_BFU_MOTORUTILISATION := 2073,
	YUNIT_BFU_ALARMS := 2074,
	ZUNIT_BFU_ALARMS := 2075,
	BOXCONVEYOR_SENSORTIMES_LIFTIN := 2076,
	BOXCONVEYOR_SENSORTIMES_LIFTOUT := 2077,
	BOXCONVEYOR_SENSORTIMES_OPENBOXLONGSIDEIN := 2078,
	BOXCONVEYOR_SENSORTIMES_OPENBOXLONGSIDEOUT := 2079,
	BOXCONVEYOR_SENSORTIMES_OPENBOXSHORTSIDEIN := 2080,
	BOXCONVEYOR_SENSORTIMES_OPENBOXSHORTSIDEOUT := 2081,
	BFU_PICKANDPLACE_SENSORTIMES_CLAMPIN := 2082,
	BFU_PICKANDPLACE_SENSORTIMES_CLAMPOUT := 2083,
	BFU_PICKANDPLACE_SENSORTIMES_PATTERNIZERPUSHERIN := 2084,
	BFU_PICKANDPLACE_SENSORTIMES_PATTERNIZERPUSHEROUT := 2085,
	BFU_PICKANDPLACE_SENSORTIMES_PATTERNIZEREXTENDIN := 2086,
	BFU_PICKANDPLACE_SENSORTIMES_PATTERNIZEREXTENDOUT := 2087,
	YUNIT_BFU_DRIVEERRORID := 2088,
	ZUNIT_BFU_DRIVEERRORID := 2089,
	BFU_PICKANDPLACE_ALARMS := 2090,
	BOXCONVEYOR_SENSORTIMES_CLAMPSECONDBOXOUT := 2091,
	BOXCONVEYOR_SENSORTIMES_CLAMPSECONDBOXIN := 2092,
	BOXCONVEYOR_SENSORTIMES_BOXSTOPPEROUT := 2093,
	BOXCONVEYOR_SENSORTIMES_BOXSTOPPERIN := 2094,
	CONVEYORS_BFU_DRIVEUTILISATION := 2095,
	CONVEYORS_BFU_MOTORUTILISATION := 2096,
	CONVEYORS_BFU_DRIVEERRORID := 2097,
	CONVEYORS_BFU_AXISERRORID := 2098,
	CONVEYORS_BFU_ERRORID := 2099,
	CONVEYORS_BFU_COVEREDDISTANCE := 2100,
	MAGAZINE_ACTIVEDRAWER := 2101,
	MAIN_PRODUCTWEIGHT := 2102,
	PATTERNIZER_ALARMS := 2103,
	OUTFEEDTRANSFER_ALARMS := 2104,
	CAMERA_YUNIT_ALARMS := 2105,
	ZUNIT_SENSORTIMES_EXTEND1OUT := 2106,
	ZUNIT_SENSORTIMES_EXTEND2OUT := 2107,
	ZUNIT_SENSORTIMES_EXTEND3OUT := 2108,
	ZUNIT_SENSORTIMES_EXTEND4OUT := 2109,
	ZUNIT_SENSORTIMES_BLOCKSTACKIN := 2110,
	ZUNIT_SENSORTIMES_BLOCKSTACKOUT := 2111,
	CAMERA_2_ALARMS := 2112,
	CAMERA_2_TIME_ACTIVE := 2113,
	CAMERA_2_TIME_IDLE := 2114,
	Z1UNIT_ALARMS := 2115,
	Z2UNIT_ALARMS := 2116,
	ZRUNIT_ZR1_ALARMS := 2117,
	HMU_ALARMS := 2118,
	ZRUNIT_ZR2_ALARMS := 2119,
	PRUNIT_ALARMS := 2120,
	LUNIT_ALARMS := 2121,
	MAGAZINE_COVEREDDISTANCE := 2122,
	Z1UNIT_COVEREDDISTANCE := 2123,
	PRUNIT_COVEREDDISTANCE := 2124,
	Z2UNIT_COVEREDDISTANCE := 2125,
	LUNIT_L1_COVEREDDISTANCE := 2126,
	LUNIT_L2_COVEREDDISTANCE := 2127,
	LUNIT_L3_COVEREDDISTANCE := 2128,
	LUNIT_L4_COVEREDDISTANCE := 2129,
	MAGAZINE_ERRORID := 2130,
	Z1UNIT_ERRORID := 2131,
	PRUNIT_ERRORID := 2132,
	Z2UNIT_ERRORID := 2133,
	LUNIT_L1_ERRORID := 2134,
	LUNIT_L2_ERRORID := 2135,
	LUNIT_L3_ERRORID := 2136,
	LUNIT_L4_ERRORID := 2137,
	ZRUNIT_ZR3_ALARMS := 2138,
	ZRUNIT_ZR4_ALARMS := 2139,
	MAGAZINE_AXISERRORID := 2140,
	Z1UNIT_AXISERRORID := 2141,
	ZRUNIT_ZR1_AXISERRORID := 2142,
	ZRUNIT_ZR2_AXISERRORID := 2143,
	ZRUNIT_ZR3_AXISERRORID := 2144,
	ZRUNIT_ZR4_AXISERRORID := 2145,
	PRUNIT_AXISERRORID := 2146,
	Z2UNIT_AXISERRORID := 2147,
	LUNIT_L1_AXISERRORID := 2148,
	LUNIT_L2_AXISERRORID := 2149,
	LUNIT_L3_AXISERRORID := 2150,
	LUNIT_L4_AXISERRORID := 2151,
	MAGAZINE_DRIVEERRORID := 2152,
	Z1UNIT_DRIVEERRORID := 2153,
	ZRUNIT_ZR1_DRIVEERRORID := 2154,
	ZRUNIT_ZR2_DRIVEERRORID := 2155,
	ZRUNIT_ZR3_DRIVEERRORID := 2156,
	ZRUNIT_ZR4_DRIVEERRORID := 2157,
	PRUNIT_DRIVEERRORID := 2158,
	Z2UNIT_DRIVEERRORID := 2159,
	LUNIT_L1_DRIVEERRORID := 2160,
	LUNIT_L2_DRIVEERRORID := 2161,
	LUNIT_L3_DRIVEERRORID := 2162,
	LUNIT_L4_DRIVEERRORID := 2163,
	MAGAZINE_DRIVEUTILISATION := 2164,
	Z1UNIT_DRIVEUTILISATION := 2165,
	PRUNIT_DRIVEUTILISATION := 2166,
	Z2UNIT_DRIVEUTILISATION := 2167,
	LUNIT_L1_DRIVEUTILISATION := 2168,
	LUNIT_L2_DRIVEUTILISATION := 2169,
	LUNIT_L3_DRIVEUTILISATION := 2170,
	LUNIT_L4_DRIVEUTILISATION := 2171,
	MAGAZINE_MOTORUTILISATION := 2172,
	Z1UNIT_MOTORUTILISATION := 2173,
	PRUNIT_MOTORUTILISATION := 2174,
	Z2UNIT_MOTORUTILISATION := 2175,
	LUNIT_L1_MOTORUTILISATION := 2176,
	LUNIT_L2_MOTORUTILISATION := 2177,
	LUNIT_L3_MOTORUTILISATION := 2178,
	LUNIT_L4_MOTORUTILISATION := 2179,
	MAGAZINE_SENSORTIMES_EXTENDIN := 2180,
	MAGAZINE_SENSORTIMES_EXTENDOUT := 2181,
	HMU_SENSORTIMES_FIXEDBUFFERIN := 2182,
	HMU_SENSORTIMES_FIXEDBUFFEROUT := 2183,
	HMU_SENSORTIMES_MOVINGBUFFERIN := 2184,
	HMU_SENSORTIMES_MOVINGBUFFEROUT := 2185,
	HMU_SENSORTIMES_BUFFERUPDOWNIN := 2186,
	HMU_SENSORTIMES_BUFFERUPDOWNOUT := 2187,
	HMU_SENSORTIMES_LOCKCYLINDERIN := 2188,
	HMU_SENSORTIMES_LOCKCYLINDEROUT := 2189,
	CHAIN_SENSORTIMES_VACUUM_1 := 2190,
	CHAIN_SENSORTIMES_VACUUM_2 := 2191,
	CHAIN_SENSORTIMES_VACUUM_3 := 2192,
	CHAIN_SENSORTIMES_VACUUM_4 := 2193,
	CHAIN_SENSORTIMES_EXTENDIN := 2194,
	CHAIN_SENSORTIMES_EXTENDOUT := 2195,
	Z2UNIT_SENSORTIMES_VACUUM_1 := 2196,
	Z2UNIT_SENSORTIMES_VACUUM_2 := 2197,
	Z2UNIT_SENSORTIMES_VACUUM_3 := 2198,
	Z2UNIT_SENSORTIMES_VACUUM_4 := 2199,
	Z2UNIT_SENSORTIMES_REJECTVACUUM_1 := 2200,
	Z2UNIT_SENSORTIMES_REJECTVACUUM_2 := 2201,
	Z2UNIT_SENSORTIMES_REJECTVACUUM_3 := 2202,
	Z2UNIT_SENSORTIMES_REJECTVACUUM_4 := 2203,
	MAGAZINE_TIME_IDLE := 2204,
	HMU_TIME_IDLE := 2205,
	Z1UNIT_TIME_IDLE := 2206,
	PRUNIT_TIME_IDLE := 2207,
	Z2UNIT_TIME_IDLE := 2208,
	LUNIT_L1_TIME_IDLE := 2209,
	LUNIT_L2_TIME_IDLE := 2210,
	LUNIT_L3_TIME_IDLE := 2211,
	LUNIT_L4_TIME_IDLE := 2212,
	CONVEYORS_C1_TIME_IDLE := 2213,
	CONVEYORS_C2_TIME_IDLE := 2214,
	CONVEYORS_C3_TIME_IDLE := 2215,
	CONVEYORS_C4_TIME_IDLE := 2216,
	MAGAZINE_TIME_ACTIVE := 2217,
	HMU_TIME_ACTIVE := 2218,
	Z1UNIT_TIME_ACTIVE := 2219,
	PRUNIT_TIME_ACTIVE := 2220,
	Z2UNIT_TIME_ACTIVE := 2221,
	LUNIT_L1_TIME_ACTIVE := 2222,
	LUNIT_L2_TIME_ACTIVE := 2223,
	LUNIT_L3_TIME_ACTIVE := 2224,
	LUNIT_L4_TIME_ACTIVE := 2225,
	CONVEYORS_C1_TIME_ACTIVE := 2226,
	CONVEYORS_C2_TIME_ACTIVE := 2227,
	CONVEYORS_C3_TIME_ACTIVE := 2228,
	CONVEYORS_C4_TIME_ACTIVE := 2229,
	CONVEYORS_C2_ALARMS := 2230,
	CONVEYORS_C3_ALARMS := 2231,
	CONVEYORS_C4_ALARMS := 2232,
	LUNIT_L2_ALARMS := 2233,
	LUNIT_L3_ALARMS := 2234,
	LUNIT_L4_ALARMS := 2235,
	PRODUCTIONCOUNTERS_TOTAL_CRATESPRODUCED := 2236,
	PRODUCTIONCOUNTERS_TOTAL_RECEIVEDPATTERNS := 2237,
	PRODUCTIONCOUNTERS_TOTAL_RECEIVEDPACKABLEPATTERNS := 2238,
	PRODUCTIONCOUNTERS_TOTAL_PACKSPLACEDINCRATE := 2239,
	PRODUCTIONCOUNTERS_TOTAL_PACKSSEALED := 2240,
	PRODUCTIONCOUNTERS_TOTAL_STACKSPLACEDINPUSHER := 2241,
	DRAWERMAGAZINE_ALARMS := 2242,
	MAIN_BSF_ENABLESEALBAR := 2243,
	ILLIG_ENABLEPLACENEWPATTERN := 2244,
	ILLIG_ENABLEPLACENEWPATTERNBUSY := 2245,
	ILLIG_PACKABLEPATTERNPLACED := 2246,
	ILLIG_REQUESTPLACENEWPATTERN := 2247,
	RELAYS_MAINAIRVALVE2 := 2248,
	RELAYS_MAINAIRVALVECRATE1 := 2249,
	RELAYS_MAINAIRVALVECRATE2 := 2250,
	RELAYS_SAFETYGATECRATE1 := 2251,
	RELAYS_SAFETYGATECRATE2 := 2252,
	INFEEDCONVEYOR_STACKTOOHIGHSENSOR := 2253,
	INFEEDCONVEYOR_ALARMS := 2256,
	STACKUNIT_ALARMS := 2257,
	FANUC1_ALARMS := 2258,
	PUSHER_ALARMS := 2259,
	REJECTSTATION_BSF_ALARMS := 2260,
	SEALUNIT_FOILMAGAZINE_ALARMS := 2261,
	SEALUNIT_TRANSPORTANDSEALBAG_ALARMS := 2262,
	SEALUNIT_PREPAREANDFILLBAG_ALARMS := 2263,
	SEALUNIT_FRAME_ALARMS := 2264,
	CRATEUNIT_FANUC2_ALARMS := 2265,
	CRATEUNIT_CRATES_ALARMS := 2266,
	INFEEDCONVEYOR_COVEREDDISTANCE := 2267,
	STACKUNIT_COVEREDDISTANCE := 2268,
	PUSHER_COVEREDDISTANCE := 2269,
	SEALUNIT_FOILMAGAZINE_COVEREDDISTANCE := 2270,
	SEALUNIT_TRANSPORTANDSEALBAG_MOTOR1_COVEREDDISTANCE := 2271,
	SEALUNIT_TRANSPORTANDSEALBAG_MOTOR2_COVEREDDISTANCE := 2272,
	SEALUNIT_PREPAREANDFILLBAG_COVEREDDISTANCE := 2273,
	INFEEDCONVEYOR_ERRORID := 2274,
	STACKUNIT_ERRORID := 2275,
	PUSHER_ERRORID := 2276,
	SEALUNIT_FOILMAGAZINE_ERRORID := 2277,
	SEALUNIT_TRANSPORTANDSEALBAG_MOTOR1_ERRORID := 2278,
	SEALUNIT_TRANSPORTANDSEALBAG_MOTOR2_ERRORID := 2279,
	SEALUNIT_PREPAREANDFILLBAG_ERRORID := 2280,
	INFEEDCONVEYOR_AXISERRORID := 2281,
	STACKUNIT_AXISERRORID := 2282,
	PUSHER_AXISERRORID := 2283,
	SEALUNIT_FOILMAGAZINE_AXISERRORID := 2284,
	SEALUNIT_PREPAREANDFILLBAG_AXISERRORID := 2285,
	SEALUNIT_TRANSPORTANDSEALBAG_MOTOR1_AXISERRORID := 2286,
	SEALUNIT_TRANSPORTANDSEALBAG_MOTOR2_AXISERRORID := 2287,
	INFEEDCONVEYOR_DRIVEERRORID := 2288,
	STACKUNIT_DRIVEERRORID := 2289,
	PUSHER_DRIVEERRORID := 2290,
	SEALUNIT_FOILMAGAZINE_DRIVEERRORID := 2291,
	SEALUNIT_PREPAREANDFILLBAG_DRIVEERRORID := 2292,
	SEALUNIT_TRANSPORTANDSEALBAG_MAIN_DRIVEERRORID := 2293,
	SEALUNIT_TRANSPORTANDSEALBAG_MOTOR2_DRIVEERRORID := 2294,
	SEALUNIT_TRANSPORTANDSEALBAG_MOTOR1_DRIVEERRORID := 2295,
	INFEEDCONVEYOR_DRIVEUTILISATION := 2296,
	STACKUNIT_DRIVEUTILISATION := 2297,
	PUSHER_DRIVEUTILISATION := 2298,
	SEALUNIT_FOILMAGAZINE_DRIVEUTILISATION := 2299,
	SEALUNIT_PREPAREANDFILLBAG_DRIVEUTILISATION := 2300,
	SEALUNIT_TRANSPORTANDSEALBAG_MOTOR1_DRIVEUTILISATION := 2301,
	SEALUNIT_TRANSPORTANDSEALBAG_MOTOR2_DRIVEUTILISATION := 2302,
	INFEEDCONVEYOR_MOTORUTILISATION := 2303,
	STACKUNIT_MOTORUTILISATION := 2304,
	PUSHER_MOTORUTILISATION := 2305,
	SEALUNIT_FOILMAGAZINE_MOTORUTILISATION := 2306,
	SEALUNIT_PREPAREANDFILLBAG_MOTORUTILISATION := 2307,
	SEALUNIT_TRANSPORTANDSEALBAG_MOTOR1_MOTORUTILISATION := 2308,
	SEALUNIT_TRANSPORTANDSEALBAG_MOTOR2_MOTORUTILISATION := 2309,
	SENSORTIMES_STACKUNIT_STACKPLATE1IN := 2310,
	SENSORTIMES_STACKUNIT_STACKPLATE1OUT := 2311,
	SENSORTIMES_STACKUNIT_STACKPLATE2IN := 2312,
	SENSORTIMES_STACKUNIT_STACKPLATE2OUT := 2313,
	SENSORTIMES_STACKUNIT_BUFFERPLATE1IN := 2314,
	SENSORTIMES_STACKUNIT_BUFFERPLATE1OUT := 2315,
	SENSORTIMES_STACKUNIT_BUFFERPLATE2IN := 2316,
	SENSORTIMES_STACKUNIT_BUFFERPLATE2OUT := 2317,
	SENSORTIMES_STACKUNIT_REJECTSTACKIN := 2318,
	SENSORTIMES_STACKUNIT_REJECTSTACKOUT := 2319,
	SENSORTIMES_STACKUNIT_SHIFTSTACKUNITIN := 2320,
	SENSORTIMES_STACKUNIT_SHIFTSTACKUNITOUT := 2321,
	SENSORTIMES_FANUC1_CLAMPIN := 2322,
	SENSORTIMES_FANUC1_CLAMPOUT := 2323,
	SENSORTIMES_PUSHER_PUSHERPLATEIN := 2324,
	SENSORTIMES_PUSHER_PUSHERPLATEOUT := 2325,
	SENSORTIMES_SEALUNIT_FOILMAGAZINE_FOILROLL1_CLAMPFOILOUT := 2326,
	SENSORTIMES_SEALUNIT_FOILMAGAZINE_FOILROLL1_CLAMPFOILIN := 2327,
	SENSORTIMES_SEALUNIT_FOILMAGAZINE_FOILROLL2_CLAMPFOILOUT := 2328,
	SENSORTIMES_SEALUNIT_FOILMAGAZINE_FOILROLL2_CLAMPFOILIN := 2329,
	SENSORTIMES_SEALUNIT_FOILMAGAZINE_FOILROLL1_ENABLEFOILOUT := 2330,
	SENSORTIMES_SEALUNIT_FOILMAGAZINE_FOILROLL1_ENABLEFOILIN := 2331,
	SENSORTIMES_SEALUNIT_FOILMAGAZINE_FOILROLL2_ENABLEFOILOUT := 2332,
	SENSORTIMES_SEALUNIT_FOILMAGAZINE_FOILROLL2_ENABLEFOILIN := 2333,
	SENSORTIMES_SEALUNIT_TRANSPORTANDSEALBAG_SHIFTVACUUMBAR1IN := 2334,
	SENSORTIMES_SEALUNIT_TRANSPORTANDSEALBAG_SHIFTVACUUMBAR1OUT := 2335,
	SENSORTIMES_SEALUNIT_TRANSPORTANDSEALBAG_SHIFTVACUUMBAR2IN := 2336,
	SENSORTIMES_SEALUNIT_TRANSPORTANDSEALBAG_SHIFTVACUUMBAR2OUT := 2337,
	SENSORTIMES_SEALUNIT_TRANSPORTANDSEALBAG_EXTENDVACUUMBARIN := 2338,
	SENSORTIMES_SEALUNIT_TRANSPORTANDSEALBAG_EXTENDVACUUMBAROUT := 2339,
	SENSORTIMES_SEALUNIT_TRANSPORTANDSEALBAG_EXTENDSEALBAR1IN := 2340,
	SENSORTIMES_SEALUNIT_TRANSPORTANDSEALBAG_EXTENDSEALBAR1OUT := 2341,
	SENSORTIMES_SEALUNIT_TRANSPORTANDSEALBAG_EXTENDSEALBAR2IN := 2342,
	SENSORTIMES_SEALUNIT_TRANSPORTANDSEALBAG_EXTENDSEALBAR2OUT := 2343,
	SENSORTIMES_SEALUNIT_TRANSPORTANDSEALBAG_KNIFEIN := 2344,
	SENSORTIMES_SEALUNIT_TRANSPORTANDSEALBAG_KNIFEOUT := 2345,
	SENSORTIMES_SEALUNIT_TRANSPORTANDSEALBAG_LOCKSEALBARIN := 2346,
	SENSORTIMES_SEALUNIT_TRANSPORTANDSEALBAG_LOCKSEALBAROUT := 2347,
	SENSORTIMES_SEALUNIT_TRANSPORTANDSEALBAG_FOLDBAGSUPPORTIN := 2348,
	SENSORTIMES_SEALUNIT_TRANSPORTANDSEALBAG_FOLDBAGSUPPORTOUT := 2349,
	SENSORTIMES_SEALUNIT_PREPAREANDFILLBAG_EXTENDFORMBAGIN := 2350,
	SENSORTIMES_SEALUNIT_PREPAREANDFILLBAG_EXTENDFORMBAGOUT := 2351,
	SENSORTIMES_SEALUNIT_PREPAREANDFILLBAG_ROTATEFORMBAGIN := 2352,
	SENSORTIMES_SEALUNIT_PREPAREANDFILLBAG_ROTATEFORMBAGOUT := 2353,
	SENSORTIMES_SEALUNIT_PREPAREANDFILLBAG_ROTATEBLOWPANELIN := 2354,
	SENSORTIMES_SEALUNIT_PREPAREANDFILLBAG_ROTATEBLOWPANELOUT := 2355,
	SENSORTIMES_SEALUNIT_PREPAREANDFILLBAG_EXTENDBLOWPANELIN := 2356,
	SENSORTIMES_SEALUNIT_PREPAREANDFILLBAG_EXTENDBLOWPANELOUT := 2357,
	SENSORTIMES_SEALUNIT_PREPAREANDFILLBAG_ROTATEVACUUMUNITIN := 2358,
	SENSORTIMES_SEALUNIT_PREPAREANDFILLBAG_ROTATEVACUUMUNITOUT := 2359,
	SENSORTIMES_SEALUNIT_PREPAREANDFILLBAG_EXTENDVACUUMHEADIN := 2360,
	SENSORTIMES_SEALUNIT_PREPAREANDFILLBAG_EXTENDVACUUMHEADOUT := 2361,
	SENSORTIMES_SEALUNIT_PREPAREANDFILLBAG_FOLDUPBAGIN := 2362,
	SENSORTIMES_SEALUNIT_PREPAREANDFILLBAG_FOLDUPBAGOUT := 2363,
	SENSORTIMES_SEALUNIT_FRAME_TILTSEALUNITIN := 2364,
	SENSORTIMES_SEALUNIT_FRAME_TILTSEALUNITOUT := 2365,
	SENSORTIMES_CRATEUNIT_FANUC2_EXTENDIN := 2366,
	SENSORTIMES_CRATEUNIT_FANUC2_EXTENDOUT := 2367,
	SENSORTIMES_CRATEUNIT_FANUC2_CLAMPIN := 2368,
	SENSORTIMES_CRATEUNIT_FANUC2_CLAMPOUT := 2369,
	SENSORTIMES_CRATEUNIT_CRATES_GATECRATECOVERIN := 2370,
	SENSORTIMES_CRATEUNIT_CRATES_GATECRATECOVEROUT := 2371,
	SENSORTIMES_CRATEUNIT_CRATES_CRATE1_LIFTIN := 2372,
	SENSORTIMES_CRATEUNIT_CRATES_CRATE1_LIFTOUT := 2373,
	SENSORTIMES_CRATEUNIT_CRATES_CRATE1_BLOCKHORIZONTALIN := 2374,
	SENSORTIMES_CRATEUNIT_CRATES_CRATE1_BLOCKHORIZONTALOUT := 2375,
	SENSORTIMES_CRATEUNIT_CRATES_CRATE1_BLOCKVERTICALIN := 2376,
	SENSORTIMES_CRATEUNIT_CRATES_CRATE1_BLOCKVERTICALOUT := 2377,
	SENSORTIMES_CRATEUNIT_CRATES_CRATE2_LIFTIN := 2378,
	SENSORTIMES_CRATEUNIT_CRATES_CRATE2_LIFTOUT := 2379,
	SENSORTIMES_CRATEUNIT_CRATES_CRATE2_BLOCKHORIZONTALIN := 2380,
	SENSORTIMES_CRATEUNIT_CRATES_CRATE2_BLOCKHORIZONTALOUT := 2381,
	SENSORTIMES_CRATEUNIT_CRATES_CRATE2_BLOCKVERTICALIN := 2382,
	SENSORTIMES_CRATEUNIT_CRATES_CRATE2_BLOCKVERTICALOUT := 2383,
	INFEEDCONVEYOR_TIME_IDLE := 2384,
	STACKUNIT_TIME_IDLE := 2385,
	PUSHER_TIME_IDLE := 2386,
	SEALUNIT_FOILMAGAZINE_TIME_IDLE := 2387,
	FANUC1_TIME_IDLE := 2388,
	SEALUNIT_TRANSPORTANDSEALBAG_TIME_IDLE := 2389,
	SEALUNIT_PREPAREANDFILLBAG_TIME_IDLE := 2390,
	SEALUNIT_FRAME_TIME_IDLE := 2391,
	CRATEUNIT_FANUC2_TIME_IDLE := 2392,
	CRATEUNIT_CRATES_TIME_IDLE := 2393,
	INFEEDCONVEYOR_TIME_ACTIVE := 2394,
	STACKUNIT_TIME_ACTIVE := 2395,
	FANUC1_TIME_ACTIVE := 2396,
	PUSHER_TIME_ACTIVE := 2397,
	SEALUNIT_TRANSPORTANDSEALBAG_TIME_ACTIVE := 2398,
	SEALUNIT_FOILMAGAZINE_TIME_ACTIVE := 2399,
	SEALUNIT_PREPAREANDFILLBAG_TIME_ACTIVE := 2400,
	SEALUNIT_FRAME_TIME_ACTIVE := 2401,
	CRATEUNIT_FANUC2_TIME_ACTIVE := 2402,
	CRATEUNIT_CRATES_TIME_ACTIVE := 2403,
	SEALUNIT_TRANSPORTANDSEALBAG_SEALBARACTTEMPERATURE := 2404,
	SEALUNIT_TRANSPORTANDSEALBAG_SEALBARSETTEMPERATURE := 2405,
	SENSORTIMES_SEALUNIT_TRANSPORTANDSEALBAG_VACUUMFOIL := 2406,
	SENSORTIMES_SEALUNIT_PREPAREANDFILLBAG_VACUUMBAG := 2407,
	SEALUNIT_FOILMAGAZINE_FOILROLL1_UNROLLEDFOILLENGTH := 2408,
	SEALUNIT_FOILMAGAZINE_FOILROLL2_UNROLLEDFOILLENGTH := 2409,
	SEALUNIT_FOILMAGAZINE_FOILROLL1_TAKEFOILFAILED := 2410,
	SEALUNIT_FOILMAGAZINE_FOILROLL2_TAKEFOILFAILED := 2411,
	SEALUNIT_FOILMAGAZINE_FOILROLL1_STATE := 2412,
	SEALUNIT_FOILMAGAZINE_FOILROLL2_STATE := 2413,
	SEALUNIT_FOILMAGAZINE_FOILROLL1_ROLLSUPPORTMOTOR1 := 2414,
	SEALUNIT_FOILMAGAZINE_FOILROLL1_ROLLSUPPORTMOTOR2 := 2415,
	SEALUNIT_FOILMAGAZINE_FOILROLL2_ROLLSUPPORTMOTOR1 := 2416,
	SEALUNIT_FOILMAGAZINE_FOILROLL2_ROLLSUPPORTMOTOR2 := 2417,
	CRATEUNIT_CRATES_CRATE1_STATE := 2418,
	CRATEUNIT_CRATES_CRATE2_STATE := 2419,
	CRATEUNIT_CRATES_RECIPENAME_CRATE := 2420,
	REJECTSTATION_REJECTCOUNT := 2421,
	SEALUNIT_TRANSPORTANDSEALBAG_MOTOR1_ALARMS := 2422,
	SEALUNIT_TRANSPORTANDSEALBAG_MOTOR2_ALARMS := 2423,
	CRATEDATAPROVIDER_ALARMS := 2424,
	MAGAZINE_2_ACTIVEDRAWER := 2425,
	BFU_PICKANDPLACE_SENSORTIMES_GUIDINGIN := 2426,
	BFU_PICKANDPLACE_SENSORTIMES_GUIDINGOUT := 2427,
	BFU_PICKANDPLACE_MESSAGES := 2428,
	ZUNIT_SENSORTIMES_SHIFT2IN := 2429,
	ZUNIT_SENSORTIMES_SHIFT2OUT := 2430,
	MAIN_DCBUSVOLTAGE := 2431,
	MAIN_DCBUSVOLTAGEFILTERED := 2432,
	MAIN_RELAYS_HIGHVACUUMPUMP2RUNNING := 2433,
	RELAYS_REQUESTFOROPENINGSAFETYGATE := 2434,
	RELAYS_ACKNOWLEDGESAFETYGATES := 2435,
	Y2UNIT_ALARMS := 2436,
	XI2UNIT_ALARMS := 2437,
	XU2UNIT_ALARMS := 2438,
	MAGAZINE_2_ALARMS := 2439,
	MAGAZINE_2_M2_1_ALARMS := 2440,
	MAGAZINE_2_M2_2_ALARMS := 2441,
	SUNIT_ALARMS := 2442,
	Y3UNIT_ALARMS := 2443,
	TUNIT_ALARMS := 2444,
	AUNIT_ALARMS := 2445,
	BOXFILLSTATION_ALARMS := 2446,
	BOXINFEED_ALARMS := 2447,
	BOXOUTFEED_ALARMS := 2448,
	SHEETMAGAZINE_ALARMS := 2449,
	UPSTACKER_ALARMS := 2450,
	Y2UNIT_COVEREDDISTANCE := 2451,
	XI2UNIT_COVEREDDISTANCE := 2452,
	XU2UNIT_COVEREDDISTANCE := 2453,
	MAGAZINE_2_M2_1_COVEREDDISTANCE := 2454,
	MAGAZINE_2_M2_2_COVEREDDISTANCE := 2455,
	SUNIT_COVEREDDISTANCE := 2456,
	Y3UNIT_COVEREDDISTANCE := 2457,
	TUNIT_COVEREDDISTANCE := 2458,
	AUNIT_COVEREDDISTANCE := 2459,
	Y2UNIT_ERRORID := 2460,
	XI2UNIT_ERRORID := 2461,
	XU2UNIT_ERRORID := 2462,
	MAGAZINE_2_M2_1_ERRORID := 2463,
	MAGAZINE_2_M2_2_ERRORID := 2464,
	SUNIT_ERRORID := 2465,
	Y3UNIT_ERRORID := 2466,
	TUNIT_ERRORID := 2467,
	AUNIT_ERRORID := 2468,
	Y2UNIT_AXISERRORID := 2469,
	XI2UNIT_AXISERRORID := 2470,
	XU2UNIT_AXISERRORID := 2471,
	MAGAZINE_2_M2_1_AXISERRORID := 2472,
	MAGAZINE_2_M2_2_AXISERRORID := 2473,
	TUNIT_AXISERRORID := 2474,
	Y3UNIT_AXISERRORID := 2475,
	AUNIT_AXISERRORID := 2476,
	SUNIT_AXISERRORID := 2477,
	Y2UNIT_DRIVEERRORID := 2478,
	XI2UNIT_DRIVEERRORID := 2479,
	XU2UNIT_DRIVEERRORID := 2480,
	MAGAZINE_2_M2_1_DRIVEERRORID := 2481,
	MAGAZINE_2_M2_2_DRIVEERRORID := 2482,
	SUNIT_DRIVEERRORID := 2483,
	TUNIT_DRIVEERRORID := 2484,
	Y3UNIT_DRIVEERRORID := 2485,
	AUNIT_DRIVEERRORID := 2486,
	Y2UNIT_DRIVEUTILISATION := 2487,
	XI2UNIT_DRIVEUTILISATION := 2488,
	XU2UNIT_DRIVEUTILISATION := 2489,
	MAGAZINE_2_M2_1_DRIVEUTILISATION := 2490,
	MAGAZINE_2_M2_2_DRIVEUTILISATION := 2491,
	SUNIT_DRIVEUTILISATION := 2492,
	Y3UNIT_DRIVEUTILISATION := 2493,
	TUNIT_DRIVEUTILISATION := 2494,
	AUNIT_DRIVEUTILISATION := 2495,
	Y2UNIT_MOTORUTILISATION := 2496,
	XI2UNIT_MOTORUTILISATION := 2497,
	XU2UNIT_MOTORUTILISATION := 2498,
	MAGAZINE_2_M2_1_MOTORUTILISATION := 2499,
	MAGAZINE_2_M2_2_MOTORUTILISATION := 2500,
	TUNIT_MOTORUTILISATION := 2501,
	SUNIT_MOTORUTILISATION := 2502,
	Y3UNIT_MOTORUTILISATION := 2503,
	AUNIT_MOTORUTILISATION := 2504,
	XUUNIT_SENSORTIMES_VACUUM_4 := 2505,
	XUUNIT_SENSORTIMES_VACUUM_5 := 2506,
	XUUNIT_SENSORTIMES_VACUUM_6 := 2507,
	XUUNIT_SENSORTIMES_VACUUM_7 := 2508,
	XUUNIT_SENSORTIMES_VACUUM_8 := 2509,
	XUUNIT_SENSORTIMES_VACUUM_9 := 2510,
	XUUNIT_SENSORTIMES_VACUUM_10 := 2511,
	XUUNIT_SENSORTIMES_VACUUM_11 := 2512,
	XUUNIT_SENSORTIMES_VACUUM_12 := 2513,
	XUUNIT_SENSORTIMES_VACUUM_13 := 2514,
	XUUNIT_SENSORTIMES_VACUUM_14 := 2515,
	XUUNIT_SENSORTIMES_VACUUM_15 := 2516,
	XUUNIT_SENSORTIMES_VACUUM_16 := 2517,
	XUUNIT_SENSORTIMES_VACUUM_17 := 2518,
	XUUNIT_SENSORTIMES_VACUUM_18 := 2519,
	XUUNIT_SENSORTIMES_VACUUM_19 := 2520,
	XUUNIT_SENSORTIMES_VACUUM_20 := 2521,
	XUUNIT_SENSORTIMES_VACUUM_21 := 2522,
	XUUNIT_SENSORTIMES_VACUUM_22 := 2523,
	XUUNIT_SENSORTIMES_VACUUM_23 := 2524,
	XUUNIT_SENSORTIMES_VACUUM_24 := 2525,
	XUUNIT_SENSORTIMES_VACUUM_25 := 2526,
	XUUNIT_SENSORTIMES_VACUUM_26 := 2527,
	XUUNIT_SENSORTIMES_VACUUM_27 := 2528,
	XUUNIT_SENSORTIMES_VACUUM_28 := 2529,
	XUUNIT_SENSORTIMES_VACUUM_29 := 2530,
	XUUNIT_SENSORTIMES_VACUUM_30 := 2531,
	XUUNIT_SENSORTIMES_VACUUM_31 := 2532,
	XUUNIT_SENSORTIMES_VACUUM_32 := 2533,
	XU2UNIT_SENSORTIMES_VACUUM_1 := 2534,
	XU2UNIT_SENSORTIMES_VACUUM_2 := 2535,
	XU2UNIT_SENSORTIMES_VACUUM_3 := 2536,
	XU2UNIT_SENSORTIMES_VACUUM_4 := 2537,
	XU2UNIT_SENSORTIMES_VACUUM_5 := 2538,
	XU2UNIT_SENSORTIMES_VACUUM_6 := 2539,
	XU2UNIT_SENSORTIMES_VACUUM_7 := 2540,
	XU2UNIT_SENSORTIMES_VACUUM_8 := 2541,
	XU2UNIT_SENSORTIMES_VACUUM_9 := 2542,
	XU2UNIT_SENSORTIMES_VACUUM_10 := 2543,
	XU2UNIT_SENSORTIMES_VACUUM_11 := 2544,
	XU2UNIT_SENSORTIMES_VACUUM_12 := 2545,
	XU2UNIT_SENSORTIMES_VACUUM_13 := 2546,
	XU2UNIT_SENSORTIMES_VACUUM_14 := 2547,
	XU2UNIT_SENSORTIMES_VACUUM_15 := 2548,
	XU2UNIT_SENSORTIMES_VACUUM_16 := 2549,
	XU2UNIT_SENSORTIMES_VACUUM_17 := 2550,
	XU2UNIT_SENSORTIMES_VACUUM_18 := 2551,
	XU2UNIT_SENSORTIMES_VACUUM_19 := 2552,
	XU2UNIT_SENSORTIMES_VACUUM_20 := 2553,
	XU2UNIT_SENSORTIMES_VACUUM_21 := 2554,
	XU2UNIT_SENSORTIMES_VACUUM_22 := 2555,
	XU2UNIT_SENSORTIMES_VACUUM_23 := 2556,
	XU2UNIT_SENSORTIMES_VACUUM_24 := 2557,
	XU2UNIT_SENSORTIMES_VACUUM_25 := 2558,
	XU2UNIT_SENSORTIMES_VACUUM_26 := 2559,
	XU2UNIT_SENSORTIMES_VACUUM_27 := 2560,
	XU2UNIT_SENSORTIMES_VACUUM_28 := 2561,
	XU2UNIT_SENSORTIMES_VACUUM_29 := 2562,
	XU2UNIT_SENSORTIMES_VACUUM_30 := 2563,
	XU2UNIT_SENSORTIMES_VACUUM_31 := 2564,
	XU2UNIT_SENSORTIMES_VACUUM_32 := 2565,
	MAGAZINE_SENSORTIMES_VACUUM_9 := 2566,
	MAGAZINE_SENSORTIMES_VACUUM_10 := 2567,
	MAGAZINE_SENSORTIMES_VACUUM_11 := 2568,
	MAGAZINE_SENSORTIMES_VACUUM_12 := 2569,
	MAGAZINE_SENSORTIMES_VACUUM_13 := 2570,
	MAGAZINE_SENSORTIMES_VACUUM_14 := 2571,
	MAGAZINE_SENSORTIMES_VACUUM_15 := 2572,
	MAGAZINE_SENSORTIMES_VACUUM_16 := 2573,
	MAGAZINE_SENSORTIMES_VACUUM_17 := 2574,
	MAGAZINE_SENSORTIMES_VACUUM_18 := 2575,
	MAGAZINE_SENSORTIMES_VACUUM_19 := 2576,
	MAGAZINE_SENSORTIMES_VACUUM_20 := 2577,
	MAGAZINE_SENSORTIMES_VACUUM_21 := 2578,
	MAGAZINE_SENSORTIMES_VACUUM_22 := 2579,
	MAGAZINE_SENSORTIMES_VACUUM_23 := 2580,
	MAGAZINE_SENSORTIMES_VACUUM_24 := 2581,
	MAGAZINE_SENSORTIMES_VACUUM_25 := 2582,
	MAGAZINE_SENSORTIMES_VACUUM_26 := 2583,
	MAGAZINE_SENSORTIMES_VACUUM_27 := 2584,
	MAGAZINE_SENSORTIMES_VACUUM_28 := 2585,
	MAGAZINE_SENSORTIMES_VACUUM_29 := 2586,
	MAGAZINE_SENSORTIMES_VACUUM_30 := 2587,
	MAGAZINE_SENSORTIMES_VACUUM_31 := 2588,
	MAGAZINE_SENSORTIMES_VACUUM_32 := 2589,
	MAGAZINE_2_SENSORTIMES_VACUUM_1 := 2590,
	MAGAZINE_2_SENSORTIMES_VACUUM_2 := 2591,
	MAGAZINE_2_SENSORTIMES_VACUUM_3 := 2592,
	MAGAZINE_2_SENSORTIMES_VACUUM_4 := 2593,
	MAGAZINE_2_SENSORTIMES_VACUUM_5 := 2594,
	MAGAZINE_2_SENSORTIMES_VACUUM_6 := 2595,
	MAGAZINE_2_SENSORTIMES_VACUUM_7 := 2596,
	MAGAZINE_2_SENSORTIMES_VACUUM_8 := 2597,
	MAGAZINE_2_SENSORTIMES_VACUUM_9 := 2598,
	MAGAZINE_2_SENSORTIMES_VACUUM_10 := 2599,
	MAGAZINE_2_SENSORTIMES_VACUUM_11 := 2600,
	MAGAZINE_2_SENSORTIMES_VACUUM_12 := 2601,
	MAGAZINE_2_SENSORTIMES_VACUUM_13 := 2602,
	MAGAZINE_2_SENSORTIMES_VACUUM_14 := 2603,
	MAGAZINE_2_SENSORTIMES_VACUUM_15 := 2604,
	MAGAZINE_2_SENSORTIMES_VACUUM_16 := 2605,
	MAGAZINE_2_SENSORTIMES_VACUUM_17 := 2606,
	MAGAZINE_2_SENSORTIMES_VACUUM_18 := 2607,
	MAGAZINE_2_SENSORTIMES_VACUUM_19 := 2608,
	MAGAZINE_2_SENSORTIMES_VACUUM_20 := 2609,
	MAGAZINE_2_SENSORTIMES_VACUUM_22 := 2610,
	MAGAZINE_2_SENSORTIMES_VACUUM_21 := 2611,
	MAGAZINE_2_SENSORTIMES_VACUUM_26 := 2612,
	MAGAZINE_2_SENSORTIMES_VACUUM_23 := 2613,
	MAGAZINE_2_SENSORTIMES_VACUUM_24 := 2614,
	MAGAZINE_2_SENSORTIMES_VACUUM_25 := 2615,
	MAGAZINE_2_SENSORTIMES_VACUUM_27 := 2616,
	MAGAZINE_2_SENSORTIMES_VACUUM_28 := 2617,
	MAGAZINE_2_SENSORTIMES_VACUUM_29 := 2618,
	MAGAZINE_2_SENSORTIMES_VACUUM_30 := 2619,
	MAGAZINE_2_SENSORTIMES_VACUUM_31 := 2620,
	MAGAZINE_2_SENSORTIMES_VACUUM_32 := 2621,
	MAGAZINE_2_SENSORTIMES_SHIFTIN := 2622,
	MAGAZINE_2_SENSORTIMES_SHIFTOUT := 2623,
	MAGAZINE_2_SENSORTIMES_CHANGEDRAWERIN := 2624,
	MAGAZINE_2_SENSORTIMES_CHANGEDRAWEROUT := 2625,
	MAGAZINE_2_SENSORTIMES_LOCKDRAWERIN := 2626,
	MAGAZINE_2_SENSORTIMES_LOCKDRAWEROUT := 2627,
	Y3UNIT_SENSORTIMES_SHIFTIN := 2628,
	Y3UNIT_SENSORTIMES_SHIFTOUT := 2629,
	TUNIT_SENSORTIMES_VACUUM_2_2 := 2630,
	TUNIT_SENSORTIMES_VACUUM_1_1 := 2631,
	TUNIT_SENSORTIMES_VACUUM_1_2 := 2632,
	TUNIT_SENSORTIMES_VACUUM_1_3 := 2633,
	TUNIT_SENSORTIMES_VACUUM_1_4 := 2634,
	TUNIT_SENSORTIMES_VACUUM_2_1 := 2635,
	TUNIT_SENSORTIMES_VACUUM_2_3 := 2636,
	TUNIT_SENSORTIMES_VACUUM_2_4 := 2637,
	TUNIT_SENSORTIMES_EXTENDIN := 2638,
	TUNIT_SENSORTIMES_EXTENDOUT := 2639,
	TUNIT_SENSORTIMES_ROTATEIN := 2640,
	TUNIT_SENSORTIMES_ROTATEOUT := 2641,
	TUNIT_SENSORTIMES_CLOSELIDIN := 2642,
	TUNIT_SENSORTIMES_CLOSELIDOUT := 2643,
	UPSTACKER_1_1_SENSORTIMES_LIFTIN := 2644,
	UPSTACKER_1_1_SENSORTIMES_LIFTOUT := 2645,
	UPSTACKER_1_1_SENSORTIMES_LOWERSTACKPLATEIN := 2646,
	UPSTACKER_1_1_SENSORTIMES_LOWERSTACKPLATEOUT := 2647,
	UPSTACKER_1_1_SENSORTIMES_UPPERSTACKPLATEOUT := 2648,
	UPSTACKER_1_1_SENSORTIMES_UPPERSTACKPLATEIN := 2649,
	UPSTACKER_2_1_SENSORTIMES_LIFTIN := 2650,
	UPSTACKER_2_1_SENSORTIMES_LIFTOUT := 2651,
	UPSTACKER_2_1_SENSORTIMES_LOWERSTACKPLATEIN := 2652,
	UPSTACKER_2_1_SENSORTIMES_LOWERSTACKPLATEOUT := 2653,
	UPSTACKER_2_1_SENSORTIMES_UPPERSTACKPLATEOUT := 2654,
	UPSTACKER_2_1_SENSORTIMES_UPPERSTACKPLATEIN := 2655,
	UPSTACKER_3_1_SENSORTIMES_LIFTIN := 2656,
	UPSTACKER_3_1_SENSORTIMES_LIFTOUT := 2657,
	UPSTACKER_3_1_SENSORTIMES_LOWERSTACKPLATEIN := 2658,
	UPSTACKER_3_1_SENSORTIMES_LOWERSTACKPLATEOUT := 2659,
	UPSTACKER_3_1_SENSORTIMES_UPPERSTACKPLATEOUT := 2660,
	UPSTACKER_3_1_SENSORTIMES_UPPERSTACKPLATEIN := 2661,
	UPSTACKER_4_1_SENSORTIMES_LIFTIN := 2662,
	UPSTACKER_4_1_SENSORTIMES_LIFTOUT := 2663,
	UPSTACKER_4_1_SENSORTIMES_LOWERSTACKPLATEIN := 2664,
	UPSTACKER_4_1_SENSORTIMES_LOWERSTACKPLATEOUT := 2665,
	UPSTACKER_4_1_SENSORTIMES_UPPERSTACKPLATEOUT := 2666,
	UPSTACKER_4_1_SENSORTIMES_UPPERSTACKPLATEIN := 2667,
	UPSTACKER_5_1_SENSORTIMES_LIFTIN := 2668,
	UPSTACKER_5_1_SENSORTIMES_LIFTOUT := 2669,
	UPSTACKER_5_1_SENSORTIMES_LOWERSTACKPLATEIN := 2670,
	UPSTACKER_5_1_SENSORTIMES_LOWERSTACKPLATEOUT := 2671,
	UPSTACKER_5_1_SENSORTIMES_UPPERSTACKPLATEOUT := 2672,
	UPSTACKER_5_1_SENSORTIMES_UPPERSTACKPLATEIN := 2673,
	UPSTACKER_6_1_SENSORTIMES_LIFTIN := 2674,
	UPSTACKER_6_1_SENSORTIMES_LIFTOUT := 2675,
	UPSTACKER_6_1_SENSORTIMES_LOWERSTACKPLATEIN := 2676,
	UPSTACKER_6_1_SENSORTIMES_LOWERSTACKPLATEOUT := 2677,
	UPSTACKER_6_1_SENSORTIMES_UPPERSTACKPLATEOUT := 2678,
	UPSTACKER_6_1_SENSORTIMES_UPPERSTACKPLATEIN := 2679,
	UPSTACKER_7_1_SENSORTIMES_LIFTIN := 2680,
	UPSTACKER_7_1_SENSORTIMES_LIFTOUT := 2681,
	UPSTACKER_7_1_SENSORTIMES_LOWERSTACKPLATEIN := 2682,
	UPSTACKER_7_1_SENSORTIMES_LOWERSTACKPLATEOUT := 2683,
	UPSTACKER_7_1_SENSORTIMES_UPPERSTACKPLATEOUT := 2684,
	UPSTACKER_7_1_SENSORTIMES_UPPERSTACKPLATEIN := 2685,
	UPSTACKER_8_1_SENSORTIMES_LIFTIN := 2686,
	UPSTACKER_8_1_SENSORTIMES_LIFTOUT := 2687,
	UPSTACKER_8_1_SENSORTIMES_LOWERSTACKPLATEIN := 2688,
	UPSTACKER_8_1_SENSORTIMES_LOWERSTACKPLATEOUT := 2689,
	UPSTACKER_8_1_SENSORTIMES_UPPERSTACKPLATEOUT := 2690,
	UPSTACKER_8_1_SENSORTIMES_UPPERSTACKPLATEIN := 2691,
	UPSTACKER_1_2_SENSORTIMES_LIFTIN := 2692,
	UPSTACKER_1_2_SENSORTIMES_LIFTOUT := 2693,
	UPSTACKER_1_2_SENSORTIMES_LOWERSTACKPLATEIN := 2694,
	UPSTACKER_1_2_SENSORTIMES_LOWERSTACKPLATEOUT := 2695,
	UPSTACKER_1_2_SENSORTIMES_UPPERSTACKPLATEOUT := 2696,
	UPSTACKER_1_2_SENSORTIMES_UPPERSTACKPLATEIN := 2697,
	UPSTACKER_2_2_SENSORTIMES_LIFTIN := 2698,
	UPSTACKER_2_2_SENSORTIMES_LIFTOUT := 2699,
	UPSTACKER_2_2_SENSORTIMES_LOWERSTACKPLATEIN := 2700,
	UPSTACKER_2_2_SENSORTIMES_LOWERSTACKPLATEOUT := 2701,
	UPSTACKER_2_2_SENSORTIMES_UPPERSTACKPLATEOUT := 2702,
	UPSTACKER_2_2_SENSORTIMES_UPPERSTACKPLATEIN := 2703,
	UPSTACKER_3_2_SENSORTIMES_LIFTIN := 2704,
	UPSTACKER_3_2_SENSORTIMES_LIFTOUT := 2705,
	UPSTACKER_3_2_SENSORTIMES_LOWERSTACKPLATEIN := 2706,
	UPSTACKER_3_2_SENSORTIMES_LOWERSTACKPLATEOUT := 2707,
	UPSTACKER_3_2_SENSORTIMES_UPPERSTACKPLATEOUT := 2708,
	UPSTACKER_3_2_SENSORTIMES_UPPERSTACKPLATEIN := 2709,
	UPSTACKER_4_2_SENSORTIMES_LIFTIN := 2710,
	UPSTACKER_4_2_SENSORTIMES_LIFTOUT := 2711,
	UPSTACKER_4_2_SENSORTIMES_LOWERSTACKPLATEIN := 2712,
	UPSTACKER_4_2_SENSORTIMES_LOWERSTACKPLATEOUT := 2713,
	UPSTACKER_4_2_SENSORTIMES_UPPERSTACKPLATEOUT := 2714,
	UPSTACKER_4_2_SENSORTIMES_UPPERSTACKPLATEIN := 2715,
	UPSTACKER_5_2_SENSORTIMES_LIFTIN := 2716,
	UPSTACKER_5_2_SENSORTIMES_LIFTOUT := 2717,
	UPSTACKER_5_2_SENSORTIMES_LOWERSTACKPLATEIN := 2718,
	UPSTACKER_5_2_SENSORTIMES_LOWERSTACKPLATEOUT := 2719,
	UPSTACKER_5_2_SENSORTIMES_UPPERSTACKPLATEOUT := 2720,
	UPSTACKER_5_2_SENSORTIMES_UPPERSTACKPLATEIN := 2721,
	UPSTACKER_6_2_SENSORTIMES_LIFTIN := 2722,
	UPSTACKER_6_2_SENSORTIMES_LIFTOUT := 2723,
	UPSTACKER_6_2_SENSORTIMES_LOWERSTACKPLATEIN := 2724,
	UPSTACKER_6_2_SENSORTIMES_LOWERSTACKPLATEOUT := 2725,
	UPSTACKER_6_2_SENSORTIMES_UPPERSTACKPLATEOUT := 2726,
	UPSTACKER_6_2_SENSORTIMES_UPPERSTACKPLATEIN := 2727,
	UPSTACKER_7_2_SENSORTIMES_LIFTIN := 2728,
	UPSTACKER_7_2_SENSORTIMES_LIFTOUT := 2729,
	UPSTACKER_7_2_SENSORTIMES_LOWERSTACKPLATEIN := 2730,
	UPSTACKER_7_2_SENSORTIMES_LOWERSTACKPLATEOUT := 2731,
	UPSTACKER_7_2_SENSORTIMES_UPPERSTACKPLATEOUT := 2732,
	UPSTACKER_7_2_SENSORTIMES_UPPERSTACKPLATEIN := 2733,
	UPSTACKER_8_2_SENSORTIMES_LIFTIN := 2734,
	UPSTACKER_8_2_SENSORTIMES_LIFTOUT := 2735,
	UPSTACKER_8_2_SENSORTIMES_LOWERSTACKPLATEIN := 2736,
	UPSTACKER_8_2_SENSORTIMES_LOWERSTACKPLATEOUT := 2737,
	UPSTACKER_8_2_SENSORTIMES_UPPERSTACKPLATEOUT := 2738,
	UPSTACKER_8_2_SENSORTIMES_UPPERSTACKPLATEIN := 2739,
	FANUC_SENSORTIMES_CLAMPLONGSIDEIN := 2740,
	FANUC_SENSORTIMES_CLAMPLONGSIDEOUT := 2741,
	FANUC_SENSORTIMES_CLAMPSHORTSIDEIN := 2742,
	FANUC_SENSORTIMES_CLAMPSHORTSIDEOUT := 2743,
	PATTERNIZER_SENSORTIMES_CLAMPSTACK1IN := 2744,
	PATTERNIZER_SENSORTIMES_CLAMPSTACK2IN := 2745,
	PATTERNIZER_SENSORTIMES_CLAMPSTACK3IN := 2746,
	PATTERNIZER_SENSORTIMES_CLAMPSTACK4IN := 2747,
	PATTERNIZER_SENSORTIMES_CLAMPSTACK1OUT := 2748,
	PATTERNIZER_SENSORTIMES_CLAMPSTACK2OUT := 2749,
	PATTERNIZER_SENSORTIMES_CLAMPSTACK3OUT := 2750,
	PATTERNIZER_SENSORTIMES_CLAMPSTACK4OUT := 2751,
	GRIPPER_SENSORTIMES_EXTENDIN := 2752,
	GRIPPER_SENSORTIMES_EXTENDOUT := 2753,
	GRIPPER_SENSORTIMES_PUSHERIN := 2754,
	GRIPPER_SENSORTIMES_PUSHEROUT := 2755,
	GRIPPER_SENSORTIMES_CLAMPSTACK10MMIN := 2756,
	GRIPPER_SENSORTIMES_CLAMPSTACK10MMOUT := 2757,
	GRIPPER_SENSORTIMES_CLAMPSTACK20MMIN := 2758,
	GRIPPER_SENSORTIMES_CLAMPSTACK20MMOUT := 2759,
	GRIPPER_SENSORTIMES_CLAMPSTACKLONGSIDEIN := 2760,
	GRIPPER_SENSORTIMES_CLAMPSTACKLONGSIDEOUT := 2761,
	GRIPPER_SENSORTIMES_VACUUM := 2762,
	SHEETMAGAZINE_SENSORTIMES_SLIDINGPANELIN := 2763,
	EXTENDOUT1_DONTUSE1 := 2764,
	EXTENDOUT1_DONTUSE := 2765,
	SHEETMAGAZINE_SENSORTIMES_SLIDINGPANELOUT := 2766,
	BOXINFEED_SENSORTIMES_CLAMPSECONDBOXIN := 2767,
	BOXINFEED_SENSORTIMES_CLAMPSECONDBOXOUT := 2768,
	BOXINFEED_SENSORTIMES_PUSHEROUT := 2769,
	BOXINFEED_SENSORTIMES_PUSHERIN := 2770,
	BOXFILLSTATION_SENSORTIMES_OPENBOXSIDE1IN := 2771,
	BOXFILLSTATION_SENSORTIMES_OPENBOXSIDE1OUT := 2772,
	BOXFILLSTATION_SENSORTIMES_OPENBOXSIDE2IN := 2773,
	BOXFILLSTATION_SENSORTIMES_OPENBOXSIDE2OUT := 2774,
	BOXFILLSTATION_SENSORTIMES_OPENBOXSIDE3IN := 2775,
	BOXFILLSTATION_SENSORTIMES_OPENBOXSIDE3OUT := 2776,
	BOXFILLSTATION_SENSORTIMES_OPENBOXSIDE4IN := 2777,
	BOXFILLSTATION_SENSORTIMES_OPENBOXSIDE4OUT := 2778,
	Y2UNIT_TIME_IDLE := 2779,
	Y3UNIT_TIME_IDLE := 2780,
	XI2UNIT_TIME_IDLE := 2781,
	XU2UNIT_TIME_IDLE := 2782,
	MAGAZINE_2_TIME_IDLE := 2783,
	SUNIT_TIME_IDLE := 2784,
	TUNIT_TIME_IDLE := 2785,
	AUNIT_TIME_IDLE := 2786,
	UPSTACKER_1_1_TIME_IDLE := 2787,
	UPSTACKER_2_1_TIME_IDLE := 2788,
	UPSTACKER_3_1_TIME_IDLE := 2789,
	UPSTACKER_4_1_TIME_IDLE := 2790,
	UPSTACKER_5_1_TIME_IDLE := 2791,
	UPSTACKER_6_1_TIME_IDLE := 2792,
	UPSTACKER_7_1_TIME_IDLE := 2793,
	UPSTACKER_8_1_TIME_IDLE := 2794,
	UPSTACKER_1_2_TIME_IDLE := 2795,
	UPSTACKER_2_2_TIME_IDLE := 2796,
	UPSTACKER_3_2_TIME_IDLE := 2797,
	UPSTACKER_4_2_TIME_IDLE := 2798,
	UPSTACKER_5_2_TIME_IDLE := 2799,
	UPSTACKER_6_2_TIME_IDLE := 2800,
	UPSTACKER_7_2_TIME_IDLE := 2801,
	UPSTACKER_8_2_TIME_IDLE := 2802,
	FANUC_TIME_IDLE := 2803,
	PATTERNIZER_TIME_IDLE := 2804,
	GRIPPER_TIME_IDLE := 2805,
	BFU_YUNIT_TIME_IDLE := 2806,
	SHEETMAGAZINE_TIME_IDLE := 2807,
	BOXINFEED_TIME_IDLE := 2808,
	BOXFILLSTATION_TIME_IDLE := 2809,
	BOXOUTFEED_TIME_IDLE := 2810,
	PICKPRODUCTSFROMUPSTACKER_TIME_IDLE := 2811,
	PLACEPRODUCTSONPATTERNIZER_TIME_IDLE := 2812,
	REJECTPRODUCTS_TIME_IDLE := 2813,
	PICKPLACEPRODUCTS_TIME_IDLE := 2814,
	PICKPLACEY_TIME_IDLE := 2815,
	PICKPLACESHEETS_TIME_IDLE := 2816,
	SHEETREFILLING_TIME_IDLE := 2817,
	BOXFILLING_TIME_IDLE := 2818,
	BOXTRANSPORT_TIME_IDLE := 2819,
	Y2UNIT_TIME_ACTIVE := 2820,
	XI2UNIT_TIME_ACTIVE := 2821,
	MAGAZINE_2_TIME_ACTIVE := 2822,
	XU2UNIT_TIME_ACTIVE := 2823,
	SUNIT_TIME_ACTIVE := 2824,
	Y3UNIT_TIME_ACTIVE := 2825,
	TUNIT_TIME_ACTIVE := 2826,
	AUNIT_TIME_ACTIVE := 2827,
	BOXFILLSTATION_TIME_ACTIVE := 2828,
	BOXINFEED_TIME_ACTIVE := 2829,
	BOXOUTFEED_TIME_ACTIVE := 2830,
	SHEETMAGAZINE_TIME_ACTIVE := 2831,
	UPSTACKER_1_1_TIME_ACTIVE := 2832,
	UPSTACKER_2_1_TIME_ACTIVE := 2833,
	UPSTACKER_3_1_TIME_ACTIVE := 2834,
	UPSTACKER_4_1_TIME_ACTIVE := 2835,
	UPSTACKER_5_1_TIME_ACTIVE := 2836,
	UPSTACKER_6_1_TIME_ACTIVE := 2837,
	UPSTACKER_7_1_TIME_ACTIVE := 2838,
	UPSTACKER_8_1_TIME_ACTIVE := 2839,
	UPSTACKER_1_2_TIME_ACTIVE := 2840,
	UPSTACKER_2_2_TIME_ACTIVE := 2841,
	UPSTACKER_3_2_TIME_ACTIVE := 2842,
	UPSTACKER_4_2_TIME_ACTIVE := 2843,
	UPSTACKER_5_2_TIME_ACTIVE := 2844,
	UPSTACKER_6_2_TIME_ACTIVE := 2845,
	UPSTACKER_7_2_TIME_ACTIVE := 2846,
	UPSTACKER_8_2_TIME_ACTIVE := 2847,
	FANUC_TIME_ACTIVE := 2848,
	PATTERNIZER_TIME_ACTIVE := 2849,
	GRIPPER_TIME_ACTIVE := 2850,
	BFU_YUNIT_TIME_ACTIVE := 2851,
	PICKPRODUCTSFROMUPSTACKER_TIME_ACTIVE := 2852,
	PLACEPRODUCTSONPATTERNIZER_TIME_ACTIVE := 2853,
	REJECTPRODUCTS_TIME_ACTIVE := 2854,
	PICKPLACEPRODUCTS_TIME_ACTIVE := 2855,
	PICKPLACEY_TIME_ACTIVE := 2856,
	PICKPLACESHEETS_TIME_ACTIVE := 2857,
	SHEETREFILLING_TIME_ACTIVE := 2858,
	BOXFILLING_TIME_ACTIVE := 2859,
	BOXTRANSPORT_TIME_ACTIVE := 2860,
	DRAWERMAGAZINE_2_ALARMS := 2861,
	XUNIT_ALARMS := 2862,
	BFU_TURNER_ALARMS := 2863,
	XUNIT_BFU_ALARMS := 2864,
	CONVEYORS_BFU_ALARMS := 2865,
	XUNIT_COVEREDDISTANCE := 2866,
	ZRUNIT_ZR1_COVEREDDISTANCE := 2867,
	XUNIT_BFU_COVEREDDISTANCE := 2868,
	XUNIT_ERRORID := 2869,
	ZRUNIT_ZR1_ERRORID := 2870,
	XUNIT_BFU_ERRORID := 2871,
	XUNIT_AXISERRORID := 2872,
	XUNIT_BFU_AXISERRORID := 2873,
	XUNIT_DRIVEERRORID := 2874,
	XUNIT_BFU_DRIVEERRORID := 2875,
	XUNIT_DRIVEUTILISATION := 2876,
	ZRUNIT_ZR1_DRIVEUTILISATION := 2877,
	XUNIT_BFU_DRIVEUTILISATION := 2878,
	XUNIT_MOTORUTILISATION := 2879,
	ZRUNIT_ZR1_MOTORUTILISATION := 2880,
	XUNIT_BFU_MOTORUTILISATION := 2881,
	XUNIT_SENSORTIMES_VACUUMLID_1 := 2882,
	XUNIT_SENSORTIMES_VACUUMLID_2 := 2883,
	XUNIT_SENSORTIMES_VACUUMSCOOP_1 := 2884,
	XUNIT_SENSORTIMES_VACUUMSCOOP_2 := 2885,
	XUNIT_SENSORTIMES_ROTATESCOOPIN := 2886,
	XUNIT_SENSORTIMES_ROTATESCOOPOUT := 2887,
	XUNIT_SENSORTIMES_CLAMPLIDIN_1 := 2888,
	XUNIT_SENSORTIMES_CLAMPLIDIN_2 := 2889,
	TXUNIT_ALARMS := 2890,
	TXUNIT_COVEREDDISTANCE := 2891,
	TXUNIT_ERRORID := 2892,
	TXUNIT_AXISERRORID := 2893,
	TXUNIT_DRIVEERRORID := 2894,
	TXUNIT_DRIVEUTILISATION := 2895,
	TXUNIT_MOTORUTILISATION := 2896,
	ZUNIT_SENSORTIMES_CLOSELIDIN := 2897,
	ZUNIT_SENSORTIMES_CLOSELIDOUT := 2898,
	ZUNIT_SENSORTIMES_FLIPCAPIN := 2899,
	ZUNIT_SENSORTIMES_FLIPCAPOUT := 2900,
	TXUNIT_SENSORTIMES_LIFTIN_1 := 2901,
	TXUNIT_SENSORTIMES_LIFTIN_2 := 2902,
	TXUNIT_SENSORTIMES_LIFTIN_3 := 2903,
	TXUNIT_SENSORTIMES_LIFTOUT_1 := 2904,
	TXUNIT_SENSORTIMES_LIFTOUT_2 := 2905,
	TXUNIT_SENSORTIMES_LIFTOUT_3 := 2906,
	TXUNIT_SENSORTIMES_EXTENDIN := 2907,
	TXUNIT_SENSORTIMES_EXTENDOUT := 2908,
	ZUNIT_SENSORTIMES_LOCKZRIN := 2909,
	ZUNIT_SENSORTIMES_LOCKZROUT := 2910,
	BFU_PICKANDPLACE_SENSORTIMES_VACUUM_1 := 2911,
	BFU_PICKANDPLACE_SENSORTIMES_SHIFT := 2912,
	BFU_PICKANDPLACE_SENSORTIMES_SHIFTCENTERIN := 2913,
	BFU_PICKANDPLACE_SENSORTIMES_SHIFTCENTEROUT := 2914,
	BOXCONVEYOR_SENSORTIMES_CLAMPBOXIN := 2915,
	BOXCONVEYOR_SENSORTIMES_CLAMPBOXOUT := 2916,
	BOXCONVEYOR_SENSORTIMES_VACUUMPUSHER := 2917,
	BOXCONVEYOR_SENSORTIMES_PUSHERINFEEDIN := 2918,
	BOXCONVEYOR_SENSORTIMES_PUSHERINFEEDOUT := 2919,
	BOXCONVEYOR_SENSORTIMES_PUSHEROUTFEEDIN := 2920,
	BOXCONVEYOR_SENSORTIMES_PUSHEROUTFEEDOUT := 2921,
	TURNER_BFU_SENSORTIMES_VACUUM := 2922,
	TURNER_BFU_SENSORTIMES_ROTATEIN := 2923,
	TURNER_BFU_SENSORTIMES_ROTATEOUT := 2924,
	BOXCONVEYOR_SENSORTIMES_BOXCENTERIN := 2925,
	BOXCONVEYOR_SENSORTIMES_BOXCENTEROUT := 2926,
	XUNIT_TIME_IDLE := 2927,
	CAMERA_YUNIT_TIME_IDLE := 2928,
	ZRUNIT_ZR1_TIME_IDLE := 2929,
	BFU_PICKANDPLACE_TIME_IDLE := 2930,
	TURNER_BFU_TIME_IDLE := 2931,
	BOXCONVEYOR_TIME_IDLE := 2932,
	XUNIT_TIME_ACTIVE := 2933,
	CAMERA_YUNIT_TIME_ACTIVE := 2934,
	ZRUNIT_ZR1_TIME_ACTIVE := 2935,
	BFU_PICKANDPLACE_TIME_ACTIVE := 2936,
	TURNER_BFU_TIME_ACTIVE := 2937,
	BOXCONVEYOR_TIME_ACTIVE := 2938,
	CONVEYORS_COVEREDDISTANCE := 2939,
	CONVEYORS_ERRORID := 2940,
	CONVEYORS_AXISERRORID := 2941,
	CONVEYORS_DRIVEERRORID := 2942,
	CONVEYORS_DRIVEUTILISATION := 2943,
	CONVEYORS_MOTORUTILISATION := 2944,
	MAIN_STEPBYSTEPACTIVE := 2945,
	LABELADJUSTMENT_MAGAZINE_DRAWER_1_CASSETTE_1_POSITION_1 := 2947,
	LABELADJUSTMENT_MAGAZINE_DRAWER_1_CASSETTE_1_POSITION_2 := 2948,
	LABELADJUSTMENT_MAGAZINE_DRAWER_1_CASSETTE_1_POSITION_3 := 2949,
	LABELADJUSTMENT_MAGAZINE_DRAWER_1_CASSETTE_2_POSITION_1 := 2950,
	LABELADJUSTMENT_MAGAZINE_DRAWER_1_CASSETTE_2_POSITION_2 := 2951,
	LABELADJUSTMENT_MAGAZINE_DRAWER_1_CASSETTE_2_POSITION_3 := 2952,
	LABELADJUSTMENT_MAGAZINE_DRAWER_1_CASSETTE_3_POSITION_1 := 2953,
	LABELADJUSTMENT_MAGAZINE_DRAWER_1_CASSETTE_3_POSITION_2 := 2954,
	LABELADJUSTMENT_MAGAZINE_DRAWER_1_CASSETTE_3_POSITION_3 := 2955,
	LABELADJUSTMENT_MAGAZINE_DRAWER_1_CASSETTE_4_POSITION_1 := 2956,
	LABELADJUSTMENT_MAGAZINE_DRAWER_1_CASSETTE_4_POSITION_2 := 2957,
	LABELADJUSTMENT_MAGAZINE_DRAWER_1_CASSETTE_4_POSITION_3 := 2958,
	LABELADJUSTMENT_MAGAZINE_DRAWER_1_CASSETTE_5_POSITION_1 := 2959,
	LABELADJUSTMENT_MAGAZINE_DRAWER_1_CASSETTE_5_POSITION_2 := 2960,
	LABELADJUSTMENT_MAGAZINE_DRAWER_1_CASSETTE_5_POSITION_3 := 2961,
	LABELADJUSTMENT_MAGAZINE_DRAWER_1_CASSETTE_6_POSITION_1 := 2962,
	LABELADJUSTMENT_MAGAZINE_DRAWER_1_CASSETTE_6_POSITION_2 := 2963,
	LABELADJUSTMENT_MAGAZINE_DRAWER_1_CASSETTE_6_POSITION_3 := 2964,
	LABELADJUSTMENT_MAGAZINE_DRAWER_1_CASSETTE_7_POSITION_1 := 2965,
	LABELADJUSTMENT_MAGAZINE_DRAWER_1_CASSETTE_7_POSITION_2 := 2966,
	LABELADJUSTMENT_MAGAZINE_DRAWER_1_CASSETTE_7_POSITION_3 := 2967,
	LABELADJUSTMENT_MAGAZINE_DRAWER_1_CASSETTE_8_POSITION_1 := 2968,
	LABELADJUSTMENT_MAGAZINE_DRAWER_1_CASSETTE_8_POSITION_2 := 2969,
	LABELADJUSTMENT_MAGAZINE_DRAWER_1_CASSETTE_8_POSITION_3 := 2970,
	LABELADJUSTMENT_MAGAZINE_DRAWER_1_CASSETTE_9_POSITION_1 := 2971,
	LABELADJUSTMENT_MAGAZINE_DRAWER_1_CASSETTE_9_POSITION_2 := 2972,
	LABELADJUSTMENT_MAGAZINE_DRAWER_1_CASSETTE_9_POSITION_3 := 2973,
	LABELADJUSTMENT_MAGAZINE_DRAWER_1_CASSETTE_10_POSITION_1 := 2974,
	LABELADJUSTMENT_MAGAZINE_DRAWER_1_CASSETTE_10_POSITION_2 := 2975,
	LABELADJUSTMENT_MAGAZINE_DRAWER_1_CASSETTE_10_POSITION_3 := 2976,
	LABELADJUSTMENT_MAGAZINE_DRAWER_1_CASSETTE_11_POSITION_1 := 2977,
	LABELADJUSTMENT_MAGAZINE_DRAWER_1_CASSETTE_11_POSITION_2 := 2978,
	LABELADJUSTMENT_MAGAZINE_DRAWER_1_CASSETTE_11_POSITION_3 := 2979,
	LABELADJUSTMENT_MAGAZINE_DRAWER_1_CASSETTE_12_POSITION_1 := 2980,
	LABELADJUSTMENT_MAGAZINE_DRAWER_1_CASSETTE_12_POSITION_2 := 2981,
	LABELADJUSTMENT_MAGAZINE_DRAWER_1_CASSETTE_12_POSITION_3 := 2982,
	LABELADJUSTMENT_MAGAZINE_DRAWER_1_CASSETTE_13_POSITION_1 := 2983,
	LABELADJUSTMENT_MAGAZINE_DRAWER_1_CASSETTE_13_POSITION_2 := 2984,
	LABELADJUSTMENT_MAGAZINE_DRAWER_1_CASSETTE_13_POSITION_3 := 2985,
	LABELADJUSTMENT_MAGAZINE_DRAWER_1_CASSETTE_14_POSITION_1 := 2986,
	LABELADJUSTMENT_MAGAZINE_DRAWER_1_CASSETTE_14_POSITION_2 := 2987,
	LABELADJUSTMENT_MAGAZINE_DRAWER_1_CASSETTE_14_POSITION_3 := 2988,
	LABELADJUSTMENT_MAGAZINE_DRAWER_1_CASSETTE_15_POSITION_1 := 2989,
	LABELADJUSTMENT_MAGAZINE_DRAWER_1_CASSETTE_15_POSITION_2 := 2990,
	LABELADJUSTMENT_MAGAZINE_DRAWER_1_CASSETTE_15_POSITION_3 := 2991,
	LABELADJUSTMENT_MAGAZINE_DRAWER_1_CASSETTE_16_POSITION_1 := 2992,
	LABELADJUSTMENT_MAGAZINE_DRAWER_1_CASSETTE_16_POSITION_2 := 2993,
	LABELADJUSTMENT_MAGAZINE_DRAWER_1_CASSETTE_16_POSITION_3 := 2994,
	LABELADJUSTMENT_MAGAZINE_DRAWER_1_CASSETTE_17_POSITION_1 := 2995,
	LABELADJUSTMENT_MAGAZINE_DRAWER_1_CASSETTE_17_POSITION_2 := 2996,
	LABELADJUSTMENT_MAGAZINE_DRAWER_1_CASSETTE_17_POSITION_3 := 2997,
	LABELADJUSTMENT_MAGAZINE_DRAWER_1_CASSETTE_18_POSITION_1 := 2998,
	LABELADJUSTMENT_MAGAZINE_DRAWER_1_CASSETTE_18_POSITION_2 := 2999,
	LABELADJUSTMENT_MAGAZINE_DRAWER_1_CASSETTE_18_POSITION_3 := 3000,
	LABELADJUSTMENT_MAGAZINE_DRAWER_1_CASSETTE_19_POSITION_1 := 3001,
	LABELADJUSTMENT_MAGAZINE_DRAWER_1_CASSETTE_19_POSITION_2 := 3002,
	LABELADJUSTMENT_MAGAZINE_DRAWER_1_CASSETTE_19_POSITION_3 := 3003,
	LABELADJUSTMENT_MAGAZINE_DRAWER_1_CASSETTE_20_POSITION_1 := 3004,
	LABELADJUSTMENT_MAGAZINE_DRAWER_1_CASSETTE_20_POSITION_2 := 3005,
	LABELADJUSTMENT_MAGAZINE_DRAWER_1_CASSETTE_20_POSITION_3 := 3006,
	LABELADJUSTMENT_MAGAZINE_DRAWER_1_CASSETTE_21_POSITION_1 := 3007,
	LABELADJUSTMENT_MAGAZINE_DRAWER_1_CASSETTE_21_POSITION_2 := 3008,
	LABELADJUSTMENT_MAGAZINE_DRAWER_1_CASSETTE_21_POSITION_3 := 3009,
	LABELADJUSTMENT_MAGAZINE_DRAWER_1_CASSETTE_22_POSITION_1 := 3010,
	LABELADJUSTMENT_MAGAZINE_DRAWER_1_CASSETTE_22_POSITION_2 := 3011,
	LABELADJUSTMENT_MAGAZINE_DRAWER_1_CASSETTE_22_POSITION_3 := 3012,
	LABELADJUSTMENT_MAGAZINE_DRAWER_1_CASSETTE_23_POSITION_1 := 3013,
	LABELADJUSTMENT_MAGAZINE_DRAWER_1_CASSETTE_23_POSITION_2 := 3014,
	LABELADJUSTMENT_MAGAZINE_DRAWER_1_CASSETTE_23_POSITION_3 := 3015,
	LABELADJUSTMENT_MAGAZINE_DRAWER_1_CASSETTE_24_POSITION_1 := 3016,
	LABELADJUSTMENT_MAGAZINE_DRAWER_1_CASSETTE_24_POSITION_2 := 3017,
	LABELADJUSTMENT_MAGAZINE_DRAWER_1_CASSETTE_24_POSITION_3 := 3018,
	LABELADJUSTMENT_MAGAZINE_DRAWER_1_CASSETTE_25_POSITION_1 := 3019,
	LABELADJUSTMENT_MAGAZINE_DRAWER_1_CASSETTE_25_POSITION_2 := 3020,
	LABELADJUSTMENT_MAGAZINE_DRAWER_1_CASSETTE_25_POSITION_3 := 3021,
	LABELADJUSTMENT_MAGAZINE_DRAWER_1_CASSETTE_26_POSITION_1 := 3022,
	LABELADJUSTMENT_MAGAZINE_DRAWER_1_CASSETTE_26_POSITION_2 := 3023,
	LABELADJUSTMENT_MAGAZINE_DRAWER_1_CASSETTE_26_POSITION_3 := 3024,
	LABELADJUSTMENT_MAGAZINE_DRAWER_1_CASSETTE_27_POSITION_1 := 3025,
	LABELADJUSTMENT_MAGAZINE_DRAWER_1_CASSETTE_27_POSITION_2 := 3026,
	LABELADJUSTMENT_MAGAZINE_DRAWER_1_CASSETTE_27_POSITION_3 := 3027,
	LABELADJUSTMENT_MAGAZINE_DRAWER_1_CASSETTE_28_POSITION_1 := 3028,
	LABELADJUSTMENT_MAGAZINE_DRAWER_1_CASSETTE_28_POSITION_2 := 3029,
	LABELADJUSTMENT_MAGAZINE_DRAWER_1_CASSETTE_28_POSITION_3 := 3030,
	LABELADJUSTMENT_MAGAZINE_DRAWER_1_CASSETTE_29_POSITION_1 := 3031,
	LABELADJUSTMENT_MAGAZINE_DRAWER_1_CASSETTE_29_POSITION_2 := 3032,
	LABELADJUSTMENT_MAGAZINE_DRAWER_1_CASSETTE_29_POSITION_3 := 3033,
	LABELADJUSTMENT_MAGAZINE_DRAWER_1_CASSETTE_30_POSITION_1 := 3034,
	LABELADJUSTMENT_MAGAZINE_DRAWER_1_CASSETTE_30_POSITION_2 := 3035,
	LABELADJUSTMENT_MAGAZINE_DRAWER_1_CASSETTE_30_POSITION_3 := 3036,
	LABELADJUSTMENT_MAGAZINE_DRAWER_1_CASSETTE_31_POSITION_1 := 3037,
	LABELADJUSTMENT_MAGAZINE_DRAWER_1_CASSETTE_31_POSITION_2 := 3038,
	LABELADJUSTMENT_MAGAZINE_DRAWER_1_CASSETTE_31_POSITION_3 := 3039,
	LABELADJUSTMENT_MAGAZINE_DRAWER_1_CASSETTE_32_POSITION_1 := 3040,
	LABELADJUSTMENT_MAGAZINE_DRAWER_1_CASSETTE_32_POSITION_2 := 3041,
	LABELADJUSTMENT_MAGAZINE_DRAWER_1_CASSETTE_32_POSITION_3 := 3042,
	LABELADJUSTMENT_MAGAZINE_DRAWER_2_CASSETTE_1_POSITION_1 := 3043,
	LABELADJUSTMENT_MAGAZINE_DRAWER_2_CASSETTE_1_POSITION_2 := 3044,
	LABELADJUSTMENT_MAGAZINE_DRAWER_2_CASSETTE_1_POSITION_3 := 3045,
	LABELADJUSTMENT_MAGAZINE_DRAWER_2_CASSETTE_2_POSITION_1 := 3046,
	LABELADJUSTMENT_MAGAZINE_DRAWER_2_CASSETTE_2_POSITION_2 := 3047,
	LABELADJUSTMENT_MAGAZINE_DRAWER_2_CASSETTE_2_POSITION_3 := 3048,
	LABELADJUSTMENT_MAGAZINE_DRAWER_2_CASSETTE_3_POSITION_1 := 3049,
	LABELADJUSTMENT_MAGAZINE_DRAWER_2_CASSETTE_3_POSITION_2 := 3050,
	LABELADJUSTMENT_MAGAZINE_DRAWER_2_CASSETTE_3_POSITION_3 := 3051,
	LABELADJUSTMENT_MAGAZINE_DRAWER_2_CASSETTE_4_POSITION_1 := 3052,
	LABELADJUSTMENT_MAGAZINE_DRAWER_2_CASSETTE_4_POSITION_2 := 3053,
	LABELADJUSTMENT_MAGAZINE_DRAWER_2_CASSETTE_4_POSITION_3 := 3054,
	LABELADJUSTMENT_MAGAZINE_DRAWER_2_CASSETTE_5_POSITION_1 := 3055,
	LABELADJUSTMENT_MAGAZINE_DRAWER_2_CASSETTE_5_POSITION_2 := 3056,
	LABELADJUSTMENT_MAGAZINE_DRAWER_2_CASSETTE_5_POSITION_3 := 3057,
	LABELADJUSTMENT_MAGAZINE_DRAWER_2_CASSETTE_6_POSITION_1 := 3058,
	LABELADJUSTMENT_MAGAZINE_DRAWER_2_CASSETTE_6_POSITION_2 := 3059,
	LABELADJUSTMENT_MAGAZINE_DRAWER_2_CASSETTE_6_POSITION_3 := 3060,
	LABELADJUSTMENT_MAGAZINE_DRAWER_2_CASSETTE_7_POSITION_1 := 3061,
	LABELADJUSTMENT_MAGAZINE_DRAWER_2_CASSETTE_7_POSITION_2 := 3062,
	LABELADJUSTMENT_MAGAZINE_DRAWER_2_CASSETTE_7_POSITION_3 := 3063,
	LABELADJUSTMENT_MAGAZINE_DRAWER_2_CASSETTE_8_POSITION_1 := 3064,
	LABELADJUSTMENT_MAGAZINE_DRAWER_2_CASSETTE_8_POSITION_2 := 3065,
	LABELADJUSTMENT_MAGAZINE_DRAWER_2_CASSETTE_8_POSITION_3 := 3066,
	LABELADJUSTMENT_MAGAZINE_DRAWER_2_CASSETTE_9_POSITION_1 := 3067,
	LABELADJUSTMENT_MAGAZINE_DRAWER_2_CASSETTE_9_POSITION_2 := 3068,
	LABELADJUSTMENT_MAGAZINE_DRAWER_2_CASSETTE_9_POSITION_3 := 3069,
	LABELADJUSTMENT_MAGAZINE_DRAWER_2_CASSETTE_10_POSITION_1 := 3070,
	LABELADJUSTMENT_MAGAZINE_DRAWER_2_CASSETTE_10_POSITION_2 := 3071,
	LABELADJUSTMENT_MAGAZINE_DRAWER_2_CASSETTE_10_POSITION_3 := 3072,
	LABELADJUSTMENT_MAGAZINE_DRAWER_2_CASSETTE_11_POSITION_1 := 3073,
	LABELADJUSTMENT_MAGAZINE_DRAWER_2_CASSETTE_11_POSITION_2 := 3074,
	LABELADJUSTMENT_MAGAZINE_DRAWER_2_CASSETTE_11_POSITION_3 := 3075,
	LABELADJUSTMENT_MAGAZINE_DRAWER_2_CASSETTE_12_POSITION_1 := 3076,
	LABELADJUSTMENT_MAGAZINE_DRAWER_2_CASSETTE_12_POSITION_2 := 3077,
	LABELADJUSTMENT_MAGAZINE_DRAWER_2_CASSETTE_12_POSITION_3 := 3078,
	LABELADJUSTMENT_MAGAZINE_DRAWER_2_CASSETTE_13_POSITION_1 := 3079,
	LABELADJUSTMENT_MAGAZINE_DRAWER_2_CASSETTE_13_POSITION_2 := 3080,
	LABELADJUSTMENT_MAGAZINE_DRAWER_2_CASSETTE_13_POSITION_3 := 3081,
	LABELADJUSTMENT_MAGAZINE_DRAWER_2_CASSETTE_14_POSITION_1 := 3082,
	LABELADJUSTMENT_MAGAZINE_DRAWER_2_CASSETTE_14_POSITION_2 := 3083,
	LABELADJUSTMENT_MAGAZINE_DRAWER_2_CASSETTE_14_POSITION_3 := 3084,
	LABELADJUSTMENT_MAGAZINE_DRAWER_2_CASSETTE_15_POSITION_1 := 3085,
	LABELADJUSTMENT_MAGAZINE_DRAWER_2_CASSETTE_15_POSITION_2 := 3086,
	LABELADJUSTMENT_MAGAZINE_DRAWER_2_CASSETTE_15_POSITION_3 := 3087,
	LABELADJUSTMENT_MAGAZINE_DRAWER_2_CASSETTE_16_POSITION_1 := 3088,
	LABELADJUSTMENT_MAGAZINE_DRAWER_2_CASSETTE_16_POSITION_2 := 3089,
	LABELADJUSTMENT_MAGAZINE_DRAWER_2_CASSETTE_16_POSITION_3 := 3090,
	LABELADJUSTMENT_MAGAZINE_DRAWER_2_CASSETTE_17_POSITION_1 := 3091,
	LABELADJUSTMENT_MAGAZINE_DRAWER_2_CASSETTE_17_POSITION_2 := 3092,
	LABELADJUSTMENT_MAGAZINE_DRAWER_2_CASSETTE_17_POSITION_3 := 3093,
	LABELADJUSTMENT_MAGAZINE_DRAWER_2_CASSETTE_18_POSITION_1 := 3094,
	LABELADJUSTMENT_MAGAZINE_DRAWER_2_CASSETTE_18_POSITION_2 := 3095,
	LABELADJUSTMENT_MAGAZINE_DRAWER_2_CASSETTE_18_POSITION_3 := 3096,
	LABELADJUSTMENT_MAGAZINE_DRAWER_2_CASSETTE_19_POSITION_1 := 3097,
	LABELADJUSTMENT_MAGAZINE_DRAWER_2_CASSETTE_19_POSITION_2 := 3098,
	LABELADJUSTMENT_MAGAZINE_DRAWER_2_CASSETTE_19_POSITION_3 := 3099,
	LABELADJUSTMENT_MAGAZINE_DRAWER_2_CASSETTE_20_POSITION_1 := 3100,
	LABELADJUSTMENT_MAGAZINE_DRAWER_2_CASSETTE_20_POSITION_2 := 3101,
	LABELADJUSTMENT_MAGAZINE_DRAWER_2_CASSETTE_20_POSITION_3 := 3102,
	LABELADJUSTMENT_MAGAZINE_DRAWER_2_CASSETTE_21_POSITION_1 := 3103,
	LABELADJUSTMENT_MAGAZINE_DRAWER_2_CASSETTE_21_POSITION_2 := 3104,
	LABELADJUSTMENT_MAGAZINE_DRAWER_2_CASSETTE_21_POSITION_3 := 3105,
	LABELADJUSTMENT_MAGAZINE_DRAWER_2_CASSETTE_22_POSITION_1 := 3106,
	LABELADJUSTMENT_MAGAZINE_DRAWER_2_CASSETTE_22_POSITION_2 := 3107,
	LABELADJUSTMENT_MAGAZINE_DRAWER_2_CASSETTE_22_POSITION_3 := 3108,
	LABELADJUSTMENT_MAGAZINE_DRAWER_2_CASSETTE_23_POSITION_1 := 3109,
	LABELADJUSTMENT_MAGAZINE_DRAWER_2_CASSETTE_23_POSITION_2 := 3110,
	LABELADJUSTMENT_MAGAZINE_DRAWER_2_CASSETTE_23_POSITION_3 := 3111,
	LABELADJUSTMENT_MAGAZINE_DRAWER_2_CASSETTE_24_POSITION_1 := 3112,
	LABELADJUSTMENT_MAGAZINE_DRAWER_2_CASSETTE_24_POSITION_2 := 3113,
	LABELADJUSTMENT_MAGAZINE_DRAWER_2_CASSETTE_24_POSITION_3 := 3114,
	LABELADJUSTMENT_MAGAZINE_DRAWER_2_CASSETTE_25_POSITION_1 := 3115,
	LABELADJUSTMENT_MAGAZINE_DRAWER_2_CASSETTE_25_POSITION_2 := 3116,
	LABELADJUSTMENT_MAGAZINE_DRAWER_2_CASSETTE_25_POSITION_3 := 3117,
	LABELADJUSTMENT_MAGAZINE_DRAWER_2_CASSETTE_26_POSITION_1 := 3118,
	LABELADJUSTMENT_MAGAZINE_DRAWER_2_CASSETTE_26_POSITION_2 := 3119,
	LABELADJUSTMENT_MAGAZINE_DRAWER_2_CASSETTE_26_POSITION_3 := 3120,
	LABELADJUSTMENT_MAGAZINE_DRAWER_2_CASSETTE_27_POSITION_1 := 3121,
	LABELADJUSTMENT_MAGAZINE_DRAWER_2_CASSETTE_27_POSITION_2 := 3122,
	LABELADJUSTMENT_MAGAZINE_DRAWER_2_CASSETTE_27_POSITION_3 := 3123,
	LABELADJUSTMENT_MAGAZINE_DRAWER_2_CASSETTE_28_POSITION_1 := 3124,
	LABELADJUSTMENT_MAGAZINE_DRAWER_2_CASSETTE_28_POSITION_2 := 3125,
	LABELADJUSTMENT_MAGAZINE_DRAWER_2_CASSETTE_28_POSITION_3 := 3126,
	LABELADJUSTMENT_MAGAZINE_DRAWER_2_CASSETTE_29_POSITION_1 := 3127,
	LABELADJUSTMENT_MAGAZINE_DRAWER_2_CASSETTE_29_POSITION_2 := 3128,
	LABELADJUSTMENT_MAGAZINE_DRAWER_2_CASSETTE_29_POSITION_3 := 3129,
	LABELADJUSTMENT_MAGAZINE_DRAWER_2_CASSETTE_30_POSITION_1 := 3130,
	LABELADJUSTMENT_MAGAZINE_DRAWER_2_CASSETTE_30_POSITION_2 := 3131,
	LABELADJUSTMENT_MAGAZINE_DRAWER_2_CASSETTE_30_POSITION_3 := 3132,
	LABELADJUSTMENT_MAGAZINE_DRAWER_2_CASSETTE_31_POSITION_1 := 3133,
	LABELADJUSTMENT_MAGAZINE_DRAWER_2_CASSETTE_31_POSITION_2 := 3134,
	LABELADJUSTMENT_MAGAZINE_DRAWER_2_CASSETTE_31_POSITION_3 := 3135,
	LABELADJUSTMENT_MAGAZINE_DRAWER_2_CASSETTE_32_POSITION_1 := 3136,
	LABELADJUSTMENT_MAGAZINE_DRAWER_2_CASSETTE_32_POSITION_2 := 3137,
	LABELADJUSTMENT_MAGAZINE_DRAWER_2_CASSETTE_32_POSITION_3 := 3138,
	LABELADJUSTMENT_MAGAZINE_2_DRAWER_1_CASSETTE_1_POSITION_1 := 3139,
	LABELADJUSTMENT_MAGAZINE_2_DRAWER_1_CASSETTE_1_POSITION_2 := 3140,
	LABELADJUSTMENT_MAGAZINE_2_DRAWER_1_CASSETTE_1_POSITION_3 := 3141,
	LABELADJUSTMENT_MAGAZINE_2_DRAWER_1_CASSETTE_2_POSITION_1 := 3142,
	LABELADJUSTMENT_MAGAZINE_2_DRAWER_1_CASSETTE_2_POSITION_2 := 3143,
	LABELADJUSTMENT_MAGAZINE_2_DRAWER_1_CASSETTE_2_POSITION_3 := 3144,
	LABELADJUSTMENT_MAGAZINE_2_DRAWER_1_CASSETTE_3_POSITION_1 := 3145,
	LABELADJUSTMENT_MAGAZINE_2_DRAWER_1_CASSETTE_3_POSITION_2 := 3146,
	LABELADJUSTMENT_MAGAZINE_2_DRAWER_1_CASSETTE_3_POSITION_3 := 3147,
	LABELADJUSTMENT_MAGAZINE_2_DRAWER_1_CASSETTE_4_POSITION_1 := 3148,
	LABELADJUSTMENT_MAGAZINE_2_DRAWER_1_CASSETTE_4_POSITION_2 := 3149,
	LABELADJUSTMENT_MAGAZINE_2_DRAWER_1_CASSETTE_4_POSITION_3 := 3150,
	LABELADJUSTMENT_MAGAZINE_2_DRAWER_1_CASSETTE_5_POSITION_1 := 3151,
	LABELADJUSTMENT_MAGAZINE_2_DRAWER_1_CASSETTE_5_POSITION_2 := 3152,
	LABELADJUSTMENT_MAGAZINE_2_DRAWER_1_CASSETTE_5_POSITION_3 := 3153,
	LABELADJUSTMENT_MAGAZINE_2_DRAWER_1_CASSETTE_6_POSITION_1 := 3154,
	LABELADJUSTMENT_MAGAZINE_2_DRAWER_1_CASSETTE_6_POSITION_2 := 3155,
	LABELADJUSTMENT_MAGAZINE_2_DRAWER_1_CASSETTE_6_POSITION_3 := 3156,
	LABELADJUSTMENT_MAGAZINE_2_DRAWER_1_CASSETTE_7_POSITION_1 := 3157,
	LABELADJUSTMENT_MAGAZINE_2_DRAWER_1_CASSETTE_7_POSITION_2 := 3158,
	LABELADJUSTMENT_MAGAZINE_2_DRAWER_1_CASSETTE_7_POSITION_3 := 3159,
	LABELADJUSTMENT_MAGAZINE_2_DRAWER_1_CASSETTE_8_POSITION_1 := 3160,
	LABELADJUSTMENT_MAGAZINE_2_DRAWER_1_CASSETTE_8_POSITION_2 := 3161,
	LABELADJUSTMENT_MAGAZINE_2_DRAWER_1_CASSETTE_8_POSITION_3 := 3162,
	LABELADJUSTMENT_MAGAZINE_2_DRAWER_1_CASSETTE_9_POSITION_1 := 3163,
	LABELADJUSTMENT_MAGAZINE_2_DRAWER_1_CASSETTE_9_POSITION_2 := 3164,
	LABELADJUSTMENT_MAGAZINE_2_DRAWER_1_CASSETTE_9_POSITION_3 := 3165,
	LABELADJUSTMENT_MAGAZINE_2_DRAWER_1_CASSETTE_10_POSITION_1 := 3166,
	LABELADJUSTMENT_MAGAZINE_2_DRAWER_1_CASSETTE_10_POSITION_2 := 3167,
	LABELADJUSTMENT_MAGAZINE_2_DRAWER_1_CASSETTE_10_POSITION_3 := 3168,
	LABELADJUSTMENT_MAGAZINE_2_DRAWER_1_CASSETTE_11_POSITION_1 := 3169,
	LABELADJUSTMENT_MAGAZINE_2_DRAWER_1_CASSETTE_11_POSITION_2 := 3170,
	LABELADJUSTMENT_MAGAZINE_2_DRAWER_1_CASSETTE_11_POSITION_3 := 3171,
	LABELADJUSTMENT_MAGAZINE_2_DRAWER_1_CASSETTE_12_POSITION_1 := 3172,
	LABELADJUSTMENT_MAGAZINE_2_DRAWER_1_CASSETTE_12_POSITION_2 := 3173,
	LABELADJUSTMENT_MAGAZINE_2_DRAWER_1_CASSETTE_12_POSITION_3 := 3174,
	LABELADJUSTMENT_MAGAZINE_2_DRAWER_1_CASSETTE_13_POSITION_1 := 3175,
	LABELADJUSTMENT_MAGAZINE_2_DRAWER_1_CASSETTE_13_POSITION_2 := 3176,
	LABELADJUSTMENT_MAGAZINE_2_DRAWER_1_CASSETTE_13_POSITION_3 := 3177,
	LABELADJUSTMENT_MAGAZINE_2_DRAWER_1_CASSETTE_14_POSITION_1 := 3178,
	LABELADJUSTMENT_MAGAZINE_2_DRAWER_1_CASSETTE_14_POSITION_2 := 3179,
	LABELADJUSTMENT_MAGAZINE_2_DRAWER_1_CASSETTE_14_POSITION_3 := 3180,
	LABELADJUSTMENT_MAGAZINE_2_DRAWER_1_CASSETTE_15_POSITION_1 := 3181,
	LABELADJUSTMENT_MAGAZINE_2_DRAWER_1_CASSETTE_15_POSITION_2 := 3182,
	LABELADJUSTMENT_MAGAZINE_2_DRAWER_1_CASSETTE_15_POSITION_3 := 3183,
	LABELADJUSTMENT_MAGAZINE_2_DRAWER_1_CASSETTE_16_POSITION_1 := 3184,
	LABELADJUSTMENT_MAGAZINE_2_DRAWER_1_CASSETTE_16_POSITION_2 := 3185,
	LABELADJUSTMENT_MAGAZINE_2_DRAWER_1_CASSETTE_16_POSITION_3 := 3186,
	LABELADJUSTMENT_MAGAZINE_2_DRAWER_1_CASSETTE_17_POSITION_1 := 3187,
	LABELADJUSTMENT_MAGAZINE_2_DRAWER_1_CASSETTE_17_POSITION_2 := 3188,
	LABELADJUSTMENT_MAGAZINE_2_DRAWER_1_CASSETTE_17_POSITION_3 := 3189,
	LABELADJUSTMENT_MAGAZINE_2_DRAWER_1_CASSETTE_18_POSITION_1 := 3190,
	LABELADJUSTMENT_MAGAZINE_2_DRAWER_1_CASSETTE_18_POSITION_2 := 3191,
	LABELADJUSTMENT_MAGAZINE_2_DRAWER_1_CASSETTE_18_POSITION_3 := 3192,
	LABELADJUSTMENT_MAGAZINE_2_DRAWER_1_CASSETTE_19_POSITION_1 := 3193,
	LABELADJUSTMENT_MAGAZINE_2_DRAWER_1_CASSETTE_19_POSITION_2 := 3194,
	LABELADJUSTMENT_MAGAZINE_2_DRAWER_1_CASSETTE_19_POSITION_3 := 3195,
	LABELADJUSTMENT_MAGAZINE_2_DRAWER_1_CASSETTE_20_POSITION_1 := 3196,
	LABELADJUSTMENT_MAGAZINE_2_DRAWER_1_CASSETTE_20_POSITION_2 := 3197,
	LABELADJUSTMENT_MAGAZINE_2_DRAWER_1_CASSETTE_20_POSITION_3 := 3198,
	LABELADJUSTMENT_MAGAZINE_2_DRAWER_1_CASSETTE_21_POSITION_1 := 3199,
	LABELADJUSTMENT_MAGAZINE_2_DRAWER_1_CASSETTE_21_POSITION_2 := 3200,
	LABELADJUSTMENT_MAGAZINE_2_DRAWER_1_CASSETTE_21_POSITION_3 := 3201,
	LABELADJUSTMENT_MAGAZINE_2_DRAWER_1_CASSETTE_22_POSITION_1 := 3202,
	LABELADJUSTMENT_MAGAZINE_2_DRAWER_1_CASSETTE_22_POSITION_2 := 3203,
	LABELADJUSTMENT_MAGAZINE_2_DRAWER_1_CASSETTE_22_POSITION_3 := 3204,
	LABELADJUSTMENT_MAGAZINE_2_DRAWER_1_CASSETTE_23_POSITION_1 := 3205,
	LABELADJUSTMENT_MAGAZINE_2_DRAWER_1_CASSETTE_23_POSITION_2 := 3206,
	LABELADJUSTMENT_MAGAZINE_2_DRAWER_1_CASSETTE_23_POSITION_3 := 3207,
	LABELADJUSTMENT_MAGAZINE_2_DRAWER_1_CASSETTE_24_POSITION_1 := 3208,
	LABELADJUSTMENT_MAGAZINE_2_DRAWER_1_CASSETTE_24_POSITION_2 := 3209,
	LABELADJUSTMENT_MAGAZINE_2_DRAWER_1_CASSETTE_24_POSITION_3 := 3210,
	LABELADJUSTMENT_MAGAZINE_2_DRAWER_1_CASSETTE_25_POSITION_1 := 3211,
	LABELADJUSTMENT_MAGAZINE_2_DRAWER_1_CASSETTE_25_POSITION_2 := 3212,
	LABELADJUSTMENT_MAGAZINE_2_DRAWER_1_CASSETTE_25_POSITION_3 := 3213,
	LABELADJUSTMENT_MAGAZINE_2_DRAWER_1_CASSETTE_26_POSITION_1 := 3214,
	LABELADJUSTMENT_MAGAZINE_2_DRAWER_1_CASSETTE_26_POSITION_2 := 3215,
	LABELADJUSTMENT_MAGAZINE_2_DRAWER_1_CASSETTE_26_POSITION_3 := 3216,
	LABELADJUSTMENT_MAGAZINE_2_DRAWER_1_CASSETTE_27_POSITION_1 := 3217,
	LABELADJUSTMENT_MAGAZINE_2_DRAWER_1_CASSETTE_27_POSITION_2 := 3218,
	LABELADJUSTMENT_MAGAZINE_2_DRAWER_1_CASSETTE_27_POSITION_3 := 3219,
	LABELADJUSTMENT_MAGAZINE_2_DRAWER_1_CASSETTE_28_POSITION_1 := 3220,
	LABELADJUSTMENT_MAGAZINE_2_DRAWER_1_CASSETTE_28_POSITION_2 := 3221,
	LABELADJUSTMENT_MAGAZINE_2_DRAWER_1_CASSETTE_28_POSITION_3 := 3222,
	LABELADJUSTMENT_MAGAZINE_2_DRAWER_1_CASSETTE_29_POSITION_1 := 3223,
	LABELADJUSTMENT_MAGAZINE_2_DRAWER_1_CASSETTE_29_POSITION_2 := 3224,
	LABELADJUSTMENT_MAGAZINE_2_DRAWER_1_CASSETTE_29_POSITION_3 := 3225,
	LABELADJUSTMENT_MAGAZINE_2_DRAWER_1_CASSETTE_30_POSITION_1 := 3226,
	LABELADJUSTMENT_MAGAZINE_2_DRAWER_1_CASSETTE_30_POSITION_2 := 3227,
	LABELADJUSTMENT_MAGAZINE_2_DRAWER_1_CASSETTE_30_POSITION_3 := 3228,
	LABELADJUSTMENT_MAGAZINE_2_DRAWER_1_CASSETTE_31_POSITION_1 := 3229,
	LABELADJUSTMENT_MAGAZINE_2_DRAWER_1_CASSETTE_31_POSITION_2 := 3230,
	LABELADJUSTMENT_MAGAZINE_2_DRAWER_1_CASSETTE_31_POSITION_3 := 3231,
	LABELADJUSTMENT_MAGAZINE_2_DRAWER_1_CASSETTE_32_POSITION_1 := 3232,
	LABELADJUSTMENT_MAGAZINE_2_DRAWER_1_CASSETTE_32_POSITION_2 := 3233,
	LABELADJUSTMENT_MAGAZINE_2_DRAWER_1_CASSETTE_32_POSITION_3 := 3234,
	LABELADJUSTMENT_MAGAZINE_2_DRAWER_2_CASSETTE_1_POSITION_1 := 3235,
	LABELADJUSTMENT_MAGAZINE_2_DRAWER_2_CASSETTE_1_POSITION_2 := 3236,
	LABELADJUSTMENT_MAGAZINE_2_DRAWER_2_CASSETTE_1_POSITION_3 := 3237,
	LABELADJUSTMENT_MAGAZINE_2_DRAWER_2_CASSETTE_2_POSITION_1 := 3238,
	LABELADJUSTMENT_MAGAZINE_2_DRAWER_2_CASSETTE_2_POSITION_2 := 3239,
	LABELADJUSTMENT_MAGAZINE_2_DRAWER_2_CASSETTE_2_POSITION_3 := 3240,
	LABELADJUSTMENT_MAGAZINE_2_DRAWER_2_CASSETTE_3_POSITION_1 := 3241,
	LABELADJUSTMENT_MAGAZINE_2_DRAWER_2_CASSETTE_3_POSITION_2 := 3242,
	LABELADJUSTMENT_MAGAZINE_2_DRAWER_2_CASSETTE_3_POSITION_3 := 3243,
	LABELADJUSTMENT_MAGAZINE_2_DRAWER_2_CASSETTE_4_POSITION_1 := 3244,
	LABELADJUSTMENT_MAGAZINE_2_DRAWER_2_CASSETTE_4_POSITION_2 := 3245,
	LABELADJUSTMENT_MAGAZINE_2_DRAWER_2_CASSETTE_4_POSITION_3 := 3246,
	LABELADJUSTMENT_MAGAZINE_2_DRAWER_2_CASSETTE_5_POSITION_1 := 3247,
	LABELADJUSTMENT_MAGAZINE_2_DRAWER_2_CASSETTE_5_POSITION_2 := 3248,
	LABELADJUSTMENT_MAGAZINE_2_DRAWER_2_CASSETTE_5_POSITION_3 := 3249,
	LABELADJUSTMENT_MAGAZINE_2_DRAWER_2_CASSETTE_6_POSITION_1 := 3250,
	LABELADJUSTMENT_MAGAZINE_2_DRAWER_2_CASSETTE_6_POSITION_2 := 3251,
	LABELADJUSTMENT_MAGAZINE_2_DRAWER_2_CASSETTE_6_POSITION_3 := 3252,
	LABELADJUSTMENT_MAGAZINE_2_DRAWER_2_CASSETTE_7_POSITION_1 := 3253,
	LABELADJUSTMENT_MAGAZINE_2_DRAWER_2_CASSETTE_7_POSITION_2 := 3254,
	LABELADJUSTMENT_MAGAZINE_2_DRAWER_2_CASSETTE_7_POSITION_3 := 3255,
	LABELADJUSTMENT_MAGAZINE_2_DRAWER_2_CASSETTE_8_POSITION_1 := 3256,
	LABELADJUSTMENT_MAGAZINE_2_DRAWER_2_CASSETTE_8_POSITION_2 := 3257,
	LABELADJUSTMENT_MAGAZINE_2_DRAWER_2_CASSETTE_8_POSITION_3 := 3258,
	LABELADJUSTMENT_MAGAZINE_2_DRAWER_2_CASSETTE_9_POSITION_1 := 3259,
	LABELADJUSTMENT_MAGAZINE_2_DRAWER_2_CASSETTE_9_POSITION_2 := 3260,
	LABELADJUSTMENT_MAGAZINE_2_DRAWER_2_CASSETTE_9_POSITION_3 := 3261,
	LABELADJUSTMENT_MAGAZINE_2_DRAWER_2_CASSETTE_10_POSITION_1 := 3262,
	LABELADJUSTMENT_MAGAZINE_2_DRAWER_2_CASSETTE_10_POSITION_2 := 3263,
	LABELADJUSTMENT_MAGAZINE_2_DRAWER_2_CASSETTE_10_POSITION_3 := 3264,
	LABELADJUSTMENT_MAGAZINE_2_DRAWER_2_CASSETTE_11_POSITION_1 := 3265,
	LABELADJUSTMENT_MAGAZINE_2_DRAWER_2_CASSETTE_11_POSITION_2 := 3266,
	LABELADJUSTMENT_MAGAZINE_2_DRAWER_2_CASSETTE_11_POSITION_3 := 3267,
	LABELADJUSTMENT_MAGAZINE_2_DRAWER_2_CASSETTE_12_POSITION_1 := 3268,
	LABELADJUSTMENT_MAGAZINE_2_DRAWER_2_CASSETTE_12_POSITION_2 := 3269,
	LABELADJUSTMENT_MAGAZINE_2_DRAWER_2_CASSETTE_12_POSITION_3 := 3270,
	LABELADJUSTMENT_MAGAZINE_2_DRAWER_2_CASSETTE_13_POSITION_1 := 3271,
	LABELADJUSTMENT_MAGAZINE_2_DRAWER_2_CASSETTE_13_POSITION_2 := 3272,
	LABELADJUSTMENT_MAGAZINE_2_DRAWER_2_CASSETTE_13_POSITION_3 := 3273,
	LABELADJUSTMENT_MAGAZINE_2_DRAWER_2_CASSETTE_14_POSITION_1 := 3274,
	LABELADJUSTMENT_MAGAZINE_2_DRAWER_2_CASSETTE_14_POSITION_2 := 3275,
	LABELADJUSTMENT_MAGAZINE_2_DRAWER_2_CASSETTE_14_POSITION_3 := 3276,
	LABELADJUSTMENT_MAGAZINE_2_DRAWER_2_CASSETTE_15_POSITION_1 := 3277,
	LABELADJUSTMENT_MAGAZINE_2_DRAWER_2_CASSETTE_15_POSITION_2 := 3278,
	LABELADJUSTMENT_MAGAZINE_2_DRAWER_2_CASSETTE_15_POSITION_3 := 3279,
	LABELADJUSTMENT_MAGAZINE_2_DRAWER_2_CASSETTE_16_POSITION_1 := 3280,
	LABELADJUSTMENT_MAGAZINE_2_DRAWER_2_CASSETTE_16_POSITION_2 := 3281,
	LABELADJUSTMENT_MAGAZINE_2_DRAWER_2_CASSETTE_16_POSITION_3 := 3282,
	LABELADJUSTMENT_MAGAZINE_2_DRAWER_2_CASSETTE_17_POSITION_1 := 3283,
	LABELADJUSTMENT_MAGAZINE_2_DRAWER_2_CASSETTE_17_POSITION_2 := 3284,
	LABELADJUSTMENT_MAGAZINE_2_DRAWER_2_CASSETTE_17_POSITION_3 := 3285,
	LABELADJUSTMENT_MAGAZINE_2_DRAWER_2_CASSETTE_18_POSITION_1 := 3286,
	LABELADJUSTMENT_MAGAZINE_2_DRAWER_2_CASSETTE_18_POSITION_2 := 3287,
	LABELADJUSTMENT_MAGAZINE_2_DRAWER_2_CASSETTE_18_POSITION_3 := 3288,
	LABELADJUSTMENT_MAGAZINE_2_DRAWER_2_CASSETTE_19_POSITION_1 := 3289,
	LABELADJUSTMENT_MAGAZINE_2_DRAWER_2_CASSETTE_19_POSITION_2 := 3290,
	LABELADJUSTMENT_MAGAZINE_2_DRAWER_2_CASSETTE_19_POSITION_3 := 3291,
	LABELADJUSTMENT_MAGAZINE_2_DRAWER_2_CASSETTE_20_POSITION_1 := 3292,
	LABELADJUSTMENT_MAGAZINE_2_DRAWER_2_CASSETTE_20_POSITION_2 := 3293,
	LABELADJUSTMENT_MAGAZINE_2_DRAWER_2_CASSETTE_20_POSITION_3 := 3294,
	LABELADJUSTMENT_MAGAZINE_2_DRAWER_2_CASSETTE_21_POSITION_1 := 3295,
	LABELADJUSTMENT_MAGAZINE_2_DRAWER_2_CASSETTE_21_POSITION_2 := 3296,
	LABELADJUSTMENT_MAGAZINE_2_DRAWER_2_CASSETTE_21_POSITION_3 := 3297,
	LABELADJUSTMENT_MAGAZINE_2_DRAWER_2_CASSETTE_22_POSITION_1 := 3298,
	LABELADJUSTMENT_MAGAZINE_2_DRAWER_2_CASSETTE_22_POSITION_2 := 3299,
	LABELADJUSTMENT_MAGAZINE_2_DRAWER_2_CASSETTE_22_POSITION_3 := 3300,
	LABELADJUSTMENT_MAGAZINE_2_DRAWER_2_CASSETTE_23_POSITION_1 := 3301,
	LABELADJUSTMENT_MAGAZINE_2_DRAWER_2_CASSETTE_23_POSITION_2 := 3302,
	LABELADJUSTMENT_MAGAZINE_2_DRAWER_2_CASSETTE_23_POSITION_3 := 3303,
	LABELADJUSTMENT_MAGAZINE_2_DRAWER_2_CASSETTE_24_POSITION_1 := 3304,
	LABELADJUSTMENT_MAGAZINE_2_DRAWER_2_CASSETTE_24_POSITION_2 := 3305,
	LABELADJUSTMENT_MAGAZINE_2_DRAWER_2_CASSETTE_24_POSITION_3 := 3306,
	LABELADJUSTMENT_MAGAZINE_2_DRAWER_2_CASSETTE_25_POSITION_1 := 3307,
	LABELADJUSTMENT_MAGAZINE_2_DRAWER_2_CASSETTE_25_POSITION_2 := 3308,
	LABELADJUSTMENT_MAGAZINE_2_DRAWER_2_CASSETTE_25_POSITION_3 := 3309,
	LABELADJUSTMENT_MAGAZINE_2_DRAWER_2_CASSETTE_26_POSITION_1 := 3310,
	LABELADJUSTMENT_MAGAZINE_2_DRAWER_2_CASSETTE_26_POSITION_2 := 3311,
	LABELADJUSTMENT_MAGAZINE_2_DRAWER_2_CASSETTE_26_POSITION_3 := 3312,
	LABELADJUSTMENT_MAGAZINE_2_DRAWER_2_CASSETTE_27_POSITION_1 := 3313,
	LABELADJUSTMENT_MAGAZINE_2_DRAWER_2_CASSETTE_27_POSITION_2 := 3314,
	LABELADJUSTMENT_MAGAZINE_2_DRAWER_2_CASSETTE_27_POSITION_3 := 3315,
	LABELADJUSTMENT_MAGAZINE_2_DRAWER_2_CASSETTE_28_POSITION_1 := 3316,
	LABELADJUSTMENT_MAGAZINE_2_DRAWER_2_CASSETTE_28_POSITION_2 := 3317,
	LABELADJUSTMENT_MAGAZINE_2_DRAWER_2_CASSETTE_28_POSITION_3 := 3318,
	LABELADJUSTMENT_MAGAZINE_2_DRAWER_2_CASSETTE_29_POSITION_1 := 3319,
	LABELADJUSTMENT_MAGAZINE_2_DRAWER_2_CASSETTE_29_POSITION_2 := 3320,
	LABELADJUSTMENT_MAGAZINE_2_DRAWER_2_CASSETTE_29_POSITION_3 := 3321,
	LABELADJUSTMENT_MAGAZINE_2_DRAWER_2_CASSETTE_30_POSITION_1 := 3322,
	LABELADJUSTMENT_MAGAZINE_2_DRAWER_2_CASSETTE_30_POSITION_2 := 3323,
	LABELADJUSTMENT_MAGAZINE_2_DRAWER_2_CASSETTE_30_POSITION_3 := 3324,
	LABELADJUSTMENT_MAGAZINE_2_DRAWER_2_CASSETTE_31_POSITION_1 := 3325,
	LABELADJUSTMENT_MAGAZINE_2_DRAWER_2_CASSETTE_31_POSITION_2 := 3326,
	LABELADJUSTMENT_MAGAZINE_2_DRAWER_2_CASSETTE_31_POSITION_3 := 3327,
	LABELADJUSTMENT_MAGAZINE_2_DRAWER_2_CASSETTE_32_POSITION_1 := 3328,
	LABELADJUSTMENT_MAGAZINE_2_DRAWER_2_CASSETTE_32_POSITION_2 := 3329,
	LABELADJUSTMENT_MAGAZINE_2_DRAWER_2_CASSETTE_32_POSITION_3 := 3330
);
END_TYPE
